(* IEC 61131-3 sources: ml2plc/benchmarks/st (part 5) *)

(* ---- GRU3.st ---- *)
FUNCTION_BLOCK GRU3_FB

    (* Model Inputs/Outputs *)
VAR_INPUT
    input_data : REAL;
END_VAR

VAR_OUTPUT
    output_data : ARRAY[0..2] OF REAL;
END_VAR

VAR CONSTANT
    weights_0_u : ARRAY[0..63] OF REAL := [-0.439286172, -0.480953246, -0.870120704, -0.69075644, -0.657077134, -0.589701712, -0.481989682, 0.11155279, -0.595970333, -0.522424638, 0.066479668, -0.477147967, -0.548775792, -0.440251201, -0.581660211, -0.851885259, -0.447049588, -0.158783153, -0.671791077, -0.790636778, -0.670549393, -0.228230864, -0.573410928, -0.463102937, 0.294410557, -0.154226393, -0.428246915, -0.419357181, -0.580893517, -0.450942427, -0.434489578, -0.354421765, -0.500179946, -0.272357315, -0.211979702, -0.347913235, -0.509638548, -0.571337163, -0.666850746, -0.102425002, -0.464207053, -0.692536592, -0.576414764, -0.25179112, -0.587422669, 0.197722241, -0.440594107, -0.0186067764, -0.233214989, -0.485925347, -0.624329388, -0.464201093, -0.771930814, -0.648595512, -0.712386131, -0.865132749, 0.0861109644, -0.699016631, -0.64285028, -0.76548481, -0.601012945, -0.522387683, -0.408631802, -0.428571761];
    recurrent_0_u : ARRAY[0..4095] OF REAL := [-0.0650523901, -0.129474998, 0.0260338224, 0.0695474148, -0.0666072816, 0.0774139315, -0.0643586814, 0.0473090038, 0.0519357473, 0.0531803295, 0.0508824363, 0.156312734, 0.0510548055, -0.0783398449, 0.0161208138, -0.0254090969, -0.0333776586, 0.0407715552, 0.0384992361, -0.00284529058, 0.0996260718, -0.0809974, -0.0287103504, 0.0288348049, 0.121645145, 0.129295856, -0.121905953, -0.0567066036, -0.0332944021, 0.10126324, -0.0619100034, -0.0120835379, -0.0321507938, 0.152141571, 0.0557904243, 0.0295200478, 0.0753500834, 0.0523380376, -0.045079913, 0.0743025169, 0.03919724, -0.0464075021, 0.0460194834, 0.0400504917, -0.0186564252, -0.0811230615, 0.0205100551, -0.0494997241, -0.0123350881, -0.0521072671, 0.0318819955, 0.0125074722, 0.086325638, -0.14838697, 0.0729614198, -0.123611242, 0.0608778223, 0.136695266, -0.0275732893, 0.103986211, 0.0964937732, 0.0746636614, 0.0518375002, 0.0131850429, 0.0481536575, 0.080832839, 0.00456657633, -0.0930995643, -0.0926894546, -0.104142435, -0.0113655347, 0.0689256042, 0.0391013213, -0.145912498, 0.0662881434, -0.125198483, -0.0359372757, 0.0683884099, 0.0814840198, -0.0467883013, -0.0385110751, 0.0412478335, -0.026082132, 0.00598589424, -0.0733542442, -0.0616489351, 0.0599563681, 0.0975151584, -0.102699503, 0.0168768093, 0.0567795113, -0.109472096, 0.0479807556, -0.0641779676, 0.0252187103, 0.0170151237, 0.052396398, -0.00687042344, -0.0297337286, 0.052699931, 0.0299865901, 0.0428941771, 0.143816575, 0.0724755228, 0.0308377538, 0.0377355814, 0.073744677, 0.100715749, 0.0200833306, 0.00330035621, 0.0808146596, 0.0683915466, 0.00292335614, -0.0387148745, -0.0278775394, 0.0165898427, -0.0266524255, -0.0119600557, 0.0607938841, -0.171499431, 0.00670967251, -0.0278419442, -0.0198536664, -0.0489947647, -0.0504177436, -0.0603820346, -0.0319245569, 0.0403733216, -0.0657449737, -0.0835127532, 0.074783206, -0.0822283328, 0.0527420714, 0.025356207, 0.00193200377, 0.0403062142, 0.011863322, 0.0911065713, -0.0981498286, 0.0448010042, 0.00674223201, 0.0832657516, 0.0133088445, -0.0096457703, -0.126930133, 0.0133038349, -0.0605163276, 0.0315002874, 0.163095102, 0.0627945811, -0.0319333449, -0.0184467398, -0.0260825343, 0.1507947, 0.0180257969, -0.113473095, -0.00113128126, 0.034390863, 0.158128366, 0.0736147836, 0.00302845053, -0.0366435051, 0.0202366989, -0.0454519801, 0.027544789, 0.00827108417, -0.116445266, 0.136078835, -0.0322153643, 0.0859275237, -0.0495595485, -0.0305913445, -0.0528560281, -0.0197725855, 0.0479791425, -0.0321966782, -0.0912050977, 0.08009094, -0.131073937, -0.073050648, 0.0158983283, -0.0129424734, 0.0236992333, -0.0654924586, 0.00780409761, 0.0303560495, 0.0224402416, 0.195856482, 0.104409501, 0.00386209786, 0.0270838067, -0.0308708213, 0.0765376315, -0.144475698, -0.00663482724, -0.0773844719, -0.0756781921, 0.0114769517, 0.07947056, 0.0525699407, -0.0490815043, -0.0797774196, -0.0738181025, 0.00899818353, 0.00655652676, -0.0247584134, -0.142790094, -0.0536906458, 0.0891067088, 0.0319167599, 0.0273121186, -0.0111009832, 0.0738681182, -0.0465159416, 0.10495235, 0.0167910457, 0.0170945786, -0.0259337351, -0.0238404684, 0.105175085, 0.0262874551, -0.0252160784, 0.0407399312, 0.0396488942, -0.000441844575, 0.0779087767, -0.101633228, 0.00611562654, -0.138864547, 0.0793924779, 0.0318161361, 0.00487799011, -0.0742631257, 0.0282261875, -0.0452414677, 0.103862561, -0.233050048, 0.0166822113, -0.0502803773, -0.105138443, 0.00815397315, 0.075144209, -0.000656956807, 0.00553116389, -0.0327767022, 0.0563323051, 0.00168130081, -0.0347454548, 0.0447669849, 0.0809304044, 0.0181033891, 0.0829547346, 0.0445744358, 0.0685421899, -0.0522269495, 0.10767854, 0.0401147828, -0.0274171568, -0.0556086302, -0.0181052946, 0.0614649057, 0.15146631, -0.107644446, -0.0519810207, -0.0192557313, -0.050705526, -0.00130558573, -0.00449152011, 0.0586461015, -0.00949175656, -0.161170155, 0.0415757112, 0.0234208908, 0.0994374529, -0.107094176, 0.0798551813, 0.00859866291, 0.00905988738, 0.17884995, -0.052185487, -0.00788529217, -0.0128635718, 0.0425841771, -0.0781655982, 0.0738354772, -0.0700388551, -0.0454497337, -0.0581207834, 0.0587512478, -0.129331231, 0.089504689, 0.0157049354, 0.0867228657, 0.0273658019, -0.0242159963, -0.0269595832, -0.0785825849, -0.0127460342, 0.0726092383, -0.0813473612, 0.0418060534, -0.098036088, -0.0871397629, 0.12796244, 0.115513436, -0.0840419456, -0.0282502882, 0.0339900963, -0.0615085512, -0.0237938426, 0.14066948, 0.0103495289, 0.0563306212, 0.0128910914, 0.0566199236, -0.0431611128, 0.0414758436, -0.0598706417, -0.00455367938, 0.010008106, 0.0502123758, -0.0128066251, 0.119871259, 0.169338882, 0.0573619083, -0.00254678726, 0.0632556081, 0.0658841059, -0.0489678681, -0.0136197284, 0.0332296528, 0.0304199178, -0.0101228859, 0.0340865031, -0.1463456, -0.0561735369, -0.078145586, -0.105770409, 0.021583017, 0.0442470424, -0.0132950321, 0.0343763754, -0.131868333, -0.0834302157, 0.0234229043, 0.0955413878, -0.00966519676, 0.133738831, 0.0799299628, -0.0209413245, -0.0201649163, -0.078094773, 0.00760632753, 0.10674265, -0.0504244342, 0.130076349, -0.0765756071, 0.0406672917, -0.0677179396, 0.0489641167, 0.0178483911, 0.0639283434, -0.0072317142, 0.0689901859, 0.0284034405, 0.0447224788, 0.080589503, -0.0753613785, -0.0883018747, -0.209824249, -0.025372155, -0.0194213465, -0.121756315, -0.0405391641, 0.0252318978, -0.113081403, 0.00984102953, -0.0379814059, -0.0696330816, -0.0607138053, 0.00136227917, -0.0684736297, 0.084016636, 0.0580409989, 0.0783514529, 0.038732525, -0.110764012, -0.184509531, -0.0218135417, 0.0410628468, 0.0143347979, 0.0210808329, 0.0938048959, 0.0952843726, 0.0369632132, -0.036689274, 0.0596370548, -0.101092562, 0.021979671, -0.00666903984, -0.0002728533, -0.102687143, 0.101846725, -0.0270557068, -0.0740891248, 0.0451480709, 0.0244468898, 0.0135530774, -0.0656716228, 0.126964301, 0.046734333, -0.0135823097, 0.104897536, 0.0116401128, -0.0351510793, -0.0270920806, -0.0317737125, -0.0427896604, 0.0606436953, -0.055717431, 0.0877809376, 0.0525183901, 0.0816646814, -0.123816505, 0.0268022101, 0.0949827731, 0.0286988262, -1.17924064e-05, -0.107156947, -0.0325826406, -0.176235095, 0.0207939055, 0.140304744, 0.0597819574, -0.0181577466, 0.117161281, 0.0191873126, 0.0420570076, 0.0174266361, 0.0642305687, -0.0820301622, 0.0203213636, -0.0772711709, 0.0149432123, 0.078445442, -0.031391941, 0.0178297423, 0.0258787423, 0.105060086, -0.185030684, -0.0465904325, 0.033022128, -0.0522077605, 0.18817015, 0.17154251, 0.0908443928, -0.114609689, -0.0463253893, 0.179783046, -0.0138813183, -0.0250236578, -0.0397495851, -0.0401404127, 0.0414455384, 0.00421553105, 0.00501056761, -0.0355476104, -0.0948569328, -0.0180768073, -0.0929266214, -6.38996717e-05, 0.0402616151, -0.04017644, 0.0292976033, 0.122893214, -0.0101269074, 0.0949848741, 0.0924490988, -0.0142561533, 0.034249723, -0.0345417485, -0.0720876306, -0.116285995, 0.0757803917, 0.0925265029, 0.0501283891, 0.0556523763, -0.0871114284, 0.063929759, 0.111392535, -0.0113485595, -0.0560661219, 0.0588565171, 0.0202990752, 0.0169391409, 0.0079346532, -0.0346361771, -0.0971538872, -0.107799433, -0.0225640163, -0.104902133, 0.0540932752, -0.0481065586, 0.0236067846, -0.135952473, 0.105642021, 0.0632608011, -0.0237644296, 0.0115678804, 0.0341430977, 0.00839798432, 0.00526432134, 0.00430205092, 0.063617371, -0.0232296586, -0.0100963581, 0.0232974347, -0.00805089623, -0.0783473253, 0.0837393031, 0.0119392872, -0.171118468, 0.0533629246, 0.0270157438, -0.0287604984, -0.024254458, -0.0379126333, 0.0377461091, -0.129247546, -0.0196368489, 0.121421359, 0.141241029, -0.0185492001, -0.0607114322, -0.118905656, 0.0243493672, 0.00225942954, -0.02267823, -0.114327833, -0.00651719887, 0.0233639106, -0.0216970742, 0.181706235, 0.0208011288, 0.019147085, -0.046965789, -0.0224242695, 0.170098603, -0.0381373689, -0.0911064297, 0.0361324437, 0.0604973882, 0.0523151048, 0.00412818976, 0.0810551196, -0.0951434225, 0.0870590508, -0.0168896336, -0.128554851, -0.0098116193, -0.0513504371, 0.0390418544, -0.0403953195, -0.101676092, 0.0051176697, -0.00728737004, 0.0545737594, 0.0803038031, -0.106364466, 0.0805499181, -0.0291947313, -0.0313916355, 0.00281906407, -0.00804035645, 0.0905895531, 0.138566479, -0.0726417452, -0.0388255194, 0.0526182652, 0.0332292169, -0.0458627641, 0.0337294526, 0.00538110361, 0.140382588, 0.0673478395, -0.0970090628, -0.0075024087, -0.0495187268, -0.0802161619, 0.123421639, -0.0669697523, 0.0695282966, 0.0278533436, 0.0633659065, 0.00612806296, -0.0442293584, -0.0825438574, 0.102498822, -0.0788070858, -0.00543309376, 0.00251733419, -0.112787522, 0.0541282296, -0.167338938, 0.0514628179, -0.0181294475, 0.00405258778, -0.144672319, 0.0080318721, -0.0168379508, 0.0630492195, -0.0291489959, 0.0451016501, -0.0668138266, 0.0430565365, 0.0430122651, -0.0329513662, 0.000115959905, -0.155294836, 0.0717644468, -0.0975336134, 0.0627146736, 0.0671754926, -0.0245223772, -0.0847209394, 0.103243671, -0.0160844456, -0.0769205019, 0.0603941306, -0.0861880928, -0.124118626, -0.0407451317, -0.0479636192, 0.0243864693, 0.0225671809, 0.0300183278, 0.0491476469, 0.0137792621, -0.101849571, 0.0899749994, -0.147746086, 0.00454038568, 0.0589881316, -0.0145919751, 0.135418221, -0.0641773641, 0.00270533562, -0.0761346892, -0.0119857313, -0.0468325913, -0.0362873077, -0.131199926, 0.0103873778, 0.119403817, 0.0133330058, 0.0119966101, 0.0999416485, -0.0672517344, -0.0058638826, -0.00583216175, 0.0140269175, -0.068311438, 0.03253185, 0.103045583, -0.0298009366, -0.0424585715, 0.049341809, 0.0334219672, 0.0674507618, -0.0598343313, -0.0709823295, -0.00613911822, -0.0969725773, -0.114717588, 0.0991245732, 0.0570561923, -0.019426886, 0.052425161, -0.0514192283, 0.0795131326, -0.0747317523, -0.0695499405, 0.0674568191, 0.0873003826, 0.183561474, 0.0483771265, 0.00801333692, -0.0329486541, 0.118730754, -0.024188403, -0.00475108158, -0.102296896, 0.0118699996, -0.0566260032, -0.00249518454, 0.0371045657, -0.0271308124, 0.0527189821, 0.0894352719, 0.186274648, 0.0990155637, -0.0390276238, -0.102149099, 0.0725147501, 0.0395716839, -0.0627084598, 0.0174233504, -0.118221872, 0.057125818, 0.00148172863, -0.0975891799, 0.0914200917, -0.0564012453, -0.00408087857, -0.115551151, 0.0542268753, 0.019407969, -0.04010031, -0.0751183033, 0.0519157983, 0.0462308973, -0.00663706008, -0.0179555975, 0.128559679, -0.0160329398, -0.0250887014, 0.0124615263, -0.0278950725, 0.0723621994, -0.0639792681, 0.0245549679, -0.0128075834, 0.0482278317, -0.00473110611, -0.0172997359, 0.0275737233, 0.0381074212, -0.0479229614, 0.15075548, 0.236614883, -0.12308903, 0.0457972996, -0.0270488337, -0.0401842594, 0.0367866941, -0.0665339977, -0.124880955, 0.0096321106, -0.0183932558, -0.0149384877, -0.0207794402, -0.0273507237, 0.0092713302, -0.137307942, 0.124376148, -0.000531716272, -0.0697186887, 0.0233710855, -0.0879249945, -0.0595673844, -0.0753096193, -0.10940744, -0.0863983482, 0.0678732842, -0.0699944496, -0.0533968322, -0.0598150305, -0.109890275, -0.0255937222, 0.0414171703, -0.028406553, 0.0625951141, 0.0562955327, -0.040136572, 0.102456421, -0.094027251, 0.0563254878, 0.0507630631, -0.100891739, 0.0114759067, -0.0276399851, -0.0600263849, -0.0218528342, 0.0106363287, 0.0762119591, 0.0472210646, 0.0182249043, 0.0761318132, -0.0902465209, -0.0155644314, 0.0497058667, 0.00891689677, -0.0575596653, -0.063269861, -0.0369747803, -0.0418471023, -0.0446194261, 0.0618177094, 0.163427904, 0.0439322591, 0.0151975229, -0.139614716, 0.0382574834, 0.0647403747, 0.0044741584, 0.0366933271, -0.0847294405, -0.098235622, -0.102225974, 0.0730303079, 0.0709254742, 0.114724368, -0.058182843, -0.0275532752, 0.0699310824, 0.073567912, -0.118505709, -0.0922444239, 0.0654501319, -0.0442147106, -0.0973261297, 0.0649150908, 0.0473677218, -0.0438311286, -0.0123466263, -0.0506518409, -0.00112013146, 0.0114555079, -0.225004256, 0.0179542284, 0.00154356682, 0.0197916869, -0.0964033976, -0.0149603887, -0.0931083262, -0.0858175233, -0.0240392219, -0.0473877937, 0.0356729813, 0.0953858122, 0.0516837016, 0.000944763422, 0.000391166657, -0.0161546711, 0.0617823638, 0.0323178768, 0.0746243447, -0.0289416965, -0.132081941, 0.0347845852, -0.00957541913, -0.146093175, 0.00121896248, -0.088182658, -0.0529079251, 0.00144353509, -0.10963767, 0.0711052567, -0.130099729, -0.127687454, -0.0238898639, 0.0237303749, -0.0463271476, -0.0377245843, 0.146435305, 0.0406003967, -0.00347847119, 0.0402232558, 0.0606766082, -0.0170659591, 0.00456166919, -0.0581656583, -0.0257244669, -0.114303187, -0.109322034, -0.000124797225, 0.0906794146, 0.0998297706, -0.0660899505, -0.0273227766, 0.00623180624, -0.0511037856, 0.0518054552, -0.130383685, -0.104795009, 0.00977518409, 0.0961738452, 0.0406313278, 0.0335147977, -0.0768964514, -0.021825349, 0.114472322, -0.0201997422, -0.0598041527, -0.0629845262, 0.105795145, -0.0276378486, -0.0260668173, -0.0237419959, -0.0401881412, 0.0480453372, 0.0071930117, 0.00337004848, 0.0128219994, 0.067926839, 0.102826566, -0.0290449653, 0.123585209, 0.0586936176, -0.129759327, -0.0223709345, -0.116297573, -0.0687413886, 0.109364361, -0.016150102, 0.0699984133, 0.0204590037, -0.0488001369, -0.0933896229, 0.11484497, 0.146208376, -0.0152992923, 0.0223931447, 0.0693335161, -0.126214027, -0.0157451089, 0.020451, -0.0159052685, 0.0770635083, -0.165799066, -0.0527213998, -0.080435276, -0.0827942193, 0.0621753186, 0.00343356607, -0.0961636975, 0.0286911149, 0.0452868044, -0.0499980301, -0.0868136883, 0.050965365, -0.0764427632, -0.0663457513, 0.0639655739, -0.121900126, -0.0106822588, 0.0629351214, -0.0268343873, -0.0563602373, 0.0208010022, -0.0950316712, 0.0376925468, 0.0941148102, 0.0284186527, 0.0386470295, -0.0649496838, 0.00324150547, -0.0536398701, 0.0218845457, 0.101267442, 0.00504809991, -0.0866092741, 0.0529379621, 0.0938520655, 0.0396423154, 0.127945945, 0.11368385, -0.0549047142, 0.114498168, -0.0241714753, 0.0520189852, -0.0362896509, 0.0509226546, -0.165635839, 0.0881007984, 0.0160411, 0.024631137, 0.0659909099, -0.0762100443, 0.0427479185, -0.00694125425, 0.143184051, -0.149732918, 0.0110863149, -0.0155461309, -0.13748844, -0.0504982434, 0.025665462, -0.0429363698, -0.0277443547, -0.0475423895, 0.0285833944, -0.0735700205, -0.144904912, -0.0755529851, -0.0403888598, -0.0527475253, -0.000688489527, 0.101409346, 0.0988431573, -0.0909979939, 0.0660976842, 0.063818492, -0.00707271695, -0.00301229395, -0.0202014614, 0.0212209262, -0.0612271912, 0.142480314, -0.102822497, 0.121017784, -0.0435582623, 0.100066409, -0.0312062576, -0.0822519436, 0.057339862, 0.0568015501, 0.0269984789, -0.0163367614, -0.0477057099, -0.101986229, -0.00421534479, -0.179487348, -0.0764475316, -0.0430073664, -0.0425812863, 0.0527436584, -0.13650541, -0.00514466688, 0.00624288665, -0.0491546728, -0.0670409873, 0.0240444243, 0.035694059, -0.0549894422, -0.0163852815, -0.0803953186, -0.0258201156, -0.0284036025, 0.0236114748, -0.0177096128, 0.0899664611, -0.136392832, -0.0611273237, 0.0208600666, 0.0675291047, -0.033409629, 0.183402792, -0.0179462973, 0.0402268246, 0.0538903326, 0.0605378859, -0.00444559008, 0.00593124051, 0.0584437177, -0.0465901792, 0.0367346182, -0.00531690102, -0.0891991258, 0.108523466, -0.000754443929, 0.0853905827, 0.0139564294, -0.0571048073, -0.0341003574, 0.0744261444, -0.0160620511, 0.0420818552, -0.072983481, 0.105422221, 0.0132888965, -0.156731457, 0.0509976372, -0.00400068983, -0.0257125702, -0.010336509, -0.0466502346, -0.0191403441, -0.0370061398, -0.0619829483, 0.0589080006, 0.085831672, -0.0815126747, -0.148456261, 0.035992898, 0.00954711344, -0.0224743038, 0.0770518929, -0.0347290412, 0.0506613515, -0.0776980445, 0.0472105034, 0.206908733, 0.0290955547, -0.113211304, 0.146189138, 0.0581367761, -0.0555344708, 0.0266725048, 0.0476324111, -0.0754805133, 0.0204973966, 0.0354307257, -0.0414481908, 0.0941888317, -0.142457843, 0.01902714, 0.00608063489, -0.142902017, -0.00904501975, -0.0471438207, 0.0187765174, 0.0261135101, -0.0300621614, 0.0145887854, -0.0236850809, 0.0117516052, -0.0394856744, 0.0042070318, -0.094953917, -0.107410148, -0.0374321714, -0.0109713413, -0.0557455085, -0.0535232276, 0.0823234618, -0.0228107423, -0.145991802, -0.142637998, -0.0141612738, 0.0681499764, -0.0601133108, -0.048684977, 0.028852893, -0.0919774398, 0.0113884229, 0.0250541884, 0.108147934, 0.125753194, 0.040229924, -0.0862782151, 0.0393346809, -0.0627611578, -0.0139939766, -0.0519772731, 0.0389488079, -0.0385627151, -0.0904045478, -0.0797261447, -0.0159214437, -0.00528162252, 0.00593003258, -0.0402139761, -0.100702733, 0.0729726627, -0.0694422498, -0.101501249, 0.026667282, -0.0488509983, -0.0981456414, 0.0895740688, -0.0577398948, -0.0186711848, -0.00111833401, 0.000157465227, 0.070121713, 0.110388353, -0.0305795819, 0.00751299458, -0.159779117, -0.0279579163, 0.0977309942, -0.00896156579, 0.0305966716, 0.0786327869, 0.0876243636, -0.0386611111, -0.0101302303, -0.160905316, 0.105016418, -0.0753878355, -0.0497038662, -0.0164555032, -0.0430143699, -0.045727957, -0.0521295182, -0.00294361566, 0.0361426473, 0.00889566541, -0.0249266233, 0.0799256191, -0.0287304316, -0.0792678446, -0.0854634121, -0.050208319, 0.0208053384, -0.0348147191, -0.114404887, 0.0125034805, -0.0298862718, -0.0686926022, 0.0476176292, -0.0698538199, -0.0111048371, 0.0644094273, 0.0129547417, -0.0727717876, -0.0681286678, 0.13020657, -0.027219126, 0.0698305443, 0.0116916075, 0.14363949, -0.113594539, -0.000844738446, 0.0082028266, 0.0454428382, -0.00381363602, 0.0126697449, -0.187009782, -0.0268669054, -0.128417894, 0.0594988614, 0.0632686764, -0.138941869, 0.107257128, 0.112114236, 0.0334792137, -0.0564817488, 0.000689910725, 0.110511348, -0.116754688, 0.00211306289, 0.0736983195, -0.00167888403, -0.0343024731, 0.0968845412, 0.0107437428, -0.0036681965, -0.0132405106, 0.0795757398, -0.0983074009, -0.17490913, -0.0407146737, 0.129254073, -0.00595551729, -0.0102427769, -0.0578140169, -0.00301308557, -0.0852808505, -0.00178171322, -0.0460724831, 0.0447371192, -0.0961295962, 0.028552942, -0.0433705673, -0.0627188534, 0.0271210223, -0.0610382147, 0.0640244409, -0.00287532061, -0.0704336017, -0.145652339, -0.163796186, -0.157491252, 0.0173620582, 0.234602943, 0.0841561556, -0.00848647393, 0.0434717573, 0.148942828, 0.0672514886, 0.0184065942, 0.0249046497, 0.0132941119, -0.065047577, 0.0867860764, -0.0353404805, -0.0038694879, -0.00896554533, -0.030097058, -0.0858454853, 0.0279321168, -0.0583353005, -0.114406154, 0.0291701369, -0.103932366, 0.10427992, -0.0508416221, 0.0617097132, 0.0285572838, 0.035257943, 0.0155800534, -0.174241856, -0.0110836942, 0.0528832301, 0.170236602, -0.0480959341, 0.0568181984, 0.0429964401, -0.0398594141, 0.142875105, 0.0198408999, -0.0234815422, 0.0413020328, 0.0316126868, -0.0242498852, -0.085475266, 0.064656049, -0.091913268, 0.00903178845, 0.0966716036, 0.0519700944, 0.050653033, -0.171772823, -0.0414884649, 0.0218126774, 0.0484813899, -0.0342098139, 0.0431513302, -0.0775837302, -0.0194175802, 0.0608915053, -0.0958085358, -0.0525278524, 0.172223568, 0.0520742238, 0.0220057666, 0.108987883, 0.130237713, -0.107932687, 0.0317093804, -0.0324443653, 0.0835223198, 0.199562863, 0.148373321, 0.112411663, -0.0236171074, -0.0052724164, -0.0620609745, 0.0111017656, -0.0111301467, 0.0467493832, -0.0206472725, 0.00297360634, -0.0119733168, -0.0970944092, -0.0316341296, -0.0132295629, -0.0338335037, 0.0520780794, 0.12766394, 0.068843931, 0.195665359, 0.0558646694, -0.0955600888, -0.077448085, -0.0211934205, -0.0296740029, 0.00166139007, 0.0591102466, 0.0120509472, 0.0354253165, 0.157639459, 0.0244942661, -0.189979553, 0.0354224183, -0.0612734891, 0.0376649685, 0.205627829, 0.00432812702, -0.02739764, -0.0818298906, -0.120526254, 0.0180814825, -0.000375784934, -0.00592299784, 0.106825203, 0.0165459365, -0.0205880832, 0.111172318, 0.0138723217, 0.0164856389, 0.0165480785, 0.062894091, -0.0380115025, 0.0288346447, 0.0361645594, 0.0495932661, -0.0227110572, 0.075070098, -0.0742200911, 0.0544882938, -0.100449175, 0.0435093604, -0.0736430958, -0.037141487, 0.0257380009, -0.0985285342, -0.0582001545, 0.0263903867, -0.133239761, 0.105293542, 0.0509466119, 0.0149480924, 0.00264212303, -0.0803615153, 0.016234152, 0.059326943, 0.0166629646, 0.129690155, 0.00954441354, -0.089779377, 0.00573088974, -0.00493869651, 0.0591944307, 0.104186028, -0.0218419582, -0.00641731732, -0.0487543717, 0.0456377119, 0.0427142642, -0.0505627245, -0.0945144147, 0.0202183761, -0.0657929033, 0.0831303746, 0.0750920549, -0.0910624713, -0.0225744545, -0.124150276, -0.152486816, -0.0330677181, 0.0442869589, -0.0471795797, -0.134105518, -0.0558637902, 0.0834738016, 0.0108987726, 0.0160592347, 0.108882993, 0.0598439351, -0.0831453726, 0.0973557979, 0.0623315871, 0.0383794159, -0.00982961245, 0.0576453581, 0.0494841523, 0.0718243048, -0.0572519116, -0.0411631241, 0.0534142479, 0.0589003153, -0.0547911972, 0.0755654052, -0.0815965533, -0.0117946044, 0.103706859, 0.0667564943, 0.0903166533, -0.038736023, 0.018129129, 0.060453929, -0.0346493199, -0.0850336775, -0.00476394966, -0.046710752, 0.0143833831, -0.015953254, 0.0134185404, -0.0532437861, 0.017363999, -3.44109721e-05, -0.149937063, -0.0611102469, -0.0427428, -0.00926883332, 0.0374133512, -0.0711838678, 0.0258399993, -0.00872873422, 0.0366705805, -0.0147527959, 0.057190951, -0.0818497464, -0.0571168959, -0.0519183539, -0.0537600778, 0.0200558268, -0.0356059968, -0.0514560342, -0.115551762, 0.0614381582, 0.0904121846, 0.0550923347, 0.09433157, -0.0337151326, 0.0622163899, 0.0612645894, 0.0891919881, -0.0207224004, -0.0534750856, -0.0296462215, -0.0158423334, 0.0887120888, -0.0703074336, 0.00989756919, 0.130590975, 0.0778346881, 0.00399551541, 0.108989477, -0.00454995502, 0.0528934747, 0.121316366, 0.0511680767, 0.0755439252, -0.0733139291, 0.0752391368, 0.0770118833, -0.000957053155, 0.0114189107, 0.0590100586, 0.00575780775, -0.0877712369, -0.0187948812, -0.0657808185, 0.0406781025, 0.0595240593, 0.00684884563, 0.0149538293, 0.00922561437, 0.114996634, -0.0660880059, 0.00837289169, 0.0117377583, 0.0296314899, 0.0261435769, 0.14703317, -0.0287333839, -0.0299690161, 0.00223761285, -0.0870166644, 0.0896945298, 0.0500493981, 0.0744577274, 0.013104694, 0.0748228654, -0.0941333324, 0.0413618535, 0.0238855034, 0.0836726874, -0.0697423667, -0.121260516, 0.0637812093, 0.0396960527, 0.0819698572, 0.0435053259, 0.0501765572, 0.00983571447, 0.0299814939, -0.0600497648, 0.04743848, 0.0918345079, -0.192011252, 0.185129195, -0.132771015, -0.0218426287, 0.0106724147, 0.0418993495, 0.07511691, -0.0415916629, 0.0514673628, 0.0512605757, -0.101605847, 0.0378510244, 0.167794362, 0.0514133871, 0.0400778428, 0.0447239429, -0.0781334937, 0.0273859277, -0.0525638573, 0.0734867603, -0.0286831781, -0.0886658579, 0.0515142232, -0.117384307, -0.161638945, 0.110049561, 0.0852481127, 0.035481941, 0.0158129036, 0.088354513, -0.00556714088, 0.0537756681, -0.0467627533, -0.00163430907, 0.0605735257, 0.109923393, 0.0235946123, -0.0543056205, -0.0435014889, -0.0780219436, 0.0887052789, 0.0288573951, 0.0956314802, -0.119991414, -0.0950825363, -0.0577025861, -0.00233832374, 0.0321475305, -0.0296782143, -0.13685973, -0.0840527713, -0.115250856, -0.086614266, -0.0719218403, 0.0350063443, 0.0287500955, -0.0230677407, 0.13799727, 0.0648974031, -0.0969269872, 0.0105827358, 0.0187805891, -0.0817399919, 0.134309664, -0.0834898725, 0.0636503398, 0.0892517194, -0.0689574108, -0.0209724437, -0.00819023326, -0.00418700883, -0.0096282959, -0.0291463416, 0.0508619435, -0.0297213681, 0.0173015445, 0.00606717542, 0.0537274331, 0.041289378, 0.00145007065, 0.0465077683, 0.130988643, -0.0168933291, -0.0218317695, 0.0134224519, 0.00168778002, -0.00168193318, -0.0929443315, 0.0933136791, 0.0271413755, 0.0012512356, -0.0429633558, 0.00577729195, 0.0381182507, 0.0506631732, 0.0104230382, -0.0946019739, -0.146492317, -0.0122778527, 0.0851407722, -0.00430129794, 0.0286120772, 0.0544554926, 0.000575783662, 0.0418614075, 0.0509960353, 0.235207349, 0.0231721811, 0.03219245, 0.0219864137, 0.0771256983, -0.0475538969, 0.0167042073, 0.043224901, 0.0525902212, 0.0109413685, 0.0310349781, 0.0262097772, -0.0763660222, 0.0886459798, 0.0879353359, 0.0266202651, -0.012050109, 0.0364502966, 0.110469103, -0.0649368986, 0.137989163, -0.00345457532, -0.00076057855, 0.0495130271, 0.0963264555, 0.0292368587, -0.0136958137, -0.0916326419, -0.09134987, -0.143160895, 0.0552338138, 0.0943126529, -0.0341492742, -0.046550639, 0.0415712446, -0.190018594, -0.0170447789, 0.0271576829, -0.0791434646, -0.0259393826, -0.0358110107, 0.114700861, -0.0451665968, 0.00859330222, -0.0176053625, -0.0665916502, -0.10659565, -0.0103667611, 0.0607822947, -0.0335317552, -0.0578957722, -0.0600993, -0.0143982824, -0.0169818364, 0.0747436732, -0.0824175626, 0.0734613463, 0.0172847919, 0.0679807961, 0.0354374871, 0.0221069511, 0.0698141977, 0.103264622, -0.0643693283, -0.0904196575, 0.0209124722, 0.0533089563, 0.138175309, -0.0808143616, 0.0518090576, -0.04021056, 0.0328150876, 0.0717661381, 0.0629613996, 0.104841411, -0.0416442491, 0.0719090104, 0.059182696, -0.15314886, 0.0215544775, -0.0130644813, 0.114227138, 0.00902843848, -0.0153322266, -0.13713704, -0.0476132631, -0.119293369, -0.0679454356, 0.122949339, 0.0693741217, -0.0994557068, 0.0399324894, -0.0314740613, -0.000461213291, 0.00562566333, 0.140679166, 0.0478050821, 0.108278081, -0.0659516081, -0.00195731036, 0.0559609048, -0.0145426169, -0.0347096696, 0.0258138534, -0.0312658995, -0.0548630729, -0.0697729737, 0.0109880194, -0.0809436738, 0.0592633858, -0.00464516133, -0.107980013, -0.0189933032, 0.0685023963, -0.0257080533, 0.074374266, 0.0587298237, -0.056436114, 0.0454883464, 0.0601172373, -0.0381640494, -0.0409820527, 0.00114455202, 0.0928920731, -0.0341993608, 0.01902242, -0.0319391079, 0.0252930373, -0.0232422352, 0.00733191008, -0.0100106141, -0.056417428, -0.0364283621, -0.0677095577, -0.0730913579, -0.0449670255, -0.112897381, -0.0383246988, 0.0491045266, -0.00531547517, -0.069094345, -0.0260258541, -0.069829613, -0.0624606349, -0.133198172, 0.0081421202, 0.0548977219, -0.0505369082, -0.021252159, -0.0689540803, 0.0545859337, -0.00222222786, 0.0334032364, 0.0678267553, 0.0439778864, -0.0222215448, 0.0925648957, -0.0336760692, 0.0680503026, 0.067150943, 0.169242263, -0.127817169, 0.0840600431, 0.0119890599, 0.0408258699, -0.0424239263, 0.0234956034, -0.0822051615, 0.127012193, -0.018799413, -0.0460282192, 0.00472665858, 0.0129743032, 0.00426072115, 0.0703843161, 0.0145993857, 0.119512692, 0.0195069741, 0.0493210033, 0.0875848681, 0.100930437, -0.0486361198, -0.0475119352, 0.0138504477, 0.208870143, 0.0598653406, -0.120691441, -0.0283632614, 0.0474334285, 0.00298458477, 0.067226842, 0.150975302, -0.0541105792, 0.0256627742, -0.0438354947, -0.0542730018, -0.00181115232, -0.105021812, -0.0556066297, 0.0338146091, -0.0549245104, 0.0143369175, -0.0539371893, 0.0432943441, -0.0535181016, 0.0258672144, -0.0821818784, -0.0270294957, 0.0225534495, -0.0127259865, 0.0120830201, 0.0125242695, -0.0619680323, -0.087769866, -0.011979159, 0.15043509, -0.10600248, 0.0364335105, -0.061168395, 0.0152373658, -0.0460021645, -0.109346926, 0.0364494249, 0.00472447462, 0.102088474, 0.0257884748, 0.0533271991, 0.0729068294, 0.00768535864, 0.112634815, -0.0691387504, -0.0601366162, 0.0453425571, -0.0314094163, 0.0349893384, 0.0256387182, -0.00378753617, 0.0768208951, -0.0505088195, 0.0269892886, -0.00966024026, 0.043255616, 0.00924504176, -0.00864656642, -0.0591106378, 0.0949935094, 0.0487293713, -0.0323852487, 0.0252678767, -0.0076211039, 0.111468486, 0.0816216171, 0.037076585, 0.00846009329, -0.0315636173, 0.0731508285, 0.10651087, -0.034380503, 0.11133229, -0.00250713434, -0.0430554636, 0.165012404, -0.0231795907, 0.0274878461, 0.0483577475, -0.0599443391, 0.0668406785, -0.0761960298, 0.0266923569, 0.00958470255, -0.0702683628, 0.0497920513, 0.0786102861, 0.0636078268, 0.021653505, -0.0515439399, 0.0863124654, 0.0131225679, 0.054686375, -0.0462396704, -0.0317671299, -0.0549215488, 0.0526956804, 0.0599532798, 0.0697892085, -0.0464518778, 0.0786490142, 0.0801427364, 0.135556832, 0.0811728388, 0.0162178427, -0.100880146, -0.0164203923, -0.09579698, 0.00686951773, 0.0556715578, 0.154748037, -0.0384738967, -0.0697567761, -0.0658533126, 0.0563082471, -0.0837014914, -0.120353431, 0.0157528166, 0.11380288, -0.0509812795, -0.184196651, 0.140463933, 0.184002206, -0.0414622352, 0.156096339, -0.0566040725, 0.127726138, -0.135966212, 0.0285594333, -0.0718551874, -0.115175165, -0.0160157103, -0.0541006215, -0.0331212506, 0.0474987626, -0.0206688922, -0.0896792114, 0.0121970847, 0.0920595378, 0.0294709988, 0.00489335647, -0.0136370827, -0.0876406729, 0.0430216789, 0.040562436, 0.0644720495, -0.0303485282, 0.122684225, -0.165262386, 0.0237433817, 0.0427406877, -0.0989692509, 0.109646007, -0.00851122849, -0.00903640781, 0.0406889617, -0.0505370982, 0.0931062922, 0.0305767655, 0.062228322, -0.0525234826, -0.102460198, 0.0645387992, 0.0533145741, -0.206492513, 0.0133064939, 0.0559483878, 0.0906168297, -0.0595491901, -0.0381035544, -0.0209744722, 0.0858725533, -0.0881853476, -0.0829888582, -0.112644993, -0.0684021264, 0.0686395615, 0.0265239459, -0.131407306, 0.0274842456, -0.166530743, -0.0467720069, 0.01258785, -0.0204203501, -0.100700855, -0.110235199, 0.0999744534, -0.067055054, 0.0858595446, 0.0564401224, -0.0734795183, 0.0984800607, 0.000628214737, -0.100944236, 0.050260745, -0.0384647399, -0.117021114, -0.00581525033, -0.118169144, -0.0531625077, -0.110389993, -0.0503460653, 0.048195146, -0.0405612253, -0.0432871655, -0.0308589637, 0.0801219493, 0.022040328, 0.0507384911, 0.0382968932, 0.0698082075, 0.0641338974, 0.00569984969, 0.0396882296, 0.019232735, -0.0757699236, 0.0707999244, 0.0159386508, 0.0308304802, 0.0468344912, 0.0355247855, 0.0718743205, -0.0121067222, -0.0105456598, 0.0769912899, 0.0374626517, 0.0373739302, -0.0699928999, 0.0847563297, -0.0230606366, -0.0388202295, 0.103667095, -0.128558323, -0.046710927, -0.0857155696, -0.0199590083, 0.151113033, 0.121398017, -0.0511609092, 0.0720787272, 0.0295494981, 0.0245097131, 0.0487351418, 0.106066108, 0.0537618995, -0.0159866326, -0.156366274, 0.0242971852, 0.159070209, 0.00524867978, -0.0994271263, 0.0449088961, -0.0211867951, -0.0390554033, 0.077684395, 0.0779460743, 0.0523676053, 0.0588788539, 0.00485968869, -0.0598566197, 0.013074277, -0.0545727536, 0.0519137047, -0.0330678336, 0.0389791094, 0.0678062215, -0.125330731, 0.0168909654, -0.0826457739, 0.0725395679, 0.123465694, -0.0158160534, 0.111778371, 0.0435737222, -0.0315076187, -0.101733088, -0.0460981056, 0.109187216, 0.0352550186, -0.0129180942, 0.171947062, 0.0519051552, 0.0502665862, -0.0938540846, -0.0937337503, 0.0209997464, 0.019742392, -0.0841773972, 0.065202415, -0.0252768025, 0.0767172575, 0.132501423, -0.041324053, 0.013803497, -0.0191468094, -0.0501539335, -0.0029412359, 0.0496336222, -0.0182176437, -0.0242415741, -0.0769018009, -0.0222259574, -0.0599570423, -0.0785850957, 0.0483198538, -0.158214718, -0.102507047, 0.0461308062, -0.0683883056, -0.0411389247, -0.0950894877, 0.100902207, -0.00471645314, 0.00992084574, 0.0858963057, 0.0614297986, 0.117100388, -0.0240918137, 0.0707100406, 0.132806167, -0.116088726, 0.00466614868, 0.0599054582, -0.0183604769, 0.0550542325, 0.0614843927, 0.00322095677, 0.0649169087, -0.0379064046, 0.0497901775, 0.0719092637, -0.154971763, 0.117400832, -0.0427108631, -0.0316413231, 0.0339113027, -0.023429919, 0.0100743826, -0.0608712286, -0.0393153466, -0.0721224099, -0.019769663, 0.0305335447, -0.00641385559, -0.0616339706, 0.0896052122, -0.0450256616, -0.0206921622, 0.0356086567, -0.0749701783, -0.0147821922, 0.0112537732, 0.097909674, 0.0569019616, 0.0509603657, -0.072360158, -0.0678833127, 0.0768040866, -0.110155649, -0.0740643889, -0.094099097, -0.0108416183, 0.060312368, -0.0583655126, -0.104549289, -0.218230203, 0.0970755219, -0.0179643556, 0.100377582, -0.0316814184, 0.0642254949, -0.0426855683, -0.0397533514, -0.0256710351, 0.0136024654, -0.0055637476, -0.200856268, 0.0169277843, 0.078002885, -0.14920415, 0.0111826845, 0.0809670985, -0.052739054, 0.0624899492, 0.0306037925, -0.0699668303, -0.0787069276, 0.0403862, 0.0614282824, -0.00977569167, -0.0857097507, 0.103655919, 0.124205105, 0.0120967291, -0.0551354587, -0.042931851, -0.0854013264, -0.0685761273, 0.0644985661, -0.0383845717, -0.0024125278, -0.063759163, 0.0521320626, 0.124909475, 0.111597076, 0.0148241296, -0.0615106374, 0.0415096581, -0.0933477953, 0.0717638135, 0.0793121159, 0.0742387325, -0.0539873391, 0.00332836807, -0.0300874971, -0.0831861719, -0.0381114557, 0.0751383677, -0.113011718, -0.0112683401, 0.0606956668, -0.172200784, 0.00429096073, 0.0602080822, -0.137329713, -0.090002872, 0.0323414132, -0.0719932467, -0.140211582, -0.0128612556, 0.0361765325, 0.0980945751, -0.010059149, -0.0461915061, -0.0139733413, -0.0086908564, 0.0273868591, 0.0861311108, 0.0443583541, 0.0680558532, -0.0228823051, 0.0917587876, -0.100482099, -0.0359601751, 0.122452661, -0.0542502478, 0.027852837, 0.0694331974, 0.00141336536, -0.109030351, -0.131108165, -0.162553549, 0.0753331035, 0.0134982076, -0.0366807505, -0.0386078581, -0.00658005895, -0.0914643705, -0.0252701417, 0.0801979229, 0.0021053683, 0.0746067539, 0.0221132264, -0.00809657201, 0.12774621, 0.0647266284, 0.0584487692, -0.064717263, -0.0277714748, 0.0883828104, -0.110183463, 0.0370126292, -0.0138474237, 0.0159780867, -0.016058648, -0.0404856317, 0.0766953677, -0.10419903, -0.141589358, 0.144594938, -0.109949932, 0.0647953376, -0.0917214304, -0.0102576986, 0.0803454667, -0.0682678446, -0.0576918498, -0.00570382923, -0.0834980905, -0.00225776061, 0.0470857583, 0.0150479516, 0.042511303, 0.0727005824, -0.128937468, -0.0655451864, -0.0340349115, -0.0954819322, -0.0620098263, -0.172165602, 0.0282320231, -0.0634708181, 0.0287884995, -0.171313956, -0.152317584, -0.0844539329, -0.0112288594, 0.120956585, -0.0573068708, -0.0637781844, -0.0221945029, 0.0527748689, -0.0105367936, 0.0755724683, -0.0467769243, 0.0614911839, -0.135969311, 0.105225481, 0.156952262, 0.0370586067, 0.15616776, -0.0840421766, -0.0951181725, -0.0149632134, 0.0322490297, 0.0670348257, 0.130084842, 0.0266189165, -0.0625972375, 0.00457772799, 0.0979716629, -0.00742265768, 0.118027046, 0.0416464359, 0.0718041658, -0.0798822492, 0.0614944771, -0.091669254, 0.00349572115, 0.0355406329, -0.0315599367, -0.0384840742, 0.0917298421, -0.0112617295, -0.0501065403, 0.0413927324, -0.0128761344, 0.0815452337, -0.0172406044, 0.130260676, -0.0188278407, -0.0011760518, -0.0579140298, 0.0338388719, 0.112019926, 0.0727667958, -0.00672438648, 0.00536828581, -0.0465201363, 0.00503383111, -0.0678088143, 0.0614547953, -0.106527671, 0.108292408, -0.0248407945, -0.0236443058, -0.0199482255, 0.0271114185, -0.0999043509, 0.0715598539, -0.0604586042, 0.0159977283, 0.101002097, 0.0251209512, -0.0435456298, 0.0404220521, 0.0287586413, -0.00336176204, 0.00109383767, 0.188423753, -0.0121071227, 0.0344866551, 0.0340253003, 0.0281979404, -0.020309411, 0.112903818, -0.0353781506, 0.0142767709, -0.0821403638, 0.0994499773, -0.0324760824, 0.108188063, -0.000992564484, 0.0135587398, -0.13331835, 0.0263649207, 0.0262281783, -0.0107785314, 0.0589572713, -0.0244767591, 0.0194578413, 0.0756996647, -0.124957405, 0.0433721058, -0.0131629705, 0.00946621597, -0.0793711543, 0.0270108059, -0.0341884941, -0.0752030089, -0.104312092, 0.0887307227, 0.0835861564, -0.0330076404, 0.162407339, 0.0132059641, 0.0758589134, -0.0445123538, 0.0380469374, -0.000802192837, -0.0470603779, 0.135118589, -0.0318722017, 0.000692218542, -0.0302473344, 0.114358984, 0.00851656124, -0.126637205, 0.0359836593, -0.00687000901, -0.0121891778, 0.0134458765, 0.0366071984, 0.0142765157, 0.0222175159, 0.000126404688, -0.0124760196, -0.0359021425, -0.0431295522, -0.0966509655, -0.0100903204, -0.0353743173, 0.0715210587, -0.081053026, 0.0999638587, -0.019016372, -0.0239935089, 0.00648718514, 0.0153071349, 0.012509536, -0.0589868091, 0.0743578523, 0.0191438161, -0.0187446624, -0.0208187737, 0.00617905706, 0.160369337, -0.025553029, -0.164978892, 0.0432493463, 0.052146554, 0.00317490846, -0.0926495492, 0.0303232074, 0.125212759, -0.0296045784, 0.024818765, -0.0604889244, 0.0330986381, -0.0673882589, 0.0580419749, -0.103213176, 0.0422696471, 0.0958758742, -0.0965849459, -0.00950852036, 0.0918902084, -0.068486914, -0.12186332, 0.0030031316, 0.131197795, 0.00548650976, -0.00403932016, 0.0173820686, -0.0290936418, -0.0979100466, 0.0117043052, -0.118052997, 0.0237339474, 0.0828405619, -0.103721827, -0.0860361904, 0.065347068, -0.0213578418, -0.00391968619, 0.0236401204, 0.0144597851, 0.054736048, 0.0231402628, -0.0840564817, 0.0548789054, 0.130872041, 0.00752765685, 0.0240224563, -0.00454153167, 0.0319019519, 0.063471444, 0.0219805893, -0.0952587053, 0.0340296663, -0.00117000053, 0.0152508952, -0.0606811643, -0.047678858, -0.0131933, 0.0261857826, 0.0161818042, -0.0327050351, -0.000714013353, 0.062065091, -0.00254658936, 0.0433586389, -0.0278949924, -0.0263456665, -0.0698257834, -0.0431765653, -0.0144449733, 0.126253545, 0.0126124537, -0.0509497039, 0.000468326733, -0.00036503002, -0.0447247848, -0.0417972095, -0.0157134756, 0.025018584, 0.0699072331, 0.0882948413, -0.0929879695, 0.00265961373, 0.00323988311, 0.00498005841, 0.00374827161, 0.0459985994, -0.0181076191, 0.0145163927, -0.0408614576, 0.0804381892, 0.0233130399, 0.00467471313, -0.0549203008, -0.0559486635, -0.0105915256, 0.0502482392, 0.0795770064, -0.162366003, 0.000561785651, 0.00131846406, -0.0867253095, -0.0644728467, -0.0526860952, -0.0904279724, 0.0680651143, 0.0549977012, -0.0198836289, 0.0226633139, 0.124892376, -0.0483702384, 0.025002405, -0.00761365099, -0.193545878, 0.116730005, 0.0593729913, -0.0828391612, 0.159838334, 0.0629694685, 0.0573315881, 0.034116488, 0.122743621, 0.00297184102, 0.0652865767, 0.0233377926, 0.0117186205, 0.00482350402, 0.00210875086, -0.133521438, -0.00392506085, 0.0866617113, 0.0794988349, 0.0499842316, 0.123910151, 0.111768797, 0.00231364276, 0.0588010177, 0.0367658734, -0.0292860344, -0.0044385083, 0.0357940495, -0.000611573458, -0.0268944241, 0.0574458987, -0.0747600868, -0.095133923, -0.0577830747, -0.0673853606, -0.0535354726, -0.000596318394, -0.035483066, 0.0208486263, 0.0316488817, -0.195054889, 0.0611732341, -0.0187134333, -0.0486381464, -0.0301590897, 0.0133740138, 0.068864353, -0.140572727, -0.0387248173, -0.0527053252, 0.108385712, -0.0978539661, -0.0396942608, 0.055108171, 0.155904785, 0.128576532, -0.0461218059, -0.00189863332, 0.0483641289, 0.0793901011, 0.0244574696, -0.0248883814, 0.108808123, -0.118639104, 0.0368720591, 0.0476099178, -0.0547937602, -0.126454487, -0.10340786, -0.131127492, -0.0437266976, 0.0529951043, 0.0883525163, 0.0980372503, -0.0825529173, 0.102423966, 0.163403392, 0.0976418331, 0.0313921869, 0.0288433321, -0.0276666954, -0.0106668435, -0.00334626157, -0.0132831838, 0.0184611958, -0.0464694872, 0.0805625767, 0.0173439197, 0.0262606516, 0.126519099, 0.138395324, -0.00254166313, 0.119938344, 0.0573389977, 0.0542154163, 0.0692043006, 0.0597935244, -0.0188125204, 0.049818065, 0.0757564455, -0.0483031236, -0.193337351, -0.00217950717, -0.0817932785, -0.106830128, -0.0650802255, -0.0446323194, 0.0341032632, 0.080365479, -0.0988180935, -0.0450610071, -0.0722491369, 0.0166641083, 0.127055496, -0.103618376, 0.0380277, -0.0759299994, -0.0933069065, 0.0111208772, 0.155003533, -0.0709212944, -0.0932924896, 0.0226059556, 0.0122168204, -0.114529938, -0.103299066, 0.0415850468, 0.00406396575, 0.0625993013, 0.00801790785, 0.0511501096, -0.0501103476, 0.1241448, -0.0662367791, -0.00844532624, 0.177476555, 0.0625147074, -0.0147227608, -0.0120679624, 0.0353377983, -0.046898514, 0.0142605919, 0.056622006, 0.172268614, -0.0329496637, -0.231005609, 0.0563728623, 0.080097951, -0.00894291885, -0.151174337, 0.0251428112, -0.0579357818, -0.0256807655, 0.0514307618, 0.0262518115, 0.0426398553, -0.001229716, -0.0286666676, -0.0170986764, -0.125903815, -0.0690000802, 0.0786091909, 0.0171093177, -0.00777454674, -0.00667924713, -0.0768917128, 0.0167301055, -0.0605392531, -0.00799709186, 0.0590173975, 0.039383892, -0.0531835444, -0.0277832299, 0.0562856458, 0.0160953552, -0.103994332, 0.0460520945, 0.190410435, 0.122205824, 0.0989888832, 0.119691916, 0.142407835, -0.022124365, -0.00849366561, 0.0506508723, 0.0850793868, 0.0271743592, -0.0376036167, 0.0482522696, 0.102856554, -0.0496400036, 0.0277350806, 0.103806086, 0.0148996105, -0.0158420596, -0.0316775106, -0.0387260206, -0.0233267397, 0.0821134523, 0.0401642285, 0.0917946175, 0.0671747178, 0.0684598088, -0.000702465884, -0.0451893173, 0.0517121479, 0.00471234322, 0.0793196112, 0.00699635781, -0.131860629, -0.0368878245, 0.104009926, -0.0268972032, -0.0428332537, 0.113431826, 0.0198208876, -0.0664840862, -0.0546237454, -0.019905258, -0.00254343264, -0.036215134, -0.0554769486, -0.0181054473, 0.140997991, 0.0111484537, 0.0367606059, -0.0674065724, 0.0212049112, -0.0561227873, 0.0290108286, -0.00833883137, 0.00222712872, -0.0847283453, 0.0431756042, -0.109141119, -0.0129319951, 0.0333293751, 0.00531570101, 0.097147122, 0.0388240851, -0.0354440808, -0.0885681733, -0.213006049, 0.0727706179, 0.036135029, 0.102887303, -0.0465593152, 0.0640048981, -0.111603916, 0.094097659, -0.0586705655, -0.075268656, 0.052961275, -0.135893717, -0.0614549555, -0.0569578558, 0.0523011349, 0.0330762491, 0.0435143337, 0.0344756283, 0.0671566129, 0.10543716, 0.0944586769, 0.0153974276, -0.050820291, -0.0458775647, -0.0345414616, 0.0962239429, -0.096707724, -0.0452955365, -0.0182661228, -0.0212264918, 0.069447279, -0.0450920016, 0.100490421, 0.0278961621, 0.0882038102, -0.0678256229, 0.0138143562, -0.0689106062, -0.00360275386, 0.0663605928, -0.0607298799, -0.0621103942, -0.0543092974, 0.0128324572, -0.0431163646, 0.0219562948, 0.00678311661, -0.0441136137, 0.0982432887, -0.0705860108, 0.182194039, -0.108619966, 0.0207179412, -0.122581631, -0.0929343551, 0.0586816929, -0.0232572667, 0.00806567539, 0.0225188695, -0.0365971811, 0.102062739, -0.055163864, 0.0595620796, 0.193907857, -0.0719701275, -0.0325663052, 0.0913035646, -0.0724671558, -0.0490570292, 0.0606238581, -0.00221333839, -0.0208245013, -0.18978031, -0.0184468329, 0.0584079362, 0.0619091392, 0.0283486024, 0.00343166548, -0.0329216793, 0.102478705, 0.0746710822, 0.042023275, -0.00857234187, 0.02867046, -0.037411008, -0.00556871109, -0.0417560525, -0.123214625, -0.00407732744, 0.0280542225, -0.115010217, 0.0420889705, -0.0983415693, 0.033393234, 0.0291160401, 0.0999559239, -0.037810795, 0.0574650541, 0.0249308553, -0.0111770369, 0.0586905405, -0.0181362778, 0.129456714, -0.028140679, -0.0116888974, 0.0460940041, -0.183939517, -0.107369378, 0.0142709417, 0.0799058527, -0.0281989574, 0.00468265638, -0.00359648839, -0.00181956217, -0.00247250684, 0.0800077394, -0.0349083468, -0.0869949088, 0.030391261, 0.0290568061, 0.0480341166, 0.0350300148, -0.218458921, -0.0633597374, -0.00389631395, 0.0858308673, -0.165539861, -0.0115812551, 0.110183015, 0.0742593631, -0.0190524422, -0.0575886704, -0.0105343126, -0.0458830781, -0.0268041249, -0.0500699021, -0.0974797457, 0.142067999, 0.00756507739, -0.0139123565, -0.219773516, -0.192728773, 0.0831120834, 0.0301636811, 0.0989038795, -0.0733708888, -0.00122421142, -0.0823754147, 0.134696111, 0.064505741, 0.099184759, 0.0629062727, 0.215615958, -0.0425261408, -0.0731833428, 0.0291134324, 0.0813642889, 0.0460265577, -0.0210361108, 0.0383235291, -0.090638876, 0.00868848525, 0.0973384976, 0.0863050148, -0.126141474, -0.0671756789, 0.0142485201, -0.00345332734, 0.085107848, -0.0468325168, -0.0311242789, 0.0531625003, 0.0203431584, 0.0540217683, 0.0213960689, -0.0126134809, 0.0620418936, 0.0049791839, 0.094513759, -0.00577996671, 0.142208964, 0.0486403853, 0.00964468438, 0.0353494138, -0.0813095719, -0.0396264419, -0.0299608354, -0.0700816289, -0.0436064377, 0.0170924012, 0.0520251021, -0.0128122233, -0.0186763313, -0.0422864184, 0.0751069486, 0.0735050514, 0.0184059013, -0.14228113, -0.0401629582, -0.0588053875, 0.110950388, 0.113210753, 0.0271767527, -0.0060010571, -0.0826001614, -0.0834111571, 0.017040506, 0.0191633068, 0.0121653015, -0.0290833972, 0.0624605678, -0.0357175432, -0.0785514563, -0.0902193189, -0.0996724367, 0.0230609588, 0.0412896797, 0.0997388065, -0.0565732531, -0.00927331299, 0.138090402, 0.0513459668, 0.142254293, 0.128031746, -0.0142473355, -0.00695161195, -0.0359653533, 0.102160811, 0.0172250327, -0.0224740561, -0.0615768358, 0.0354183391, -0.141508907, 0.00267085433, 0.0222913697, -0.133883581, 0.0196404234, -0.0762126669, -0.0453807004, -0.0193437468, 0.0606390536, 0.140449613, -0.0485979468, -0.0578757189, 0.130762786, 0.0309764072, 0.0085640084, -0.0317615718, 0.0492270291, -0.04021018, 0.0889722332, -0.0266411975, 0.0901532173, 0.132348806, 0.0413502529, 0.0548291393, 0.0590111315, -0.0898910612, 0.0582996011, 0.065266408, -0.0744625032, -0.0377952904, -0.0368359089, 0.0469830334, -0.116807431, -0.115320541, -0.0879266933, 0.00238024257, 0.0103788227, -0.069691278, 0.00391908037, 0.024099797, 0.0738078877, 0.0303493738, 0.0550419018, -0.121972822, 0.0200210288, -0.0166991334, -0.0649560243, 0.0218866523, 0.0012789527, -0.071845673, 0.120481841, -0.219442159, -0.0388041958, -0.0489232615, 0.0408151038, 0.0525902323, -0.0625492558, -0.0334295034, -0.179259941, 0.0485134721, -0.00684842002, -0.172918841, 0.0152828321, -0.00353746861, 0.0797556043, 0.171828106, -0.0856639072, 0.0483391657, 0.106606655, -0.0346524417, -0.0662102997, 0.000548389042, -0.0723318458, -0.0226519592, -0.0298163742, -0.00970225781, -0.00914438255, 0.0463590994, -0.0031957943, 0.0499412045, -0.0235150084, -0.0300997011, 0.0376598649, 0.198073745, 0.0993624479, -0.0572848916, -0.109548002, 0.0868605822, -0.0564789772, -0.113025799, 0.0835291892, -0.0292221382, 0.0901703537, 0.108187534, -0.0882775038, 0.0816135556, 0.0239357501, 0.0677815974, 0.00296494737, 0.0748788863, -0.0120913768, 0.0256078783, 0.0664716363, 0.0385060161, 0.0163188521, -0.0646069273, -0.0842390433, -0.0362252221, 0.0761245117, 0.0370759107, 0.162758842, -0.119829409, -0.015496552, -0.0286020041, 0.127342939, -0.00396361947, 0.0463322103, 0.0827808231, -0.0372733176, -0.0234975945, -0.0555949658, -0.05986543, -0.0525532961, 0.0899257213, -0.0632371083, 0.00453333929, 0.139113203, 0.0346173048, -0.00875579193, 0.0369689353, 0.116822541, 0.000411467627, -0.0311805699, -0.0324053466, 0.042315729, 0.0325569808, 0.0705077425, -0.158490002, -0.0692853034, 0.014626611, 0.127531514, 0.085432902, -0.0120464228, 0.0703074709, 0.0510105826, 0.0701586604, -0.0554094948, 0.0482138582, 0.124873832, 0.0997996107, 0.00841645058, -0.0322865173, 0.00332034309, -0.0512876958, 0.00796328858, -0.0496845655, -0.0817840248, -0.0284804404, 0.207782403, -0.00811658893, 0.0207694601, -0.0552041009, -0.00310244411, 0.0468787253, -0.133973569, -0.155573621, -0.118333511, 0.0644147024, 0.0424428135, -0.0530001745, 0.0445820577, 0.0557935536, 0.0129037797, -0.0369238518, 0.127312809, -0.0277343579, -0.0698076189, 0.15275225, 0.0398202725, -0.0484452844, -0.0406120904, -0.0565820746, 0.00224541454, 0.0964962691, 0.00645267218, -0.0306327064, -0.118842952, 0.0958830044, 0.0555735417, -0.0384260118, -0.00305845402, -0.0558330007, 0.0854666829, -0.0205603279, -0.035670273, 0.0723932087, 0.0588418469, 0.0438152626, 0.0188954454, 0.101422183, 0.0711393803, 0.111880019, -0.0488751605, 0.013999437, -0.048159752, -0.0452164672, -0.0451781154, -0.00924299285, -0.158946276, 0.0276355017, -0.019252412, 0.050336957, 0.0381732211, 0.0468685105, -0.100663327, 0.0153418193, -0.0391150564, -0.057868544, 0.107873701, -0.00606214022, 0.0402068198, 0.112427071, 0.055900462, -0.00954103004, -0.0631262213, -0.0752608627, -0.121419631, 0.0537686422, 0.0702112317, -0.0317528136, 0.0155923311, 0.0643391088, 0.0823150501, 0.011424928, 0.0866788924, -0.0557377785, 0.0242005736, 0.0581678934, 0.0170797296, 0.0112792905, -0.029697597, 0.0732057691, -0.153560072, 0.0463197939, 0.00305291638, 0.187867433, 0.0859213769, -0.0525866076, 0.0788777024, 0.0505607501, -0.0339050591, 0.00377000868, -0.0081246607, -0.0502759106, -0.0199783258, -0.0896850973, 0.0376046449, -0.159608096, -0.0208158493, -0.0547869429, 0.140949667, 0.00822881982, 0.0426262915, -0.00746865384, -0.0208673328, -0.0236783735, 0.0556462817, 0.0360817984, 0.00203144737, 0.0328801721, 0.0383945853, 0.0120557062, 0.00986700132, 0.138688341, -0.0186713263, 0.0991785973, -0.0621830449, 0.102392785, 0.196683288, -0.113352746, 0.0307539217, 0.160915852, -0.00642421097, -0.0744954497, 0.0174026955, 0.0922159851, -0.00581721589, -0.104899362, 0.0780781731, -0.0671591014, -0.00771567598, 0.0277557056, -0.0648308918, 0.128763229, 0.0467619039, 0.035747759, -0.0413503721, 0.15562813, -0.0232945103, 0.125851959, -0.230834201, 0.0893382207, -0.0495846346, -0.0385772809, -0.0353227928, 0.0507783592, -0.035266526, -0.047131449, -0.0176881682, 0.0360539183, -0.0857599825, 0.0258405209, 0.0694242418, -0.00353942811, -0.0398704633, -0.0827132091, 0.0523384586, -0.117656805, 0.0172490813, -0.0411410183, -0.0999691635, -0.0979274511, -0.114667013, 0.0348461792, -0.0144496374, 0.058701843, 0.0706167221, -0.0642464906, 0.119065277, 0.131035864, -0.0304263122, -0.0137733072, -0.0363757685, 0.0266923793, -0.0455352701, 0.0286264122, 0.00583955739, 0.00585118961, 0.175062031, 0.00927729532, -0.0204659514, -0.0332344584, -0.0079884883, -0.0494965687, 0.0365244783, 0.0589441247, -0.0634012818, 0.0168215558, 0.00974214636, 0.0313278846, -0.0947920382, -0.0776266083, 0.0622960627, 0.0688989311, -0.0952006131, -0.0346632153, -0.0338409357, 0.0726115108, 0.197687849, 0.007835133, 0.00582121126, -0.00569648948, -0.00252835872, -0.0110833589, 0.0878808126, -0.00196283776, 0.165228099, 0.0459995419, -0.00982443895, -0.0796034783, 0.00905897189, -0.153510392, 0.108211473, 0.158081084, -0.0377744958, 0.0505883135, -0.0575247556, -0.075220719, 0.0338324197, -0.130541414, -0.0906890631, 0.0591744483, 0.0738413781, -0.149436235, -0.0250280201, -0.0346436054, -0.0141798705, -0.108943425, 0.00232343376, 0.00533589954, -0.127761394, -0.032311108, -0.0971097201, 0.0150812231, -0.0370598696, -0.00486735255, -0.0548874661, -0.0815641657, -0.0441496521, -0.130818218, -0.0627015531, 0.0333955213, -0.0187171474, 0.0680370629, 0.0568083078, 0.0401994251, 0.0638009235, 0.00617516972, -0.0177865513, 0.0456849448, 0.0413590893, -0.0400048085, -0.00927871279, 0.122263268, -0.0846701115, 0.0735645965, -0.0731005818, 0.0534018949, -0.0490769558, 0.07646323, -0.0171432532, 0.111487597, -0.0126327146, -0.0667313784, 0.0441563725, 0.0396787003, -0.0108370492, 0.0236835256, -0.0392706022, -0.102848731, -0.0621793605, -0.0423569158, -0.0354129225, 0.0208173264, 0.0364403203, -0.142889783, 0.0237936713, -0.0149820875, -0.145569399, -0.0394799598, 0.0969427079, -0.054175701, -0.134356916, 0.0276410729, 0.0506090187, 0.0710193217, 0.0870926604, -0.0606542602, -0.0026505813, -0.160247087, 0.0402680226, 0.0271979403, -0.0864291713, 0.0413569026, -0.0622934103, -0.0218009725, 0.089244321, 0.0332072489, 0.0657498166, -0.00505386665, -0.0492895395, -0.0890076309, 0.0782933906, 0.0204010755, -0.0450760461, -0.0718519688, 0.0547425337, 0.0627222061, 0.0665706843, 0.0384123474, -0.00860513374, 0.012388546, -0.0839210823, -0.0487274155, -0.0539148673, 0.0449279994, 0.078998886, -0.0950290188, -0.050470002, -0.0429880768, -0.0437469818, -0.048291862, 0.10736306, -0.0979295671, -0.0811112747, -0.0530942306, -0.153853074, -0.16854775, -0.0392187871, 0.0121662412, 0.00176871335, 0.0253451467, -0.0658509582, -0.0616914257, 0.0228686966, -0.10971415, 0.135989681, -0.0335242748, -0.000956429169, 0.0553396866, 0.126581058, 0.0474915504, 0.0211014152, -0.0707104206, 0.119461305, -0.0858744234, -0.0533777773, -0.206835583, 0.0496135354, -0.0852625817, 0.0548041314, 0.108932175, -0.0661319047, 0.00594475213, -0.0798635483, -0.00666934438, -0.00316115795, -0.0238929577, 0.0638570264, -0.0389510468, 0.0643313378, -0.0307526607, 0.0883754566, -0.0476251803, 0.00247806869, 0.0990912765, 0.0571272932, -0.0656959936, -0.0876581669, 0.0539998636, 0.0428763889, -0.0565429293, 0.0822702497, -0.0976557434, 0.0224922448, -0.137141794, 0.0516681969, -0.173518211, 0.00714187324, -0.0489615425, -0.0682698637, 0.0697755441, -0.0377197936, -0.0324800834, 0.0682256967, -0.0459169932, 0.16174911, -0.00530527253, 0.0351424366, -0.0741646439, 0.0660107434, -0.0197895616, -0.141294301, -0.07206662, 0.0847613141, -0.0939313322, 0.0219362117, -0.153947011, -0.0551418439, 0.154210478, 0.04822056, 0.0734988078, -0.0403701477, -0.138773963, 0.0329378285, -0.00727817742, 0.0566106662, -0.0855385438, -0.0894598365, -0.0608090162, 0.012729533, 0.0434634276, 0.0687907189, 0.148822874, -0.0516477674, -0.0554004386, -0.0936880261, -0.0658270121, 0.0839076266, 0.0431993119, -0.00819264818, 0.0264952667, -0.016709324, -0.00969122909, 0.138044655, -0.0653872341, -0.0255857483, -0.0257683992, 0.0354169458, -0.169573903, 0.0797453597, 0.0307036862, -0.0552977026, -0.136601239, -0.0300603788, 0.050477773, 0.070897989, -0.00995214283, -0.0248042196, -0.066885978, 0.0727180913, 0.0737626031, 0.0173303485, -0.025581304, 0.0635150671, -0.0901748165, -0.0042982474, -0.0772284865, -0.0734660327, -0.0484250672, -0.0562392324, -0.0777136534, -0.142158046, 0.118982479, -0.122404516, 0.0402211547, -0.0368508734, 0.029629685, 0.0634636134, -0.0273319464, 0.0272786859, 0.0352585874, -0.0379413068, -0.0257819872, -0.0336226448, -0.0354589596, -0.0424527749, 0.102676675, -0.0579748675, -0.0432516821, -0.0110586304, 0.123912379, -0.0254480392, 0.0900846422, -0.0209755339, -0.0430043302, -0.0256560706, -0.0365977176, 0.0179417226, 0.050363481, 0.127457201, 0.0994190574, 0.0845612884, -0.0200168267, -0.104750745, 0.239868566, 0.0186115988, 0.178199813, 0.0310933404, 0.062885955, -0.0562206246, -0.0392183103, -0.0526602902, -0.0727086812, -0.0366779007, -0.122839846, -0.0177269597, -0.020671878, -0.0447096899, 0.112125948, 0.0552616157, -0.0793292597, 0.11010053, 0.0566014536, 0.0105314925, 0.0649300516, 0.0124685336, -0.065028511, -0.0814464539, -0.0535159707, 0.075172931, 0.0512848869, 0.124607354, -0.0304890964, -0.0202325247, -0.0133397505, 0.00607856037, 0.0542979315, 0.0357338227, 0.0694069266, -0.0883907303, -0.0505184866, -0.0274258684, -0.0451109298, 0.0880140737, 0.0571361668, 0.0118459854, 0.0533859767, 0.101867095, 0.00520355441, 0.12812005, 0.200060204, 0.120280221, -0.0197006054, -0.0587520935, 0.0717615932, 0.166860014, -0.0882551745, -0.0660146177, -0.0328773782, -0.137794584, -0.0938184783, -0.00144285941, -0.118490122, 0.023691915, 0.0282468814, -0.0695485622, -0.0863662213, -0.104297206, 0.0190177113, -0.00720984489, 0.0746551752, -0.054489132, 0.16164881, 0.127069384, 0.0143358847, 0.0857696831, 0.0835655481, -0.0396123752, -0.116242573, -0.0264006965, -0.0861118883, -0.0320002288, -0.0515784696, 0.0245875269, -4.10219654e-05, -0.0561805964, 0.0511259586, 0.0491109192, -0.0950999707, 0.0726895705, -0.108802855, 0.018060118, -0.133699417, -0.00267339405, 0.0589299276, 0.0167818218, 0.0702794045, 0.000833958387, 0.0499559194, 0.0545615032, 0.162329838, -0.0680439919, -0.0699060559, -0.15240258, -0.0243935026, -0.00303140096, 0.00623072311, -0.020528052, 0.00236353464, 0.0902205631, -0.0367763489, 0.0199145116, 0.0212102402, -0.0352000743, -0.00631831959, 0.0320474952, 0.0281665921, 0.0808550641, 0.0251082182, 0.0282254033, 0.0036831554, -0.0160769746, 0.0233788732, 0.0261787195, 0.0226513185, -0.0150998672, 0.0153304236, 0.0188213531, 0.0503936633, -0.045406118, 0.0820774511, 0.0189963859, -0.0735352412, 0.0783244967, 0.0159697533, 0.123810753, 0.0472124331, 0.0501417145, 0.0643201843, -0.0742305368, -0.0364033878, -0.054758314, 0.0295691304, -0.00533509441, -0.0248704236, 0.0944912434, 0.0813809186, 0.0800662935, 0.0420621634, -0.104065731, -0.00707397517, 0.0386740789, 0.168509588, -0.0944282636, 0.0742100775, 0.121663205, 0.0613658726, 0.0363074765, 0.138406873, -0.078356795, 0.0452519581, -0.0600139759, 0.150149718, 0.023582831, 0.0457559377, -0.0855897516, 0.0482263267, 0.00215817336, 0.00113095716, 0.0506576933, 0.0123284925, 0.0568627268, 0.00802153349, 0.133727148, 0.0333910063, -0.023536358, 0.141339049, 0.0279657394, -0.105808012, -0.00864004344, -0.012913486, 0.0723010227, -0.0580282882, -0.0980359167, -0.121762902, 0.0335033461, 0.0492193848, -0.00799391884, 0.0229605138, -0.0465496927, 0.0366377011, -0.0190207548, -0.0344992056, -0.0638491586, 0.19049722, -0.0673196018, 0.163322881, 0.0370728299, 0.0201039165, -0.117321387, -0.0258302167, -0.021659717, -0.0786858648, -0.042272266, 0.082426101, 0.0618773587, -0.00105269952, 0.0102046933, -0.0235174112, -0.0510242581, -0.116305858, 0.0226745121, 0.0556324944, 0.120265208, 0.0731783137, 0.0661707222, -0.0280066542, -0.0199447945, 0.0128385788, 0.0226939432, 0.0104000568, 0.00935876649, -0.213882118, 0.043200016, 0.0241836477, -0.13518852, 0.140135095, 0.0253206324, -0.089445211, 0.00240788609, -0.0890551805, -0.0191624686, 0.0517471433, -0.0367655568, 0.0598453246, 0.112564206, -0.116867706, -0.0396824777, -0.0163099933, -0.118076362, 0.11046911, 0.0247966498, 0.0313623138, -0.108059898, 0.0364985466, -0.0730506554, -0.0836252645, 0.0544317178, 0.0144574177, 0.0365974307, -0.0178850703, -0.055263631, 0.130582184, 0.0158302486, 0.0212825127, 0.0239027031, -0.0166860893, -0.0275060162, 0.0294779949, 0.0809956118, 0.0361995175, 0.0210323408, -0.0460734852, -0.0791156143, 0.0205498245, -0.0106738573, -0.00989503041, 0.0165876858, -0.0203668587, 0.0815822035, -0.0239934083, 0.0604061931, -0.00175664946, 0.0208463781, 0.0540469699, 0.174571007, -0.0146036129, 0.0423222333, 0.0977733657, -0.0425417535, -0.0710100755, 0.0760513246, 0.113821641, -0.0535171703, -0.00542533398, -0.0697968975, -0.0428297296, 0.0674038902, -0.0297512412, -0.066744484, 0.0181291327, -0.00508406153, -0.0266535934, -0.0606855378, -0.0260272212, -0.029811386, -0.107172653, -0.150785118, -0.0542859547, 0.0356353149, -0.122487269, 0.0750695467, -0.0401163846, -0.0629263371, -0.0792647377, 0.104086034, -0.0047227107, 0.103974536, 0.0502419882, 0.0476147234, 0.052882392, 0.081533879, 0.0924756974, -0.0315656103, -0.0200783983, 0.130904391, -0.0245863274, 0.0448258296, -0.0867705271, -0.0143366829, -0.0240080208, 0.0499560311, -0.00190844573, 0.0032625813, -0.000506900251, -0.0229720958, 0.0386845991, -0.0575748906, 0.00777366385, 0.0670741051, 0.065418154, 0.149928927, 0.0400025733, 0.124139905, 0.0728096142, 0.00236796588, -0.120325178, 0.16046533, -0.0657965019, -0.0568519235, -0.00610711426, 0.0497483648, -0.00804714486, 0.0444892272, 0.0504619479, -0.133039102, 0.00865272805, 0.0114317089, -0.00698417053, 0.0169084482, -0.0348446779, -0.0723827779, 0.0108677205, -0.00218051486, 0.0390979648];
    bias_0_u : ARRAY[0..63] OF REAL := [-0.931392431, -0.669652343, -1.55073643, -1.15129042, -0.928060949, -0.835326016, -1.05773425, -0.809125721, -1.0343436, -1.36020243, -0.812485695, -0.596730828, -0.800589681, -0.83492893, -1.23361444, -1.4201777, -1.06900442, -1.04275012, -1.86629462, -1.68873703, -1.34019673, -0.945544183, -0.886029959, -0.729185879, -0.675665855, -0.875132143, -0.690106928, -0.763296306, -0.747061849, -1.10096192, -0.758312643, -1.23618972, -1.4139967, -1.28251481, -0.887215853, -1.12884796, -1.17651927, -1.66531849, -1.57700455, -1.01120985, -0.878331959, -0.872978032, -0.621329427, -1.0162462, -0.99940753, -0.698668599, -1.47800922, -0.852591813, -0.93049854, -0.788715541, -0.874885857, -0.572944462, -1.31330848, -0.807830811, -0.895757496, -1.79783428, -0.845625222, -1.08024359, -1.43994868, -1.82642233, -1.50900924, -0.701206744, -1.07954109, -1.05142236];
    weights_0_r : ARRAY[0..63] OF REAL := [-0.301351488, 0.191772759, -0.403094679, -0.385009229, -0.325696975, -0.344430864, -0.430924505, -0.490683407, -0.380927861, -0.361935526, -0.291825026, 0.270645022, -0.557896674, -0.624442339, -0.570287347, -0.547084689, -0.328458816, -0.604146957, -0.345501393, -0.616985977, -0.625005603, -0.563085496, -0.468810678, -0.398420662, -0.227860957, -0.486180753, 0.0191694256, -0.046916645, 0.234420627, -0.389543176, -0.00718040438, -0.374701381, -0.612858176, -0.358533949, -0.574734867, -0.603802323, -0.283780545, -0.357478797, -0.447851956, -0.458725035, -0.410655737, -0.376305223, 0.303187847, -0.553753257, -0.386509717, -0.504178882, -0.474493176, -0.238366574, -0.448695511, -0.551571906, -0.411650151, 0.404194504, -0.465952367, -0.147349313, -0.468469918, -0.304423511, -0.4342767, -0.47622183, -0.525499105, -0.457058758, -0.439959496, 0.0408562459, -0.552530468, -0.292028844];
    recurrent_0_r : ARRAY[0..4095] OF REAL := [-0.0834894925, 0.0467989594, -0.0922519863, 0.0892271101, -0.0968513042, 0.0679784194, -0.0419990122, -0.0955153108, -0.0172851142, -0.0447769873, 0.0400388502, -0.0478489809, 0.0498131029, 0.0975087509, 0.103417948, -0.0618524924, 0.138862789, -0.0484442562, -0.106181331, -0.132875144, 0.0242299326, 0.0707813576, -0.0631774291, 0.0927816704, 0.146799028, -0.0673606545, 0.0149163306, 0.158295408, -0.0541859716, -0.0671267807, -0.00778596848, 0.000831183046, 0.0179751236, 0.0616365261, 0.0552535653, -0.11939618, 0.00227971375, 0.0860660523, 0.0384575725, 0.0739784613, 0.00518694334, -0.0637862906, -0.00229425658, -0.0886000842, 0.119190097, -0.0505612381, -0.100778803, -0.11373806, -0.046051234, 0.0172212869, 0.00996381789, 0.0867178142, 0.00406045653, 0.0659313872, 0.0901537985, 0.00407537259, -0.155829459, -0.0182549451, -0.0341455899, 0.124589838, -0.0760684684, 0.0296373926, 0.00549710728, 0.0332801342, 0.0679366067, -0.0555260926, 0.0819408521, -0.0728703663, 0.020875264, -0.0447206348, -0.024039913, 0.0543668233, 0.0924990252, -0.0224341024, 0.0680758804, -0.0131752398, 0.0171246715, -0.0379354954, -0.118314825, -0.0296662319, 0.0103624333, -0.150564685, 0.0755786151, -0.0666730851, -0.0181739815, -0.0342114717, 0.0339080915, -0.0595367178, 0.0309331622, -0.0153474286, 0.0614931062, -0.0788206384, -0.0491645597, -0.0551766492, 0.110275842, -0.0309414417, -0.087802209, -0.0610899068, -0.00560984015, 0.0977157503, 0.00970546156, -0.156553969, -0.0635337755, 0.00846432708, -0.0481569208, -0.156108454, -0.0311011374, 0.0380924568, 0.0604931377, -0.106866658, 0.0386045091, 0.0167547446, -0.0975543559, -0.0810313448, -0.00664621964, -0.0154656004, 0.0141974762, -0.0400947481, 0.0326277912, -0.0616046824, -0.0670897216, 0.163002104, 0.01041748, 0.0679064617, -0.0368735157, -0.0427763127, -0.0614703819, -0.0516258851, -0.0362892523, -0.0502930507, -0.0644264519, 0.040134564, 0.163039222, 0.0453167073, 0.0265058093, 0.0309302956, -0.0310254358, -0.0870743915, 0.0869462565, -0.0102094412, 0.02950841, -0.0191445109, 0.0157393347, 0.112097934, 0.142738387, -0.0986512154, 0.101732939, 0.0275557972, -0.0516387671, -0.024218658, -0.00215544179, 0.0165637061, 0.0156634506, 0.0115557984, -0.0915465057, -0.0172377117, 0.0396726206, -0.0412831642, 0.0991871059, -0.0850381553, 0.122572176, 0.059342213, -0.0229966789, -0.0314630009, 0.00477001816, -0.0216304138, -0.0459695496, -0.0558857583, 0.0364166088, 0.0599161908, -0.0168819502, 0.155651927, 0.141873583, 0.126577303, 0.0584061071, -0.0245434716, 0.07191585, -0.125751734, -0.096313253, 0.0990332961, 0.0953751877, 0.0237817224, 0.0773518533, -0.0857243687, 0.138499305, 0.0413452238, -0.00136547722, 0.0418496765, -0.00384547003, 0.0725840926, 0.0687962323, -0.221241683, -0.0535463355, -0.0130795371, -0.152106091, 0.00108890608, -0.0629126653, -0.109754905, 0.0672944188, 0.0458643995, -0.127328977, 0.0779956579, -0.0260329992, -0.0222704634, 0.0060250815, 0.0342492759, 0.0469465703, 0.0682547241, 0.0466573387, -0.0317380279, 0.118174516, 0.0363855176, 0.0165183749, 0.216430724, 0.0503736399, -0.0601224527, 0.047193028, 0.131177261, -0.0908262208, -0.15726164, 0.0594424009, -0.0204188749, -0.0278644171, 0.101016611, -0.0298268441, -0.080154486, -0.0577925071, -0.106108546, 0.00219925866, 0.0538200289, -0.000312333927, -0.0564782694, 0.0101036718, 0.00516057666, 0.00766485184, 0.0177538376, 0.00237444974, -0.0577772781, -0.127201959, 0.0181556642, -0.00818925537, -0.0185058136, -0.0378008261, -0.0132604018, 0.0929510295, 0.0808474272, -0.0706657469, -0.113311686, -0.0553113446, 0.0279085524, -0.105972864, -0.0372796655, -0.0130742528, 0.0488647111, 0.0226176027, 0.0247713439, 0.0545698255, -0.0249881856, -0.0808280632, 0.0343040675, 0.0220307633, 0.0778453946, 0.00909530744, 0.00474842079, 0.0245809406, 0.027137503, -0.0232185125, 0.140213117, 0.0256274082, 0.0719716772, -0.0154388361, -0.0446083136, 0.0152545236, -0.0324217938, 0.0500168242, -0.114832193, 0.0540725663, -0.201761976, 0.0459797718, 0.0488682203, -0.0374526232, -0.0756408647, 0.0282250922, 0.0548831299, -0.151702717, 0.0439265333, 0.0316746458, 0.0101707652, 0.0837145448, 0.0808735639, 0.0973392278, -0.0686043128, -0.0390135162, -0.037535198, -0.0250067096, -0.0664628521, 0.0204570256, 0.0354304649, -0.057973817, 0.0578858256, 0.0356692336, 0.0886768922, 0.0543263741, 0.0420739315, 0.084652096, 0.180876732, -0.0387669355, 0.0118383123, 0.0290507115, -0.0599402376, 0.0485393032, -0.0703626052, -0.0345942751, -0.0286344141, 0.0617277063, -0.0411391258, -0.0778558925, -0.0121396091, 0.0011215657, 0.0436940789, 0.000647306093, 0.0169583671, 0.0537803844, 0.0782520995, -0.0194653235, -0.0218962058, 0.00249565719, -0.010981407, -0.0674014688, -0.0330897793, 0.018824378, 0.157535002, 0.0308090374, -0.0746396407, -0.0875643045, -0.00356309139, 0.00969221443, 0.0921113268, -0.0434736833, 0.0130275963, -0.0466789939, -0.0251713507, 0.10718137, 0.155800402, 0.0190462153, -0.0899385735, 0.137247831, -0.0866682157, -0.0320754685, -0.0946900174, -0.0161404721, 0.0882564411, -0.112924516, -0.088722147, 0.192345887, -0.0126325535, -0.0174161885, -0.0645587966, 0.0146739678, -0.0393769257, 0.0789906681, -0.0809244365, 0.0494276024, 0.0675513595, 0.0875197873, 0.168436021, 0.0236752108, -0.0369569995, 0.0797938108, -0.119467117, -0.0492167324, 0.0533705875, -0.000214729458, 0.0990879759, 0.0621759742, 0.0427966863, 0.0239031687, 0.0799559504, -0.0621714219, 0.0745402873, 0.0781922266, 0.0327110179, 0.0261501111, 0.011958912, 0.106199577, -0.0313672908, 0.0454588458, 0.0187561624, -0.0123822438, 0.0570373051, -0.0774810463, -0.0445477366, 0.195391595, -0.0160081312, -0.0467466153, -0.15215385, 0.0304640979, 0.0530834794, 0.0519628152, -0.142502248, 0.0521924794, -0.0213847924, 0.137605369, -0.0943483561, -0.0639615729, 0.0294855349, -0.000336129218, -0.104782604, 0.0927328095, -0.028684549, 0.132814825, -0.0141541846, 0.0926760733, 0.0494773462, -0.0836238563, 0.0119094858, 0.0856154338, -0.139292598, 0.0450100079, 0.0095192045, 0.0648575351, 0.0879206955, -0.0362641513, 0.0149863679, -0.093047604, 0.0910623372, -0.0729507431, 0.099900797, 0.00975495018, 0.10402672, -0.0265085027, 0.00896766782, -0.0797617286, 0.0680103824, -0.00225491449, -0.111769781, -0.0673333183, -0.107364029, 0.0766148716, 0.0842316598, 0.0189867634, -0.139816821, -0.0133126192, -0.125086024, 0.0900506675, 0.107696734, 0.0128689855, -0.0446564034, 0.0704938099, -0.0910163745, 0.120799132, -0.0846302807, -0.0124115273, 0.010663012, 0.0126034543, -0.0300969128, 0.0170655474, 0.0514482073, 0.0689900517, -0.00158789381, 0.149908528, -0.0603792854, 0.0131468186, -0.0535668321, -0.118181631, -0.025183931, -0.109207809, 0.00673588412, -0.124501571, 0.0124984011, 0.0683000535, -0.0511983112, -0.0355482064, 0.0124112274, -0.105003238, -0.0914214924, -0.037354432, -0.0406142324, 0.0181756504, -0.0504919142, -0.0960488319, -0.0375996903, 0.0391708873, -0.0349344909, 0.0847899988, -0.0085113775, -0.0851751342, -0.0951333269, 0.0153997168, -0.0674072206, 0.0236242227, 0.0501294322, -0.0528307669, 0.131298378, 0.0220658295, -0.0347023904, 0.029442694, 0.0483123884, -0.16232118, 0.0271872394, 0.0621333644, -0.0257400814, 0.0729334578, -0.0658665001, -0.105266467, -0.171774209, -0.0453840047, -0.0155880339, 0.0938720107, 0.0879871398, 0.0643682331, 0.0427748635, -0.0361816436, -0.0438858196, 0.0104101989, -0.134780109, 0.0869414657, 0.00118048675, -0.00513844192, 0.0182014499, -0.0240692645, -0.0398045331, -0.0146628786, 0.0358414315, -0.0180199072, -0.0287214592, 0.0866206288, -0.0701739937, 0.000415597111, 0.0721387342, -0.0679822639, 0.171161994, 0.0371262208, -0.0477780961, 0.0761367232, 0.00384224392, 0.130283386, -0.0281605236, -0.0999097824, 0.00152361393, -0.0915167928, -0.0212306529, 0.0126610585, 0.0154684512, -0.0978761613, 0.0650571138, 0.107376486, 0.0881768167, 0.0337237157, 0.054977864, 0.0540641472, -0.134753376, -0.131919801, 0.0537733622, -0.0841272324, -0.0393206924, 0.0709122196, 0.102772944, 0.156615913, 0.0902129337, -0.0831259787, 0.0207677744, -0.0577425808, 0.0763535425, 0.0751461163, 0.0386200547, 0.0937433094, -0.0476259813, -0.0373367108, 0.0155079169, -0.0248294845, -0.120135389, -0.0352638401, 0.145516515, -0.100795284, -0.0410206988, -0.141030952, -0.0106899496, -0.0759382918, -0.0494840071, -0.0805307701, -0.0583564751, 0.0285217259, -0.0824788734, -0.000849559903, 0.0188932419, -0.0336842611, -0.0506386012, 0.0203082673, 0.0773929581, -0.0287808534, -0.06769678, -0.0738249421, 0.155622259, 0.0350486711, 0.0308453329, -0.0915696025, 0.0791843161, -0.0964923128, -0.00887560379, -0.0208047107, -0.133802965, 0.0323152542, -0.026939515, -0.0812889114, 0.0496312641, 0.0404926501, -0.1019504, -0.0131298713, 0.100097105, 0.115483843, -0.00638710242, 0.163589418, -0.0991462022, -0.0362230949, -0.0176009014, -0.0313397944, -0.0212460831, -0.0176329389, 0.0253308993, -0.0264203008, -0.0197697654, 0.0765542611, -0.0138612632, 0.0492661186, 0.00846538972, -0.0992811099, 0.120879501, 0.0574992225, 0.0359927192, -0.0615425259, -0.0063858442, 0.0557737239, 0.0424413607, 0.130089223, -0.0444395095, 0.107088849, -0.0397110581, -0.053124819, 0.011124542, -0.0532939099, 0.0410669371, 0.0292511564, -0.101436161, -0.0138421534, 0.261617333, 0.0745773017, -0.00261045154, -0.0530744269, 0.0931384563, -0.041711852, 0.0388382412, -0.0277338717, -0.137989819, 0.0612927973, 0.104822055, 0.0361424498, -0.081897676, 0.082424067, -0.0292748399, -0.0650308207, -0.0574782565, -0.0816696733, 0.115542442, 0.108364627, 0.150625765, 0.0555263087, 0.000987943262, 0.0676554143, -0.0174685903, -0.019615002, -0.095944263, -0.0548800603, -0.0220668316, 0.0540091395, 0.040932171, 0.0198501125, -0.0563352332, -0.0535954833, 0.0527449995, 0.157754645, 0.00486304238, -0.177564219, -0.0268895626, -0.0191486217, -0.0552683026, -0.0416013673, -0.147009224, 0.0570645519, 0.114052191, 0.0689847618, -0.00186852366, -0.0354810581, -0.0787176266, -0.0754320398, -0.0211988557, 0.00642943941, -0.0388428755, -0.0820757076, -0.0232652538, -0.0523139276, -0.192835316, -0.0925032943, 0.0320784673, 0.0165662523, -0.050621748, 0.048093807, -0.0466006622, -0.0441171862, -0.0852081925, 0.0172305536, -0.0356022976, 0.125120699, 0.00274382625, 0.0296839103, 0.0180109572, -0.00339450128, -0.200602382, -0.0330988802, 0.00348684168, -0.143698916, 0.0309801847, -0.0543181002, -0.0799558908, 0.190914512, -0.0614015609, 0.00774812885, 0.0226198081, 0.0531787537, -0.0618811138, -0.0585327186, -0.0788292214, -0.00366556738, 0.0347583294, -0.0325671248, -0.134057224, -0.0463110805, 0.0597175434, 0.0521154925, 0.00114774657, -0.0531816185, 0.019560026, 0.0392225087, -0.00842877384, -0.101296403, 0.14710924, 0.0299691372, -0.0620323084, 0.10974852, -0.0141659304, -0.0494842306, -0.0295206457, 0.0119519308, -0.0382294469, -0.139502227, -0.131658226, 0.0115597174, 0.0770779178, -0.0218290314, -0.0121306516, -0.0382104144, 0.060878098, 0.142750472, -0.0589798763, 0.0676200837, 0.0185247324, -0.0410691239, 0.0299137048, -0.127572939, -0.0378006473, -0.100536868, -0.0363167077, 0.00676896796, -0.167191088, 0.0212077759, 0.0868244767, -0.132884994, 0.0342110395, -0.0611182749, -0.0260481872, 0.102945745, 0.0365496017, 0.0234432518, -0.0248310417, 0.175976261, 0.0216019899, -0.00532627665, 0.00764858723, 0.027753979, 0.0405078456, -0.0206162166, -0.00527708791, 0.0114256972, 0.0365030132, 0.0336980522, 0.0692263246, -0.0243159756, 0.0986577272, 0.10393206, -0.0943767056, 0.00742093101, 0.0436499268, 0.0341592506, 0.0456877351, 0.0279276185, -0.039765738, 0.135489181, 0.233778447, -0.0658682585, -0.0471731834, 0.000448940322, 0.00922876596, 0.117229208, 0.011610589, 0.0243017413, 0.031091243, -0.0900265202, 0.0601132065, 0.00408360083, 0.0275879912, -0.118830316, -0.0615517758, 0.0681044236, 0.158631369, -0.0484357812, 0.124020174, -0.0326664746, 0.0409314819, -0.00422460213, -0.0324111953, 0.0290527269, -0.103400938, -0.107562162, 0.0932063311, 0.0250069126, -0.124122925, 0.03050589, 0.102034807, 0.138139054, -0.0296162739, 0.0276926365, -0.0569745451, 0.129586026, 0.0547338687, -0.116471387, -0.0195134766, 0.0506814942, 0.0076626474, -0.0558482297, -0.101829417, 0.069013834, 0.0300411563, 0.0648475587, 0.166248247, 0.101213507, 0.0444345027, 0.147666112, 0.0086207306, 0.0374275669, 0.0151421484, -0.0581510216, -0.0248833448, -0.0628596321, -0.133901253, -0.0859556645, -0.0856730938, 0.045230452, -0.0480204336, 0.033454746, 0.0220677182, 0.054104574, -0.0845751017, -0.00932334457, 0.0160639696, -0.0344653763, 0.0510070175, -0.0676326752, -0.034518566, 0.00499220565, 0.0302092172, -0.0518940836, -0.00955612399, 0.00382014737, -0.0239019413, -0.115307562, -0.0828005672, 0.0636793822, -0.0738432407, 0.0954737216, -0.109313734, -0.0578072183, -0.012398852, -0.0527146682, 0.0275513027, -0.0815594122, 0.00507738208, 0.045145262, -0.0461822748, 0.0274811871, 0.0118764099, 0.0133302175, 0.133594975, -0.0398499705, 0.065370582, 0.0196005814, -0.114700183, -0.107491247, -0.030636169, -0.0373892598, -0.00918629952, 0.129107028, 0.0423830003, 0.0965084732, -0.100005589, -0.115171194, 0.00263285707, 0.060572587, 0.0379161015, -0.0931825787, -0.116522536, 0.0266920701, -0.0241217595, 0.00282175466, 0.0295968801, 0.000478329137, -0.110135563, -0.0414175317, -0.0636743531, 0.0197038241, -0.00920526311, 0.0625352487, -0.0236603841, -0.138025969, -0.0883734673, 0.0917572156, -0.11933253, 0.0258444548, 0.0710579157, -0.0780234337, -0.0148170441, 0.0312691033, -0.00566856563, -0.0145191867, -0.0349283367, -0.00670860149, 0.105804041, -0.0641736388, -0.0366437323, 0.0522898138, 0.115683272, -0.0386916995, -0.215895638, 0.0518536642, 0.0728991702, 0.0477389321, 0.0112064974, 0.0782056302, 0.0881057382, 0.024451958, 0.120363623, -0.0709322169, 0.06867598, -0.0660766438, 0.00340095931, 0.149231806, 0.0184066538, -0.0856160894, -0.0739547834, 0.0312558375, -0.0619605556, 0.0516609736, 0.0347899199, -0.15554671, -0.0294578224, -0.0578455925, 0.0576982014, 0.036413908, 0.0532127656, -0.0513671227, -0.030536525, -0.0260005239, -0.0207533687, -0.01641028, -0.116865128, 0.124191687, 0.114527084, 0.0870671272, 0.119564414, -0.0358877964, 0.0894882455, -0.0142037831, 0.0589610264, -0.00495830178, 0.0118975155, -0.0367976651, -0.106736168, 0.0531613529, 0.00647791289, 0.0446007475, -0.0617889166, -0.0287456177, -0.124598369, 0.0289232414, 0.128152966, 0.0362791494, -0.0292951427, -0.0408745706, -0.0576321818, -0.0480503216, 0.161305472, -0.00748889893, -0.0536159575, -0.019543618, 0.0229161847, 0.038694039, -0.00959399343, -0.036313355, -0.0360907875, -0.0258969292, 0.0174424201, 0.005995363, 0.0753622204, -0.0476423204, -0.0331449658, 0.0135375774, 0.0225478727, 0.079924807, -0.0982389003, 0.100322366, 0.0484079532, 0.0593880564, -0.104930677, -0.0233237967, -0.121263564, -0.047104951, 0.0493723154, 0.0864522606, -0.00893124938, 0.0428383239, 0.0720678344, -0.0713310167, -0.00386607088, 0.093112953, 0.00370634254, -0.0390104242, 0.0295266621, 0.184043735, -0.00185719877, 0.0377220772, -0.0604721606, -0.0894271433, -0.10692969, -0.0459658429, 0.00398916379, -0.0968620628, 0.0383661166, -0.0810789838, -0.0860629678, -0.109189242, 0.169216365, 0.1289244, 0.0566616319, -0.0316038765, -0.0574379712, 0.0202376135, -0.0542436466, -0.025901895, -0.018552348, -0.00465473533, 0.0463921055, 0.00306424685, 0.0593580268, -0.0218768641, 0.0863000751, -0.00658572465, -0.0336344652, 0.0975641906, 0.0272094943, -0.167632833, 0.0712785348, 0.0234816838, 0.0755730569, 0.121718504, -0.0777702406, 0.0686770678, -0.050026767, 0.0416301936, -0.0960736573, 0.0664560124, 0.102550723, 0.0625562221, 0.110591643, -0.113259137, 0.0022691451, 0.0703474581, 0.0666949004, -0.0071596792, 0.061394833, 0.0293247029, -0.0631409734, 0.020673316, -0.0263614226, 0.0982172564, 0.00699460227, -0.0455927588, 0.0802026019, -0.10190887, 0.0846148133, -0.11210525, -0.0350118726, -0.0242762193, -0.000193818472, 0.0546705574, 0.0366264507, 0.134070396, -0.0260837413, -0.0177230798, 0.0196370408, 0.0894785747, -0.0395769067, -0.107305057, 0.0529573187, -0.081204012, -0.152088001, 0.0303028487, 0.0674561337, -0.0395990945, 0.0461127982, -0.0541351065, 0.00466474006, 0.00836414658, 0.104049645, -0.00101429038, 0.13354446, -0.0696410462, -0.0254141055, 0.00835372508, 0.000807271339, -0.0187259577, -0.0563195646, 0.105594195, 0.0708100349, -0.0317827202, 0.0994293988, -0.0434136167, 0.102707855, -0.0394269079, 0.0146331284, -0.00732005015, -0.0310396105, -0.0530030057, -0.0496953093, -0.0778527483, 0.00890290551, 0.023694545, -0.0329473205, -0.0327186771, 0.023676496, 0.0597901158, -0.0215158965, -0.0325211063, 0.0834325701, 0.0684324652, -0.0814330131, -0.0691422001, -0.0356172249, -0.0329068005, 0.0185153484, -0.0137839317, -0.0288640819, 0.136546835, -0.037425831, -0.0333168395, 0.0422376283, -0.0332692713, 0.0755482465, 0.0192054361, -0.0823622718, -0.0410633124, -0.0412313119, 0.138509929, 0.0316699706, 0.132271022, 0.0183287039, 0.0480044708, 0.147155046, -0.0573583022, -0.0365737379, 0.107809931, 0.0909634158, -0.0412379578, -0.123732083, 0.0469360687, 0.111640856, 0.0569434911, 0.0930527151, 0.140695393, -0.0894969255, 0.00256445911, 0.0125999935, -0.0562401563, -0.114302367, -0.0382896215, 0.0104759187, -0.0232379213, 0.0542952791, -0.034059599, -0.146358714, 0.066709727, -0.0732627437, -0.00571516529, -0.0198372602, 0.120803088, -0.105709523, -0.100433663, -0.0215995014, -0.0400962122, -0.0655378699, -0.0331503414, 0.0164581686, -0.0318296552, -0.100893125, -0.181700885, 0.120456025, -0.0762417614, 0.0831995532, -0.00903397053, 0.143906787, 0.0352139436, -0.0112549327, 0.0669031441, -0.0417459607, 0.00541909691, 0.0642425418, 0.116839305, -0.179413512, -0.067691505, -0.00389492046, -0.00482019968, 0.00230792724, -0.0782617629, 0.0633524507, 0.0558453351, 0.0827809349, 0.108852305, -0.0359224975, 0.0284109451, -0.0222191606, -0.101449154, -0.127913833, -0.109366447, 0.146415055, -0.0545229688, 0.157297999, -0.0392694511, -0.136351794, 0.0631641373, 0.0868870541, -0.047785867, 0.128236473, -0.0711336285, -0.0256616995, 0.125207156, 0.073627241, -0.0366111249, 0.0887460783, -0.139744967, -0.0566972345, 0.0924156308, -0.00253159087, 0.0565007627, 0.0418369919, -0.119484343, 0.0318732932, -0.0316493884, 0.00976659823, -0.0111968163, -0.123742029, 0.0509138629, 0.0725260526, -0.0395703204, -0.00607385579, -0.00724574691, -0.0408083349, 0.0192282572, -0.0687208474, 0.00142038311, -0.125461325, 0.0599353909, 0.084194988, -0.057588283, 0.00553785916, 0.0209137872, 0.00708530564, -0.064549908, 0.000950800255, 0.0361906178, 0.106690891, -0.0902081355, -0.010964714, -0.0176610649, -0.0183612779, -0.0169377495, 0.0292202812, -0.00526601076, -0.0592814647, -0.0923140794, 0.0702977553, -0.0418194905, -0.00336346775, 0.0736140683, 0.0709515214, -0.0671726838, 0.119039156, -0.044654049, -0.0310713947, -0.058872927, -0.0735617876, 0.111595832, -0.000629011542, 0.0473766737, -0.0703351051, -0.103621587, -0.062163122, 0.0484706573, 0.0491833352, -0.0284291729, 0.120324776, 0.0621699095, 0.0961769968, -0.112067148, 0.0347730964, -0.126400009, 0.0318991877, -0.0962366164, -0.0341994688, 0.0218884982, 0.0080213882, -0.0774020925, -0.0732281432, 0.00689242594, 0.0167558584, -0.0840547979, 0.0384579897, 0.0810027942, -0.145067349, -0.100323461, 0.00845299568, 0.0601886511, 0.0302432552, 0.0088377092, -0.153663918, -0.0154264988, 0.00787600968, 0.0539445095, -0.164799377, -0.0100836325, 0.00179879088, -0.0612194575, 0.0524255112, 0.0441213287, 0.042193003, -0.0278313346, 0.0382799134, -0.00075703254, -0.0351711512, -0.00383648649, 0.0892538652, -0.120289706, 0.0880583376, 0.0809447318, -0.0352157615, -0.0152201615, 0.0262710433, -0.108669877, 0.0415507369, 0.019583337, 0.161030442, 0.0468844399, 0.00803215057, 0.00341675803, -0.0586863384, -0.127230674, 0.0464866236, 0.020540949, -0.0430138856, -0.194104955, 0.00367502496, -0.0318855755, -0.134010583, 0.0450272001, 0.0145560429, -0.246621549, 0.0988970846, 0.0510415658, 0.0687515289, -0.0536560044, -0.0625091419, -0.0327615403, 0.0907914191, 0.0783033073, 0.0203253068, 0.0194462538, 0.0553661026, -0.0425359383, 0.0350326747, 0.128417015, 0.0408646986, 0.026424367, -0.105355956, -0.113743819, 0.126335546, -0.00976781547, -0.0702449083, 0.0934237987, -0.0495629832, -0.120837845, 0.140801162, -0.0129696168, -0.0515523106, 0.0654594451, 0.0878215879, 0.00559131615, -0.0391941629, -0.110382959, -0.0833658129, -0.0678980723, -0.121550776, -0.0277186874, -0.0747896284, -0.0528696813, 0.062489666, 0.0258378275, 0.14689526, 0.0139871612, -0.0774390623, -0.0257221013, -0.133306846, -0.027471479, -0.0779962316, -0.0114445668, -0.0644760877, 0.0602955893, 0.0901463851, -0.0512889475, 0.0411484092, -0.0123691522, -0.0285694972, 0.0619165599, -0.0283145756, 0.0895031691, -0.0317250974, 0.0182393733, 0.0494113527, 0.0265502576, 0.0284394547, -0.109676167, 0.106926247, -0.00997429341, 0.0960271582, -0.0780220181, 0.0630786344, 0.0139888963, -0.0320418403, 0.0691434443, 0.0730710551, 0.0373421013, 0.109231554, -0.0456483439, 0.188781306, 0.0167414919, 0.0248027481, 0.0556567833, -0.131824747, 0.0671918541, -0.0238614921, 0.0298387464, 0.0921626911, -0.043094404, 0.078622967, -0.0343140215, 0.0269713774, -0.0172435343, -0.0108120041, 0.0982474908, 0.0519196466, 0.0162194744, 0.118766591, 0.0149338562, 0.0667814463, 0.032377176, -0.115251333, 0.0373098627, -0.0259436853, -0.0307341777, -0.11223197, -0.091855742, -0.115036793, -0.0118110599, -0.0412412398, -0.104448631, 0.0298828408, 0.054202266, 0.0600945503, -0.0280554015, 0.0998843983, -0.0229049902, -0.0153931035, -0.0195422284, 0.0835999846, -0.00953147747, -0.0565470383, 0.107559517, -0.0194214284, -0.0247669406, -0.0479892194, -0.0300220288, -0.0323037095, 0.0216859505, 0.0141581837, -0.0876181722, -0.00716956332, -0.16756773, -0.0205360614, -0.046861358, 0.0352517217, -0.0290013291, 0.124769107, 0.0261376947, 0.0112239327, -0.0346608944, 0.062852174, -0.0236231424, -0.153502658, -0.19097279, -0.106461793, -0.0408299826, -0.125152305, -0.0721943304, 0.0340681151, -0.0453003272, -0.061441943, -0.102795735, -0.0569854006, 0.034737654, 0.0421225093, -0.0153091736, -0.0218936522, -0.146173477, -0.00829258747, 0.184158102, 0.122241288, -0.084177345, 0.168531835, -0.00641076453, 0.0334824249, -0.0122941528, 0.032062754, 0.059957698, 0.0355172753, 0.107312627, 0.0144212283, 0.0861650929, 0.0188808516, 0.0193134509, -0.145267516, -0.0889582932, -0.0842778534, 0.0916769803, 0.0411723703, 0.00554753607, 0.0037490651, -0.10848517, 0.051846154, 0.0776569173, 0.101116732, 0.112386301, -0.0098252669, -0.0481179878, -0.0171496551, 0.0795148313, -0.0189479142, -0.018890053, 0.178836018, 0.0138866231, -0.0821822882, 0.0711538345, 0.0129677355, 0.146517605, -0.0250943117, 0.0803776085, 0.0770965517, -0.0571847223, -0.00601102784, -0.0542757064, -0.0443117172, -0.0133484909, -0.102817506, 0.0237798542, 0.00735295052, 0.0711276382, -0.0795218721, -0.0454166718, 0.0172596034, 0.0610119589, 0.0483013652, 0.0160205476, 0.0464293063, -0.0604674481, -0.0779783204, -0.089457497, 0.0523129627, -0.0215199031, -0.0400521234, 0.125532493, 0.00734655932, -0.0142266527, 0.17185384, 0.0890401602, 0.0309686381, -0.00859410036, -0.00727661327, 0.0869946256, 0.0273250788, 0.0912422165, 0.0242036991, 0.0311453603, -0.020802971, 0.16884917, 0.023390457, -0.011494942, 0.0450326912, -0.0799407959, -0.0613714755, 0.0293006413, -0.0254077837, 0.0961817577, 0.0673164576, -0.106642745, 0.0756556317, -0.119609937, 0.00969868712, -0.0904721096, -0.0404048115, -0.0239201784, -0.0613796264, -0.0403573252, 0.00890928507, -0.0665615574, -0.026793398, 0.00395689905, 0.00609805994, -0.0335235782, 0.0222840495, 0.0283607394, -0.0275544729, 0.080691807, -0.0175271239, 0.0861111283, -0.101052701, -0.0350018553, -0.0074343998, 0.0489694923, -0.04479919, -0.0272994488, -0.000515452353, 0.11313732, 0.00529505312, 0.0637723953, -0.0843197331, -0.0343549028, 0.0817853212, 0.0610746928, -0.0720800161, -0.0684199333, 0.0722889081, 0.0581635833, 0.0892965198, 0.0583080053, -0.000900680199, 0.0381048024, -0.0110369334, 0.0662589222, 0.059857443, 0.0375354849, -0.0301726814, -0.0731346235, -0.0929167867, 0.054312624, -0.0291669834, 0.0284009241, -0.0290024541, 0.0465549082, -0.11410591, -0.139297336, 0.0127172079, -0.0130840633, -0.0452667475, 0.12527664, 0.00445348769, 0.112321369, 0.109566353, -0.0398729518, 0.0398472846, 0.151911288, 0.0120465476, 0.0567985326, -0.0720740855, -0.0592865236, -0.0561313517, -0.163934529, -0.0104121789, 0.0304081552, -0.0932850093, -0.0522189215, 0.045732826, -0.066893436, 0.0734580308, -0.0794622451, -0.00772430375, 0.0656402558, -0.00430299528, 0.0265939385, -0.0601608455, -0.0750281513, 0.00693067675, -0.00672144443, -0.0678872094, 0.0953256115, 0.121188894, -0.0479607396, -0.000628431328, 0.0833768621, -0.044921536, 0.0608398728, -0.0442973524, -0.0231449939, -0.0572286695, -0.0221622698, -0.0162954461, -0.041878514, -0.192133889, -0.0224961266, -0.0339366198, -0.0900944024, 0.0720057562, -0.0412492082, -0.0521879941, 0.00318414159, 0.028346613, -0.0885099247, -0.000461629592, 0.103174105, 0.0511165485, -0.0606587902, -0.033228077, 0.0603607632, -0.06066975, 0.00644999929, 0.0252265558, -0.0471164212, 0.0586018898, -0.0240608919, -0.0429954156, 0.166241214, 0.0847603455, -0.0853525251, 0.11635372, 0.0768302977, 0.0145210586, -0.12955749, 0.00712409057, -0.0659702271, 0.0281008687, 0.0699765086, -0.013855814, -0.0146459248, -0.0388546735, -0.00915924273, 0.0566541813, -0.0674254894, -0.0491815172, 0.0648297444, 0.0113611426, 0.00847549736, -0.00886135548, 0.0137894098, 0.0638384819, 0.00420870353, 0.090354532, -0.0619390905, 0.171965525, 0.187458158, 0.0527163669, -0.043487113, -0.147247821, 0.033757668, 0.0188759882, 0.00401037186, 0.0405628979, 0.0586508065, 0.0865700543, -0.152879521, 0.0159267597, 0.0652434751, 0.0097250808, -0.0354112461, 0.084558472, 0.0526328981, -0.0632263646, -0.00106894691, -0.00946753658, -0.100315794, 0.0185935926, -0.14264448, 0.0788547918, 0.0478432029, -0.0242307168, -0.0160921402, 0.0731759369, -0.112183109, 0.0706517175, -0.0978575125, 0.0518998057, 0.0293896683, -0.00136082526, 0.120696381, -0.0453348346, 0.091407612, -0.0290567577, 0.074232772, 0.0126435924, 0.0418775305, -0.0812566578, 0.105791613, 0.0246349741, -0.0152652264, 0.018106509, -0.0737674311, 0.150271326, -0.215129614, 0.0300735831, -0.113408081, 0.0650518909, 0.0222016051, -0.0797848776, 0.0827352777, -0.00763365626, -0.0335478373, 0.0528862737, -0.0798040032, -0.0421789326, -0.0122761875, 0.0529228002, -0.0549547821, 0.100646958, -0.00234978111, -0.00746429106, -0.0555395149, -0.173543662, 0.0105401687, 0.00531535782, -0.0594168641, -0.129437089, -0.00683795381, 0.108063489, -0.00755071267, -0.109399363, 0.114717439, 0.104691789, -0.0698268041, 0.028761737, -0.0772326216, -0.044201903, 0.0836420134, -0.0357559994, -0.0959446877, 0.016582489, 0.104911201, 0.0475973561, 0.0710235164, 0.0856918842, -0.0608736686, -0.00993047655, -0.0893506557, 0.0339855142, -0.0493616611, -0.137649253, 0.130620331, 0.0248426832, 0.034240786, -0.0214420035, -0.0842188001, -0.0435745195, 0.115031354, 0.0328332856, -0.0987135395, 0.0862497985, -0.0302738771, -0.0708632991, 0.0572016239, -0.0762674138, 0.0691025257, -0.037434496, 0.0217761323, -0.0370992795, -0.0456319712, -0.0147401839, 0.0181538314, 0.0726551414, 0.00899257138, -0.0270052366, -0.0836559385, 0.0980546325, 0.061095994, 0.000828944147, -0.057132408, -0.0950826257, -0.0256363545, -0.0929112732, 0.0425492786, -0.0024689571, -0.0306376722, -0.0523114949, 0.101528853, -0.0523844846, 0.0640822276, -0.0737137944, -0.137838081, -0.0076995492, 0.136963502, -0.0478355587, 0.0325510614, 0.111381933, 0.117927238, 0.10202948, -0.0806948617, -0.0648256764, 0.133120418, -0.00224611163, -0.0104684122, -0.000627145171, -0.0603796095, -0.0283243842, 0.0665622652, -0.142835289, -0.0274916962, 0.00142771378, 0.0558498278, -0.0643476769, -0.00676162913, -0.053988494, -0.00484051928, 0.0715775266, 0.0154943559, -0.00997336302, -0.0383435152, -0.0402208492, -0.0872833431, -0.0233834311, 0.145907968, -0.0435767137, 0.0957608968, -0.028151758, 0.0649675578, 0.190936983, 0.06481345, -0.000855347142, 0.162423104, 0.0394274928, -0.0496312082, -0.0455062985, -0.222967058, 0.0792990401, -0.137906283, 0.149159878, -0.0124643315, -0.0468844511, -0.102703512, -0.0351455733, 0.117990598, 0.106325418, 0.0819974691, 0.0866898969, -0.0903978422, -0.0957485512, 0.0534124188, -0.0865085721, -0.0171378478, -0.0201135948, 0.065308623, -0.0143852551, -0.102555662, 0.0376451202, 0.00103474874, 0.0305470023, -0.0194290355, 0.0443652645, 0.0108052883, -0.050805755, -0.0560781658, -0.0568571538, 0.0239526071, 0.0536852479, 0.0659016892, -0.00530015863, -0.113984883, 0.00188809633, -0.00598471193, -0.0527855679, -0.00734733976, 0.0682486147, 0.0730547756, 0.074361369, -0.0592212304, 0.123616904, -0.0555166192, 0.0351577625, 0.0318785086, -0.0688275099, -0.0140260011, -0.113746852, 0.0592081994, 0.0959497392, 0.0216836743, 0.0712018013, -0.0673099607, 0.103493616, -0.0469349474, -0.0424249321, 0.0547314994, 0.111671314, 0.0592016429, 0.0379485413, 0.083008185, 0.0462957546, -0.00969570689, 0.14310959, 0.0635819286, -0.120568633, -0.105409615, -0.0384053178, -0.0211726725, 0.0320640057, 0.0474545248, 0.00662817247, 0.0142514175, -0.0209808461, 0.0332401618, -0.048783768, -0.0646389797, -0.0202070791, 0.0606515482, -0.0727318227, -0.0261643417, 0.0628451109, 0.011384422, 0.0278099049, 0.0245810207, -0.0205679573, -0.080847986, 0.0436471552, -0.0715225264, -0.0238368548, 0.0790551603, -0.00950204767, -0.0530045927, 0.105068803, -0.00632932503, -0.0153049761, -0.0635962635, -0.00862434041, -0.0106838793, -0.0973426327, -0.0257954448, -0.124228589, 0.0763272569, 0.211909845, -0.0236179382, -0.0810620636, 0.0319620222, -0.002163684, -0.0705077499, -0.014357605, 0.0262934938, -0.0343292169, 0.0361409076, -0.103956789, -0.0340285748, -0.0602297559, 0.174030885, 0.0790194348, 0.0161414575, -0.0282022953, -0.0180360191, 0.0213341229, -0.00993218832, 0.0482341982, -0.0360355154, -0.0160495229, -0.0549918339, -0.0281617641, -0.215279579, -0.0329001322, -0.13107945, -0.0194422733, -0.0811705217, 0.0703393519, 0.0948659852, 0.0860955417, 0.00298020244, 0.0174867325, 0.104314342, 0.00757317059, 0.0873776898, -0.109705932, -0.00641422626, 0.0342337042, -0.0431328341, 0.140281439, -0.0141475201, -0.00715182908, -0.0821413025, -0.166424349, 0.0175308995, -0.00971734151, -0.0294843055, 0.024879612, -0.0663464367, 0.0145991985, -0.113094434, 0.0108234081, -0.0424563773, 0.0702047348, 0.146885216, 0.0739716291, 0.0807786584, -0.0294531658, 0.0644897372, 0.0465509035, -0.140208289, 0.0105558988, 0.061719127, 0.119625054, 0.122069746, -0.00659644231, -0.0888892189, 0.0391467549, 0.0318171196, 0.0392123535, -0.0693224147, 0.03465968, -0.0476835184, 0.0632190555, 0.00752518512, -0.0693088621, 0.0556228012, -0.034609288, -0.0562940314, -0.0935908407, 0.0894165337, 0.0460318811, 0.0946106911, 0.0970253497, -0.0378115699, -0.0580373146, 0.00685130805, -0.0240787845, -0.0655495301, 0.0920475721, -0.0572968684, 0.0907118097, -0.000337135047, 0.0958020017, -0.00220216811, -0.105195656, -0.00343512697, 0.135109693, -0.0170508716, -0.0159937311, 0.0629626587, 0.038738329, 0.043182198, -0.149704367, -0.0275805071, 0.0830653906, 0.135414079, -0.0911396965, 0.0255063958, 0.0678325221, 0.117846638, -0.0977108777, -0.0146968234, 0.0410707369, -0.0079479944, 0.00758772902, -0.0975005254, -0.0584881231, -0.0411358178, -0.0954357386, 0.0131467246, 0.0884373337, 0.0314341597, -0.0540474504, -0.131020159, 0.00755074248, 0.00428653974, -0.0513308756, -0.144464895, -0.0465611182, -0.0106990952, 0.166800812, 0.0565037616, 0.0638967529, 0.0368259996, -0.00591901131, 0.0741597861, -0.0822639316, -0.0216166861, -0.0142547525, -0.105811425, -0.129464537, 0.00880646706, -0.124055475, 0.0486171208, -0.0312933289, 0.0335986391, -0.0956721902, 0.0666646883, 0.00134075899, -0.0241167396, 0.0286073964, -0.0168476515, 0.0488022156, -0.204614803, 0.119252726, 0.0173368528, 0.0164972693, 0.0484212488, -0.00370501354, -0.0814251751, 0.0140291722, 0.0981728882, 0.0892434344, -0.0246675052, 0.0102536585, -0.0505557954, -0.0823860988, -0.132501259, 0.0507950634, -0.0830733478, -0.0402466208, -0.121927015, 0.0505604818, -0.0569023155, -0.217993006, 0.0493810214, -0.069898285, -0.109336302, -0.00529927202, -0.0074481531, 0.00809708796, 0.0706185475, -0.0761374906, 0.0308077484, -0.0390697792, -0.0364637785, -0.120178454, 0.0378564, -0.014556909, -0.0459425524, 0.0791534483, 0.00495853275, 0.100030519, -0.0384478159, 0.0553810075, 0.0197767988, 0.0948791057, 0.0416829251, -0.0923174024, 0.0716896504, -0.0207008142, -0.128450945, -0.00730367564, 0.0726294816, -0.0313276686, -0.143590629, 0.0255806707, 0.0434266813, -0.0224328507, -0.0891770571, -0.0527072251, 0.0488626324, -0.0659937114, 0.0346077457, 0.00469872728, 0.0800054744, 0.0616751239, 0.133224607, -0.0785946772, 0.0515422523, -0.0605530702, -0.0692069903, 0.0869517401, -0.113503605, -0.0688326433, -0.0344808921, 0.0939441845, -0.0693285838, -0.129364058, 0.0331576131, 0.00330016902, -0.060806904, -0.0473938957, -0.0382475108, 0.163586751, -0.0755013227, -0.00396516128, -0.0122583583, 0.0928661376, -0.0399830714, -0.0281913932, -0.0356783494, -0.0565432012, -0.174874783, 0.00862659141, -0.0120314248, -0.10457021, -0.0178394355, -0.0528360493, 0.0537608564, 0.00123192556, 0.00244560465, 0.12382669, -0.119202323, 0.0578210056, 0.0637606233, 0.00625109719, 0.0115161706, -0.0988153443, 0.056037128, 0.0449979082, 0.0104337549, -0.0543784313, 0.0196551364, -0.0442993864, 0.0959204882, -0.10798794, -0.116974369, 0.0091380924, -0.0100636166, -0.0393831953, -0.0654226393, -0.0669216812, 0.0244851075, 0.0065101916, 0.00610528141, -0.106983304, -0.106025919, 0.00486871041, -0.0126079768, -0.0479022302, 0.023387013, 0.0537120663, -0.0453917272, -0.0491301902, 0.0628812015, -0.00236194581, -0.00814808439, 0.0227814056, 0.0942559615, 0.020572044, -0.116628557, 0.025704002, 0.0473104045, 0.00108542852, -0.0587278195, 0.0383057073, -0.0542852655, -0.0688491538, -0.0918664262, 0.00669162348, -0.10958086, 0.122720167, 0.0522697493, 0.0986699238, 0.106197536, -0.0432841703, 0.169561595, 0.117332898, -0.101258755, 0.0558797084, -0.125172824, 0.0544885956, -0.0112890974, 0.0185600091, 0.0578551888, -0.0466390587, 0.0376987047, 0.0864820108, -0.00115627423, -0.103971407, -0.00704975054, -0.0842340961, -0.204760641, -0.0627957657, 0.0418024473, -0.0980946198, -0.0473582223, -0.165247455, 0.0316605121, -0.00382990995, -0.0291041918, 0.0644813552, 0.0037751901, -0.0172346979, -0.0422124676, -0.0885811895, 0.0166758206, -0.0435407236, -0.0773774311, -0.0941780284, -0.0396579728, 0.0649015829, 0.0159331262, -0.0516304076, 0.0835015997, 0.00978837535, 0.0443133749, 0.0297001377, 0.02662565, -0.0238366965, -0.0462984852, 0.102302514, 0.0762243196, -0.0488283187, 0.0705497861, -0.0327157043, -0.11041598, -0.131304458, -0.0191016868, 0.0133641809, 0.0544066913, -0.0260483604, -0.0965383798, 0.0911923945, -0.0630287379, 0.0826769471, 0.133001104, -0.00473366678, 0.117705062, -0.0240012761, -0.00132794864, 0.0508191586, 0.0196961872, 0.159875497, -0.130224124, 0.0234762207, -0.0394301713, 0.018752683, -0.126942426, -0.0310703404, -0.0265759863, 0.0904723406, 0.0263345651, 0.000180898234, -0.00895390101, -0.139537156, -0.00722809602, 0.00720465649, -0.0559882782, -0.0860758871, 0.127098158, -0.0140588926, -0.0518677309, -0.0136835892, -0.0306002814, -0.0346528962, -0.0281581506, 0.0666721463, -0.115534246, -0.0981145948, -0.0289623868, -0.042298682, 0.0434158035, 0.0336587578, 0.0614327639, 0.0575813316, 0.0614780337, 0.0796466991, -0.0453872308, -0.0191985294, 0.135225505, 0.123685859, -0.0242740791, 0.0496836677, -0.0200163014, -0.00225748867, -0.0373399705, 0.00826786831, -0.014817981, 0.0557427146, -0.0234015342, 0.0436130874, -0.00313477032, 0.0691500381, 0.0741273835, 0.0460153595, 0.0242686737, -0.104999177, -0.0285043865, -0.171705365, 0.145800456, 0.0221375152, -0.00735259522, 0.0132935327, 0.0232473984, -0.112734877, -0.0114636961, -0.0499154553, 0.0371822603, 0.144290581, -0.0236323997, 0.0746450275, -0.00084541738, 0.0358160064, -0.0982175469, 0.0101916995, 0.0164498053, -0.0282862056, 0.112586729, -0.0157094374, -0.0454060249, 0.0233968291, -0.048598811, -0.071312651, 0.0603617281, -0.0299381651, -0.001147056, 0.0363889188, 0.0820527822, 0.0915727168, 0.00140509382, -0.0425595418, 0.0359408632, 0.0342875011, -0.0242629163, -0.0147682372, -0.0239619911, -0.0616740361, -0.106484808, -0.00417627115, -0.0359819755, 0.178155974, 0.0617378056, 0.00666147145, 0.07771945, -0.128619179, -0.063391149, -0.0276715122, 0.02143934, 0.112703092, -0.048061125, 0.0585327521, -0.0517405607, -0.0120576713, -0.0157191195, -0.14012593, -0.0363316238, -0.0819730535, 0.027305495, 0.0567959249, -0.00592879578, 0.0371960476, 0.0609055422, 0.0134695498, -0.0132031692, -0.0557713658, 0.015527321, 0.0689506158, 0.104819506, -0.014489511, -0.0784410834, 0.0254593417, 0.0180023275, -0.0046950113, -0.147947267, -0.0200401265, 0.106144421, -0.0275860094, -0.0517215878, 0.0516379327, 0.112819403, 0.0810719505, 0.034373235, -0.0147770941, 0.0814909488, -0.119913943, -0.0797332674, 0.018588502, -0.0902142748, 0.0192847736, 0.0663855523, -0.00207715854, -0.0844640508, 0.0395605639, -0.0880021155, 0.0426400639, 0.0728933513, 0.0677083433, -0.0474901125, 0.00312681869, -0.14532721, -0.111008584, -0.0410129428, 0.0849896818, -0.0987597853, 0.0398582518, 0.0964793861, -0.0304511748, -0.153164774, 0.00261903834, -0.0031320611, -0.0169175528, 0.014321099, -0.0595640317, 0.0555091128, -0.0140340831, -0.134952247, 0.00902788155, -0.108637534, -0.0187828317, 0.115464345, -0.0165707469, 0.119169354, -0.0362934433, 0.00672626123, 0.0907325149, -0.00682189502, 0.146521851, -0.0830077678, -0.120897137, 0.127929941, -0.115087472, 0.0116726132, 0.0962724537, -0.045083411, -0.15104124, 0.0840260535, 0.0407922938, 0.0877076387, 0.0777267292, 0.0350440107, -0.0656366274, 0.0713185966, 0.0618479177, -0.10615126, 0.0526302494, -0.0329756998, 0.160746917, 0.0684841126, -0.0272260159, 0.0634056702, -0.1046855, -0.0855556726, -0.0170933641, 0.000779412687, 0.0131857395, 0.0752171651, -0.048603531, -0.0176196843, -0.021763932, -0.0501052067, 0.0336745158, -0.0360268988, -0.0449153185, 4.29404899e-05, 0.0571754873, -0.0033179298, 0.0603400432, 0.168848693, -0.0462715253, 0.0458389819, 0.029579103, -0.0101604685, 0.033889018, 0.0622398555, 0.051276058, -0.0375341959, -0.0438668318, 0.0143896788, -0.0366873965, -0.00446784124, 0.0593102835, 0.0402583517, -0.0951602682, -0.180572614, -0.0796765611, -0.190664366, -0.0470530353, -0.0576060265, -0.0824119672, 0.0122747859, -0.110321932, 0.03454623, -0.0523498654, 0.0735493973, -0.0132928854, -0.00104576163, -0.0827548802, 0.0604652017, 0.0155662512, -0.0757914558, -0.0429328866, 0.0148150176, -0.0697317421, 0.0528019294, -0.0969544649, 0.111104771, -0.196005717, -0.0987585634, 0.0712072104, 0.00649388041, -0.0332998447, -0.0260967277, -0.0369820669, 0.0213686749, 0.0171974748, 0.123341791, 0.000567279756, -0.056413956, 0.0690545887, -0.0805647224, 0.00467581116, -0.0327795148, 0.0471625067, -0.0631929487, -0.0601705611, -0.0225944482, 0.0228578821, -0.0516695455, -0.0419914871, -0.0148608834, 0.196023926, -0.0900745094, -0.0365177616, 0.0983268544, -0.0211878717, -0.00590895489, 0.0804941356, 0.0306762606, -0.0259889401, 0.0064141457, -0.0201188475, 0.045681648, 0.116616346, 0.031765677, -0.056428425, 0.0712942854, -0.0335800052, 0.124227926, 0.135445073, -0.103780881, -0.0415219292, 0.0239031091, 0.0332115144, -0.0683033392, -0.112730265, -0.013637932, -0.0741279274, 0.1100403, -0.0143038603, 0.111749701, 0.0307638887, 0.0331706181, 0.0272779148, 0.0609667897, -0.055300042, 0.0078124404, -0.0154411234, -0.0340315588, 0.0390034989, 0.107351936, 0.0303496346, 0.00232033804, 0.0530956686, 0.0861958787, -0.0758782923, -0.015927013, 0.0752552003, -0.00799689069, -0.0265250653, -0.010232335, -0.0755146593, -0.0187492482, 0.0497631207, 0.0227313042, 0.086643979, -0.0903109387, 0.0361445211, 0.0851439014, -0.0371047631, 0.0125641655, -0.0443306118, 0.0184564423, 0.0641649738, -0.00154084526, -0.0506638959, -0.0268343985, -0.0993898287, -0.132515728, -0.0298210531, 0.031581834, -0.0476533435, -0.0211789683, -0.0385781489, -0.0643052086, -0.102327302, -0.0622971244, -0.0804271996, 0.0161505565, -0.083058618, -0.0220388602, 0.0415044576, 0.00775893964, 0.100917056, 0.0302919801, 0.0594701506, -0.032192573, -0.109479927, 0.00380911306, 0.0257576611, -0.0429031029, -0.0120052826, 0.0295684189, 0.132145762, 0.0901322439, -0.0651533455, 0.0392933302, 0.0356644392, -0.0225292798, -0.1250287, 0.0637708455, -0.12362133, -0.0713968426, -0.00440163491, -0.129764214, 0.0308040008, -0.123995245, 0.0727155209, 0.0359779857, 0.0557515621, -0.00788295828, -0.0418291837, -0.0556169599, 0.0073938407, -0.0131131299, -0.09903799, 8.13147053e-05, 0.0302125141, -0.0278899334, 0.0535467304, -0.0798689798, -0.0573887378, -0.0173641667, -0.00622116029, 0.0335880443, -0.0624668077, 0.0515625998, 0.11595048, -0.0661625415, 0.10432899, -0.11084725, 0.0875949562, 0.0392709337, -0.0364517421, -0.0743830502, 0.00235208124, 4.60073352e-05, -0.0377354324, -0.0205002762, 0.139248654, -0.00987232476, 0.0279238559, -0.0376371965, -0.0748126581, -0.14912799, 0.0279988665, -0.0754584074, 0.0367791727, -0.0684543997, -0.120797753, 0.210929647, -0.0683470666, 0.0416743346, -0.00167389307, -0.03560495, -0.0740633756, 0.0182297807, 0.0579238199, -0.0464916304, 0.0312767625, 0.0230260603, 0.00420898199, -0.00905129593, -0.0361692533, 0.0551778674, 0.0748246461, 0.0900884718, 0.106486678, 0.046182286, -0.0436386056, 0.0318417326, -0.0593780093, -0.0390714593, -0.00232599862, 0.0168671533, -0.00128097087, -0.0234770365, -0.207413524, 0.091397658, 0.0404496193, -0.0955121964, -0.0953916684, 0.0376782902, 0.0643178821, 0.0802147463, -0.069396995, -0.00916909426, 0.0369172953, 0.0255105644, -0.0491899848, -0.032136552, -0.107756861, 0.0107436292, 0.019768646, 0.0980418399, 0.0568639934, 0.0204656459, 0.0187228061, -0.00544637628, 0.0828665942, -0.00240248069, -0.0522129759, 0.0143650025, 0.0482954122, 0.0405194908, 0.117483482, 0.0239349958, 0.00080441311, -0.0541618094, 0.0940204933, -0.105444238, 0.118430451, -0.0870203078, -0.123753317, 0.0329259448, 0.0420681946, 0.132282391, -0.0484123155, 0.000465761404, 0.146358669, 0.177483767, -0.0771356225, -0.0731008649, 0.0138120726, -0.0384135433, 0.0724786445, -0.0743359923, -0.034141764, -0.0258353278, 0.0891263932, -0.0614453405, 0.149894118, -0.0627272725, -0.0523161069, 0.0335989147, -0.041771844, 0.0213093907, 0.0459769294, -0.00445639715, -0.0234814584, 0.103136525, 0.0533659272, -0.022723956, -0.0382430181, 0.0330411904, -0.147755891, -0.0439336523, -0.10285791, 0.0145746469, -0.0746227801, 0.0824759454, -0.067650646, -0.11463163, -0.136612028, -0.0311640576, 0.00981829129, 0.00207894668, -0.0804388374, 0.0687851235, -0.00379346497, 0.0771161541, -0.130354851, -0.0437753089, 0.00205173716, 0.0463164002, -0.0175507255, 0.0375224687, 0.10031689, -0.0767227262, 0.0601984486, 0.0444888584, -0.0265136808, -0.084761098, -0.000143888872, 0.0326584131, -0.0210909694, -0.0118333716, 0.118986979, -0.00320465397, -0.0930535793, -0.0411692336, -0.0462614559, -0.0252511725, -0.0238584261, 0.0695445091, -0.00723118708, 0.0638550073, -0.0812215209, -0.171835899, 0.055236809, -0.0854737982, 0.00169022381, 0.108785376, 0.0245490521, -0.0220617913, -0.121044368, 0.0211217031, -0.0161820352, 0.151667625, -0.092914477, -0.110812977, -0.0416993797, 0.0688993037, 0.0716673583, 0.0323226042, 0.0435284115, 0.0607336052, -0.048121959, -0.0266444664, -0.0232259948, -0.012700025, -0.107227765, -0.0672004223, -0.207843721, 0.037615329, -0.0249993652, -0.0910415351, 0.157347187, -0.0610164329, 0.191035032, -0.0491201542, -0.0428905301, -0.0213949382, -0.0874956697, 0.10035333, 0.0531928726, 0.0230856277, -0.0840579718, -0.0603243746, 0.0622626655, -0.0587715544, 0.0670978352, 0.0656613708, 0.00271900184, -0.0609509796, -0.0492823869, -0.0401115902, -0.0509398505, -0.0496883169, 0.065441981, -0.0381773636, 0.0243011992, -0.00364368455, -0.00995516777, 0.0427191481, -0.127105564, 0.0633584261, -0.0931454301, 0.049144771, 0.0516123921, 0.0413496122, 0.00990300626, 0.048000738, -0.0535469465, -0.0971256196, -0.0142761804, 0.0540780574, 0.0527291261, -0.0447016656, 0.081862554, -0.0444602482, 0.0722750202, -0.0399135537, -0.0010391192, -0.0163113624, 0.0631549135, 0.0347271562, -0.0251329131, -0.0387175083, 0.0111792628, -0.0346063338, -0.071156919, -0.046510119, 0.107706293, 0.0824263543, 0.0127300788, 0.127644643, 0.016475996, -0.0238917824, 0.151583269, 0.114829041, 0.0530352108, -0.0179952569, 0.0800536871, -0.070317775, -0.152198091, -0.04821942, -0.0494440272, -0.024356192, -0.0940830857, 0.0912103504, -0.119127162, 0.066063486, 0.00056592375, -0.011524695, -0.00827786606, 0.0117728822, -0.0889376029, -0.00546765141, -0.0990630835, 0.145165592, -0.00199469179, 0.12126606, -0.0608006977, -0.124840729, -0.0649535656, -0.144844249, 0.0948657542, 0.0110113937, 0.0435435511, 0.0776191503, 0.0173303783, -0.0691903085, -0.0406034701, 0.0872050077, -0.0880143195, 0.021160692, 0.114508845, 0.157790467, 0.0701552182, -0.140762731, 0.0232453775, 0.0812149644, 0.0195620134, 0.0553476885, 0.00700753927, 0.0144191021, 0.0325794406, 0.00836092979, 0.00485529378, -0.150897592, 0.137030959, -0.0338992923, -0.00199312624, 0.0158948619, 0.0711862817, 0.0803703815, 0.00394163653, 0.0166742392, -0.0637132823, 0.0576172471, 0.0989794806, 0.0588038862, -0.017602291, 0.0131374076, -0.103191964, 0.149016008, 0.0303576104, -0.00741250627, 0.0757397935, -0.014678305, -0.0112621728, 0.03361753, 0.0766832829, 0.0150260366, 0.0720072687, 0.140976176, 0.0125573575, 0.0717029348, 0.00362505531, 0.0787613168, -0.084628731, 0.044434987, 0.0376896113, -0.0569761284, -0.0480788872, 0.0425903611, 0.0584106147, 0.149757862, -0.00124625303, 0.0625538826, 0.0381772146, 0.00189108262, -0.0102716405, 0.147797242, -0.0874876529, -0.0679499805, -0.00844030268, 0.0668255314, -0.0102202641, 0.0443724021, 0.00881034881, -0.0599477515, 0.0419975035, -0.109376848, 0.031993825, 0.175400287, 0.0698224381, 0.0410628542, -0.150160089, -0.0284209065, 0.022347793, 0.00905410666, -0.0653152615, -0.0166206267, 0.21127218, 0.0454411879, 0.103180595, -0.0458617359, -0.0995125696, -0.0363291949, -0.0063140206, 0.0859165043, 0.0356240943, 0.0178990569, 0.0507258661, -0.0424911156, 0.032425534, 0.0798085704, 0.013637729, -0.072872974, 0.0755365044, -0.15487203, 0.0912024528, -0.121919304, -0.0774344206, 0.0649062693, -0.047781039, -0.0749223232, 0.114782691, 0.0160173289, -0.00308426097, -0.0619944185, 0.0919422507, -0.0676485077, -0.0958780199, -0.0106051993, 0.10275393, -0.0781324804, 0.0431928039, 0.00466829911, -0.0837497413, -0.017176494, 0.0481531695, 0.138138577, 0.105663054, 0.00645310851, -0.0261352975, 0.0743861869, 0.0354747064, -0.0858714581, -0.109296694, 0.069152981, 0.029206302, -0.17600356, 0.0795082301, -0.0715349987, -0.0060289707, 0.0259194784, -0.0387955941, 0.0371407866, 0.170553535, 0.0257288963, -0.0508159474, -0.0873826891, 0.0374071039, 0.0141317174, 0.00928837713, -0.0462122709, -0.0323836878, -0.111822888, -0.0685174242, -0.11734613, -0.0474074483, -0.0817076787, 0.0350165591, -0.154563427, 0.0498186871, -0.0998867452, 0.0855002999, 0.0407505259, -0.0847005695, 0.126987442, 0.00445590727, 0.148815557, 0.0157598257, -0.0677889213, 0.0678885877, 0.103936262, -0.0291266404, 0.108563244, -0.0531429797, 0.0151067507, -0.0193862207, 0.0237437859, -0.0711940601, 0.0665370151, 0.0799864382, 0.0235979799, 0.0302098636, -0.0391180962, 0.109693781, -0.0150751481, -0.0459537059, -0.123312064, -0.0431641638, 0.101107523, 0.0692357495, -0.0784172863, 0.0979446694, -0.029822316, -0.0326684006, 0.058933042, 0.0962768197, 0.0850250125, 0.032953918, 0.0947572589, -0.0437288508, 0.0137972319, -0.016414253, -0.00187447667, -0.0200755466, 0.0115629043, -0.0379117168, -0.0243147463, -0.0448954776, 0.0678378791, 0.000306433998, 0.0608597174, -0.0208371188, -0.0125763938, 0.00191673636, -0.0388574079, 0.0198504198, -0.0477382392, 0.0470644236, -0.0107967202, 0.173992619, -0.102686241, 0.0256157219, -0.0265013464, -0.163954511, -0.155132473, 0.12658456, 0.0500281639, 0.113883637, -0.00256442651, 0.0142556829, -0.0291736908, 0.0763308406, 0.0677200407, 0.0141491592, -0.0876829028, -0.0043666102, 0.0281589571, 0.0958286226, 0.0770577639, 0.0776152313, -0.0528775752, -0.0903838351, 0.0163058825, 0.00771669205, -0.0348566175, 0.0437220633, -0.0509710833, 0.0560960732, -0.00657285191, -0.0746331811, 0.0848636627, -0.0706262589, 0.104398347, -0.00784252677, -0.0019404497, 0.0469817668, -0.0435572118, -0.00113693834, -0.0457589179, 0.010874318, -0.0671563074, 0.024623489, 0.0105352551, 0.132269993, -0.0817873329, -0.0788935944, -0.040544644, -0.0617846958, -0.045770146, -0.0200390257, -0.145366877, -0.125423431, 0.0690955371, 0.0694849268, 0.0396142192, -0.0329445079, 0.0800578892, 0.0373657644, -0.0451677516, -0.0645712614, -0.0983189866, 0.00463890284, 0.0835429803, -0.0858966112, -0.0550517738, 0.0273464136, 0.0102375317, 0.0260891337, 0.0637064651, 0.00832006708, 0.0627907887, 0.0263583213, -0.0573627055, -0.0497084148, -0.123706594, -0.0853701085, 0.00854441524, 0.0208358113, -0.00285715237, 0.00765209273, -0.0266407281, -0.011619661, 0.0538106933, -0.120938472, 0.0332855321, -0.00340719614, -0.0140140066, -0.0576705113, 0.0325996391, 0.00708473613, 0.0657776147, 0.125871018, -0.0396783389, -0.0111825448, -0.0575863793, 0.101352975, -0.00209203176, 0.0176176727, -0.0766469836, 0.0313168392, 0.117277868, -0.0965819955, -0.103153199, -0.12177901, 0.0318619497, 0.0340569839, 0.0417677611, 0.205428436, -0.0218155142, 0.0979215279, -0.0488391891, 0.0437722132, 0.0320034884, -0.176868066, 0.0120335966, 0.0552526861, 0.13601996, 0.00721526891, 0.0537095554, -0.00682887249, 0.066698432, -0.0331088603, 0.058147911, -0.00401602685, 0.122633085, -0.0158447456, 0.142422378, -0.0176462829, -0.0290186554, 0.0217498466, 0.094007045, 0.0252387803, 0.00824793242, -0.0841873437, 0.122685328, 0.0434680283, 0.0487815365, -0.00721960329, 0.0800359696, 0.104408838, -0.0127684064, 0.0803305358, 0.0346615277, -0.032716807, -0.011786636, -0.0229381695, -0.0916494429, 0.0812630504, 0.0130644422, 0.027639389, -0.0231682099, 0.0505290926, 0.0093316352, 0.11424952, 0.0581807382, -0.0550244935, 0.0636840761, -0.0720747635, 0.10009405, -0.0246030726, -0.0192512758, 0.00266349874, -0.0312189572, -0.0594217815, 0.0872601718, -0.0480652973, -0.122673392, 0.0865379944, 0.137365401, 0.037465483, 0.0619018823, -0.0269445628, -0.0328418948, 0.110974364, 0.0480593592, 0.0864270777, 0.0263310969, 0.00914893672, -0.00284557976, -0.0217671227, -0.208772793, 0.0288814195, 0.082782194, 0.0077932477, -0.079423517, 0.0557791069, -0.003898561, -0.0291814711, 0.0399448611, -0.212592274, -0.126046807, -0.0656942427, -0.00784858316, -0.0898812488, -0.038078744, 0.00671042874, 0.0882877707, -0.106805675, 0.0206672121, 0.041465424, -0.0600041747, 0.0516393073, -0.0254743993, -0.00919895619, -0.0451346785, 0.0543551184, -0.0814894438, 0.0576454438, -0.0658828095, 0.104196236, 0.104056939, 0.0577372834, 0.0187297054, -0.1470038, 0.0328220278, 0.170873776, 0.0212486815, 0.00120717101, 0.0415091738, 0.0503896177, 0.0504891835, -0.114958778, 0.0143279154, 0.0389872454, -0.13502562, 0.104704447, 0.0744781494, 0.0312258564, 0.033509139, 0.00126305455, 0.0864359662, 0.0316561647, 0.0597085692, 0.111281879, -0.106449686, 0.0440641195, -0.0202647336, -0.0856270716, 0.0558689423, -0.0269347504, 0.0359246768, -0.00160080194, 0.125313014, -0.0114528965, 0.00402942672, -0.00101586059, 0.137872115, 0.0583958626, 0.00933099166, 0.124417253, -0.139215901, -0.0709310174, -0.147631377, -0.0317863114, -0.0459677838, -0.0470133126, 0.0606892928, 0.00546924025, 0.00531811826, -0.0243411474, 0.103531994, -0.0519852005, 0.0847287029, -0.044240281, 0.0635881126, -0.0433895402, 0.0413641483, 0.0175644141, 0.00655454025, 0.0130689368, 0.0702279434, 0.0816664398, -0.048228085, 0.13485229, -0.0109039508, 0.103604622, -0.0530207232, 0.048280403, 0.0366703942, -0.139046192, 0.0208499897, 0.0570953153, 0.0474857166, -0.0780786127, 0.0406286307, -0.023971118, -0.0951811895, 0.00127734989, -0.0205095876, -0.0751637295, -0.0296861902, 0.0369220525, -0.0240838528, 0.0758907795, 0.0400747061, 0.0179445073, 0.00428873487, 0.0070068296, -0.0846178532, 0.00317023322, -0.133584976, -0.0213891938, -0.010071286, -0.0526180975, -0.0439036749, -0.0216051992, -0.121510625, 0.0654005706, -0.0649946854, 0.0866615921, -0.00906985719, -0.11152412, 0.112167574, -0.0759050325, 0.0826534778, 0.0364894494, -0.0107544642, 0.0045947358, -0.0329279341, 0.159991831, -0.0640158802, -0.0484168828, 0.00337100029, -0.0512236133, 0.0678056479, -0.0402449071, 0.0908964649, 0.0604753233, 0.0151774399, -0.0899197906, -0.0495723039, 0.213968858, -0.00480384473, 0.0268741772, -0.107549869, 0.0347231999, 0.0437693372, -0.0361597687, 0.0470806845, -0.044883579, 0.0238408744, -0.0446516797, 0.0489419661, -0.0254730321, -0.0200302601, -0.104077362, 0.062718153, -0.0531329736, 0.0116707636, -0.117419451, 0.0254259072, 0.0750542581, -0.00397553854, -0.0665199682, -0.0184707958, -0.00270925183, 0.0763828158, 0.0337355435, 0.0279260315, -0.0583564714, -0.0531061068, 0.0229404271, 0.0293381512, 0.0615486503, 0.0824794471, 0.0113682449, -0.0790008307, 0.00741539523, 0.0823355466, -0.0864413232, -0.116274506, -0.000888613984, 0.0231170058, 0.0744010955, -0.000226739794, -0.0138292881, -0.0131120011, -0.0975422934, -0.0224729143, -0.0196888447, -0.140870899, 0.0356945992, -0.0985943973, 0.123549551, -0.000760247931, -0.0291051362, 0.0804991275, -0.0239255689, -0.0181377307, -0.0692903325, -0.0611725226, -0.0522443131, -0.134671256, 0.18177627, -0.110332564, -0.144453228, -0.106152989, -0.0792289972, -0.052244164, 0.00281627057, 0.0507592373, 0.0200824514, -0.0920186713, -0.142175823, 0.0308848098, -0.0685959309, -0.0735030398, -0.0047179726, 0.0742548928, 0.0716363564, -0.051056657, -0.000936691533, -0.0247088131, 0.0673220307, -0.103734247, 0.113195941, -0.0123151951, -0.0716323107, 0.0879234299, -0.0706144571, 0.0800992474, -0.116462201, 0.0710284188, -0.0274224319, 0.0911740512, -0.0591697395, 0.128571212, 0.00942194462, 0.0112342853, 0.0594393238, 0.122481525, 0.0518759452, 0.00391112827, 0.00459925085, -0.00107023492, -0.0406995639, 0.0181504153, 0.0787359923, 0.0413333066, -0.0773825496, 0.134060547, 0.105162509, 0.100520976, -0.0857238472, -0.0685628951, 0.0463460349, -0.128627837, -0.0599386021, 0.109882325, -0.00504093058, -0.0323709436, 0.0150102321, 0.039100565, 0.00190809369, 0.033697173, 0.00305089541, 0.00202031806, -0.146391481, 0.0123923076, -0.0165218934, 0.0793899894, 0.0192385539, -0.0389196128, -0.0517317243, 0.0559310243, -0.0768021494, 0.0226306207, 0.121306881, -0.0522455648, 0.00339139812, -0.0556291714, -0.0995496213, -0.0963014066, -0.0816042349, -0.11229635, 0.0557814501, -0.0740598366, -0.0173649304, 0.139369071, -0.0306224898, -0.0580060631, -0.091436848, -0.1747071, 0.118114039, 0.02228209, -0.0473897681, 0.0664613992, 0.0720168129, 0.0845688134, 0.0528362468, 0.000815280247, -0.102460355, 0.0476971269, -0.0671160519, 0.0525707528, -0.0415160656, -0.102914102, 0.0113827325, -0.083965674, -0.0490029082, -0.0314759016, -0.0968770608, -0.0548568815, -0.104666732, -0.0537175536, -0.0062415353, 0.10947898, -0.0233759973, -0.117974564, -0.0366625525, 0.0608506501, 0.0428013578, -0.0998068377, -0.118065089, -0.0119977761, 0.124744356, 0.0283070784, -0.0802738294, 0.0655657947, -0.0954824314, 0.0362423845, 0.0332849324, -0.0834430009, 0.0715879798, 0.0472209863, -0.0373611376, -0.0470067151, -0.0612793155, 0.0413198546, 0.0846912786, -0.0206781477, 0.148907751, 0.0997918695, -0.0374904834, 0.0923477262, -0.164048508, 0.0363637581, 0.12508589, 0.0251565874, 0.0373173356, -0.0349174105, -0.0210640188, -0.0291269049, 0.0575178042, -0.0673399717, -0.111204684, 0.000690751011, -0.0608374774, 0.0883233175, 0.0703906566, 0.00799492467, -0.0885908753, 0.0663681254, 0.00513501652, -0.0683957562, -0.0635244995, 0.0509348921, -0.045457378, 0.067822583, -0.0514202528, 0.0347993821, -0.105504952, 0.0464331098, -0.0200170074, 0.124304675, 0.00249845907, -0.139286578, 0.0419195741, 0.138129503, -0.137769043, -0.0693240017, -0.144727841, -0.0269639567, -0.0316476636, -0.00926445797, 0.0155554442, 0.0988779292, 0.0360196903, -0.11852254, -0.146118566, -0.141063496, 0.0180321112, 0.044023633, 0.0607468039, 0.0902918354, -0.0553643666, -0.0225360487, -0.0291328467, 0.120564714, 0.00701142848, 0.0940650702, 0.0386316068, -0.066673629, 0.0376338474, 0.0764669105, -0.0897704884, -0.0251525287, -0.00749431085, -0.0358690172, 0.0398492031, 0.0265903752, -0.0361888818, 0.125865638, 0.054716222, 0.0339330956, -0.0974758416, -0.0556336716, 0.0554950386, 0.0709042475, -0.0551284701, -0.150779456, 0.0356293619, -0.0151905287, -0.0415148139, 0.0461233035, -0.0375088528, 0.0776319429, 0.078568168, 0.0219056439, -0.0641739443, 0.0184024908, -0.0559999272, 0.00853113644, -0.0582099259, 0.0130015435, -0.000109020621, 0.0413256809, -0.0175708272, 0.00443046819, 0.0459968075, -0.0424706116, 0.00485516898, -0.139668763, -0.107954606, -0.033286605, 0.000858554617, 0.0112799844, 0.0316995755, -0.00445954315, 0.0098643275, 0.00362277031, -0.176973119, 0.0289542675, 0.0964407027, 0.0178754423, -0.0725989938, 0.0330223516, -0.0307930931, -0.136516929, -0.0208547302, 0.0932566077, -0.0433047451, 0.127082095, 0.0337875597, -0.0496471711, 0.0266216137, -0.0302028675, -0.0671077296, -0.069399491, -0.194116816, 0.107985169, 0.119947314, 0.116231322, -0.00947291963, -0.0721068382, -0.119167857, 0.0993771553, 0.0410175882, 0.0651499629, 0.113678746, -0.0722037777, 0.0489135459, -0.0615688562, 0.00746499747, -0.0885654688, 0.00774631463, -0.00619787909, 0.0144832283, -0.00118065253, -0.0396787487, -0.000157682225, -0.138799325, -0.094255127, 0.135156259, 0.0337659083, 0.0495264307, -0.00455174129, -0.098026149, 0.13226442, -0.00644892734, -0.0126878396, -0.119426385, 0.106981225, 0.0939402208, 0.0869578496, 0.0459269434, -0.0357407071, 0.0646807551, 0.067193076, -0.0493923053, 0.0898668766, 0.0236707926, 0.00805385411, -0.079227671, -0.087250486, 0.00157636264, -0.091030851, -0.0203078557, 0.0409940705, 0.0134612247, -0.0116334986, 0.0569527075, 0.0660834983, -0.13612771, -0.0281860009, -0.0982794464, -0.0445884764, 0.0251589492, 0.0647347793, 0.0288546849, 0.0464992821, 0.0603758171, -0.0300618839, 0.0956698805, -0.129332364, 0.0559479222];
    bias_0_r : ARRAY[0..63] OF REAL := [-0.173484892, -0.0675045773, 0.0491046086, 0.0463505276, -0.0815096349, -0.110554256, -0.0473120436, 0.437425762, -0.00653401855, 0.176917329, 0.370717168, 0.0396423079, -1.08117795, -0.0953554064, 0.150914401, 0.0577960424, -0.0104229543, 0.249676898, 0.0947834998, 0.126156241, 0.072207287, 0.261239588, -0.102599576, -0.646232307, 0.596568823, 0.280415773, -0.238218173, -0.300266802, -0.174425423, 0.181508452, -0.275678068, 0.177939966, 0.170858145, 0.144983739, 0.305772722, 0.21602802, -0.058799278, 0.16263026, 0.152120188, 0.226213232, -0.139869258, -0.26692462, -8.2628685e-06, 0.244418189, -0.0422431342, 0.486167401, 0.180008084, 0.371829987, 0.247329235, -0.39782384, -0.508523405, 0.0987078175, -0.00799489487, -0.575995445, -0.137379125, 0.00688174972, 0.359871328, -0.0202121828, 0.147642806, 0.0532373562, 0.141280323, -0.153836474, 0.204907924, -0.00387164229];
    weights_0_h : ARRAY[0..63] OF REAL := [0.511881709, 0.529895723, -0.477809012, -0.506132901, 0.537910998, -0.527767479, 0.491260558, -0.324178755, -0.548811018, 0.494253427, 0.363518178, -0.522180617, 0.508872926, -0.535762608, -0.393660396, 0.486902118, -0.543106973, 0.495763212, 0.534182966, -0.454969078, 0.549818516, 0.410422921, -0.523729563, 0.518692791, -0.241631955, 0.380803972, -0.511416197, 0.452509254, 0.450534821, 0.378833294, -0.505145967, -0.454468369, -0.521197736, -0.407331824, -0.358680755, -0.488305509, 0.447431266, 0.542436302, -0.509502351, -0.401503712, -0.546306491, -0.521000624, 0.419856697, -0.42881614, -0.506078959, 0.265747756, 0.523313284, 0.384962797, -0.367372096, -0.544435382, -0.486974597, 0.513249099, 0.413192004, -0.513616383, 0.459577471, -0.420617849, -0.35950458, 0.482437223, -0.450004786, 0.459671527, 0.469759375, 0.540518165, -0.404790819, 0.54321909];
    recurrent_0_h : ARRAY[0..4095] OF REAL := [0.0151014654, 0.0315691419, -0.00384554872, -0.105252482, 0.0954181105, -0.0486003868, 0.0757943094, -0.0748094544, 0.103059046, 0.0163525231, -0.0429565907, -0.0707249939, -0.123956338, -0.0394361317, -0.146633834, -0.103257373, 0.0837373883, 0.0299536027, 0.0506832749, -0.0691065937, -0.0754909143, -0.0278890803, -0.156872854, -0.0413584113, -0.137698248, 0.0687828958, 0.0563442335, 0.018389143, 0.0312211905, -0.0644816086, -0.0680799186, 0.102891371, -0.121650897, -0.0529458225, 0.092071712, -0.00170892943, -0.0130693149, 0.12133313, -0.124405108, 0.15404433, 0.0598416552, 0.0570201501, -0.0286285356, -0.0331414379, 0.0462406948, 0.0842860341, -0.0477161668, 0.0449983403, -0.0474944636, -0.0678177997, -0.0183854587, -0.0297140516, 0.106223077, -0.00322339637, -0.0999261439, -0.0824365318, 0.0240056701, 0.0590381622, -0.0936049968, 0.0295491889, 0.107780747, 0.080072917, 0.0176341012, -0.17420283, 0.0588149242, -0.0870779753, -0.134306341, -0.0692487508, -0.157706246, -0.0270572938, 0.0707601011, 0.149820372, 0.110426478, -0.00743779354, -0.0465169512, 0.0691735372, 0.111401349, -0.0139408177, 0.0205599926, -0.0962041765, 0.0503444895, 0.0740744546, -0.0419505239, 0.0196950305, -0.0837824196, 0.0464542881, -0.0288814493, -0.0535249971, 0.0254174136, -0.0666553527, 0.0397340655, -0.0178836547, 0.0203624424, -0.0447266363, -0.0661628321, 0.0150283603, -0.122055553, 0.0711871386, 0.0188331716, -0.109750815, -0.0493549854, -0.0550094284, -0.00762387738, -0.0353097506, 0.135499761, -0.015370369, 0.0184302274, -0.0249744803, 0.2203383, -0.0442610495, 0.0065962784, 0.0633476973, 0.0377533771, -0.0880632102, -0.0339279845, -0.0212823916, -0.0435293168, 0.0181129221, -0.0127849532, 0.110028744, 0.0964113325, -0.0344761126, -0.0126675069, 0.00523473881, -0.108181819, 0.129458338, -0.154461205, -0.0144926272, -0.0874574408, -0.0518219285, 0.0588002875, 0.014298114, 0.0187594295, -0.0174597241, 0.199162781, 0.134521887, -0.0472685322, -0.0397187695, -0.0142858475, 0.0857593864, -0.0718451291, -0.0385252982, -0.0189274848, -0.0534091666, -0.00660294015, -0.0306221731, 0.0354711525, -0.0566619001, -0.0506171137, 0.0256853756, -0.0265512876, -0.0473412536, -0.0894344822, -0.116834685, -0.0509595014, 0.0759056807, 0.0700788572, 0.00462372554, 0.089258492, -0.0152192153, 0.0457421429, -0.0269401558, -0.0140602961, 0.106877066, 0.123079993, -0.0989074409, 0.0320937112, 0.0529134832, -0.00390504859, 0.0247814283, 0.0754490569, -0.121886, 0.145266309, -0.121950209, -0.0752653405, -0.0901928097, 0.00366103277, 0.0372722931, 0.0210407581, -0.0174527131, -0.0353134423, -0.00717110001, -0.0354144573, 0.0215394534, 0.0330921113, 0.0686442032, -0.0344005786, 0.0645818338, -0.0111237355, 0.0727535784, 0.0465916693, -0.0652130917, 0.106176965, 0.0119006718, -0.0605614632, 0.0079497043, 0.0370872803, 0.00775675802, 0.0357049927, -0.126892924, -0.0222051032, 0.0738216713, 0.0740928352, 0.0294515938, 0.0681039169, -0.0378874578, 0.0758690089, 0.0175420642, -0.0628558099, -0.0672130585, 0.0307014622, -0.0804512277, 0.176019937, 0.132123068, -0.0889720023, -0.0831062198, -0.135356486, -0.143481523, -0.0899433345, -0.0380111784, -0.0449125469, -0.0193431079, -0.0362437889, -0.0266001876, -0.0325177684, 0.0157292224, 0.0499577671, 0.0174572486, 0.0536411963, 0.121578008, -0.0687552541, 0.0890867636, 0.0383188464, 0.0148758721, -0.0303913709, -0.00649094395, 0.0854870602, -0.102338418, -0.0666316673, -0.0281381235, 0.0549249165, 0.0424676798, 0.0872980133, -0.0456232056, 0.022293983, -0.148441434, 0.0569621846, -0.0632671192, -0.0296576694, 0.118491352, 0.0409092493, -0.054831367, -0.105856366, 0.0819140747, -0.128674701, 0.0155766308, -0.00430044997, 0.0650782585, -0.08370094, 0.0713149831, 0.0574905761, 0.0671258867, -0.0950446203, -0.0663676858, 0.0711896271, 0.00114663318, -0.00647407491, -0.119475968, 0.160537824, 0.0439400226, -0.0349544063, -0.012381129, 0.0524228588, 0.138963565, -0.100225538, 0.00670948718, -8.71550292e-05, 0.160157681, 0.0178130865, 0.02238499, 0.0803312287, -0.00828377903, 0.00724661164, 0.0321915038, 0.0242249686, 0.0313558206, 0.00169815496, -0.042619694, -0.0616292879, -0.0522229746, -0.0935247093, 0.153820843, 0.0857300758, -0.172498316, -0.021524474, -0.0319245197, 0.0929623768, 0.0532867275, 0.0314655602, -0.0274347682, -0.0879180729, 0.0986205786, -0.0337646529, 0.0416346788, 0.0332635641, 0.0381301343, 0.079621613, 0.0737273619, -0.0366122052, 0.119512878, 0.0474161692, -0.211196274, 0.0176645368, 0.0787715167, 0.0302956551, 0.0390346721, 0.00925036147, -0.0182805713, -0.041102685, -0.0138021689, -0.0270654373, 0.0491370782, -0.0514427237, -0.0751671568, 0.0477790311, 0.0277377404, -0.0619665608, 0.0156615973, 0.00482634781, -0.00682761334, 0.00939017069, 0.067990765, 0.137770802, 0.0574506521, 0.0701330528, -0.0982482061, -0.0862303302, 0.0904136226, 0.0466973111, -0.0325784385, -0.000851515681, 0.0318356156, 0.0433966741, 0.00800497457, -0.00970953703, -0.0271797776, 0.0797721297, -0.118577689, 0.0206320807, 0.017929947, 0.0955219716, 0.17246969, -0.0278012976, 0.0755585432, 0.079024449, -0.0478332341, -0.06807217, 0.0914565176, 0.20822309, 0.0121487696, 0.0471593961, 0.0288373716, -0.00932216831, -0.149716005, -0.0538578369, 0.0268720426, -0.0361705907, 0.117366888, 0.0253876261, -0.0262836274, 0.0496964678, -0.0192397106, -0.0702153593, -0.0391614847, -0.161675587, -0.136856928, 0.0672038645, -0.0700094998, -0.00911142305, 0.038635321, 0.0767850429, -0.0122583732, 0.183748305, 0.0132101532, 0.0678323731, -0.211896747, 0.0235066377, 0.0453544036, -0.0898434073, 0.103501424, -0.0940179378, -0.016603183, -0.00502588693, 3.42298299e-05, -0.013213018, 0.0565248802, -0.0319322944, 0.0672975481, -0.0400523022, -0.134900898, -0.0601539873, 0.0332695991, -0.0905719399, 0.0467153937, -0.0810768381, 0.127729416, -0.0900901854, 0.0902750939, 0.0299907867, 0.0586670302, 0.0495708399, 0.1158012, 0.0336007997, 0.00532219745, 0.123860262, -0.0363541022, 0.0275619552, -0.00662331656, 0.109502621, 0.0298098996, -0.00811201707, 0.0412303284, -0.0805860385, -0.0472148471, 0.102457054, 0.0257757008, 0.0102556758, -0.0890942737, -0.0421103425, 0.0365854949, -0.0659021437, 0.111958601, 0.0964360982, -0.046282202, -0.0126719587, -0.0458573662, 0.116932459, -0.0212433711, -0.0881072953, -0.00770005584, -0.0857032984, 0.0025970079, 0.0132948514, 0.0339403749, -0.0626496002, -0.0146684814, 0.0161503572, 0.000780121423, -0.032719072, 0.0686777085, 0.0906086937, -0.0502825528, 0.0462821573, -0.180640206, 0.00406896137, -0.0251903422, -0.11153277, -0.0614060163, 0.0169649497, -0.00545855705, 0.0387234055, 0.061546132, -0.0173524842, -0.0139072761, 0.0299902521, 0.00907874666, -0.00572424382, -0.0507996082, -0.0923170522, 0.0297425594, 0.0514120758, -0.0830440968, 0.0198585112, 0.0656371266, -0.0585631095, 0.0178769249, -0.0531284511, -0.0271281898, -0.140999585, -0.0196059793, 0.119963646, 0.111532696, -0.103885248, -0.100702703, -0.010400556, 0.0219070762, -0.0126086501, 0.0240438357, -0.060223829, 0.0423679128, -0.00986079872, 0.0329693109, -0.0818725005, -0.0714677423, -0.0257736444, 0.0543711409, 0.0940362662, -0.119938776, -0.0633669943, -0.116895951, -0.0374297909, 0.0153847542, 0.0372343957, -0.0610368811, 0.113813013, -0.0170616098, 0.00195942726, 0.00671724509, -0.0389183983, -0.0128870467, -0.113415472, -0.0129363602, -0.0356861092, 0.0534268841, -0.0288733747, 0.0418036468, -0.153400227, 0.0296305232, 0.0245947726, 0.066393964, -0.00165655045, -0.122910373, 0.0488593057, 0.0413906798, -0.0627416894, 0.0645338818, -0.026778372, -0.0406190902, -0.0442537032, -0.00246794894, 0.0225111302, -0.00398455374, -0.0284111463, 0.124458574, 0.130251542, 0.113397017, -0.0720993355, -0.0414232314, 0.0428066999, 0.0329683721, -0.0125187151, 0.115253933, -0.0684984401, 0.0104852254, -0.136497185, 0.00998436473, 0.0500208177, -0.0262930356, 0.0352597348, 0.0552926809, -0.134685189, 0.100826129, 0.0628324151, 0.0390063636, 0.010178389, 0.0558182113, -0.00302903913, -0.0310565364, 0.0949583054, -0.153061911, 0.0321237296, -0.051590357, 0.0456893779, -0.023379581, 0.0882194489, -0.0808342993, 0.093459636, 0.00758528709, -0.106659807, 0.00587938726, -0.0590616018, -0.0399960913, 0.00719778053, 0.108343609, 0.0468838401, 0.0391731933, -0.016234532, 0.0277812388, -0.0368827656, 0.00372426142, 0.0314919986, -0.0181080867, 0.0381364822, 0.112079777, 0.157007411, -0.0116896331, -0.0103837289, -0.155438438, 0.030527778, -0.114068605, 0.108232319, -0.0308927819, 0.117109597, 0.00867082179, -0.0103414804, -0.0227078237, -0.0242070407, 0.0158710014, 0.0176119618, -0.0023907884, 0.02301763, -0.172001734, -0.0185527913, 0.066018872, -0.00374495611, 0.00550355855, 0.0396729745, 0.0719289333, 0.0583389513, 0.228415847, 0.0289598331, 0.0523797348, -0.0487385169, -0.038304951, -0.0288884249, -0.0958547294, 0.0831411406, 0.00722385664, -0.0514185987, 0.0281225797, -0.0335371867, -0.0953213423, 0.0357710347, -0.00273016654, -0.0733452439, 0.0190322548, 0.0579749383, -0.0754311532, 0.0323413908, 0.130112335, 0.0591265336, 0.0263809413, -0.0889221877, 0.0362376422, 0.00274141366, 0.0602396727, -0.00956112519, -0.0633085221, -0.0705631971, -0.00269171223, -0.0227907635, -0.0692018792, 0.0450100601, -8.21100548e-05, 0.085006319, -0.0117384307, -0.178841949, 0.00916172564, -0.0331595391, 0.0488371365, 0.0309088267, -0.0520205721, 0.0543855466, -0.0609956905, -0.0151451491, -0.119706556, 0.0521327071, -0.0239361376, 0.0619983524, -0.0344233587, 0.0928516462, 0.123764999, -0.0510081723, 0.051918298, 0.134016812, 0.00433373079, -0.0399642885, -0.0476095639, 0.058590617, 0.0102138538, 0.0473462418, 0.0685652196, -0.00715079717, 0.0423923582, -0.123237118, -0.0599423945, -0.0193803404, 0.0810124949, 0.0482463613, 0.010171093, 0.0322510414, -0.0855225101, -0.0134441592, 0.0353776589, 0.0357695967, 0.0157995224, 0.00592060806, 0.0427856967, 0.019695485, -0.120965153, 0.0518125519, -0.025982812, 0.00440140441, -0.101803318, -0.00751397945, -0.0489026457, -0.110446945, 0.0387411118, -0.0329769477, -0.026433032, -0.0734259188, -0.0359849557, 0.0301200077, 0.0163871422, 0.00114649849, -0.10535416, 0.0533666052, 0.0522046946, -0.00681710057, -0.0213999078, -0.0203455649, -0.063229993, 0.0781266317, 0.0768756866, -0.0961050317, -0.065041244, -0.133748487, 0.0100543723, -0.0106222974, -0.0259819292, -0.0329633467, 0.0461320877, -0.0447794944, 0.003435269, 0.0207778122, 0.065288499, -0.028659109, 0.0149778146, 0.0349693224, 0.0478700735, 0.014303416, -0.0856329799, 0.10475678, 0.0338214226, -0.154605776, 0.00877577253, -0.132177755, -0.0806690902, -0.00436068373, -0.0136294104, -0.0454847552, -0.108277924, -0.0509702489, -0.10566017, 0.0186794251, 0.0360619947, 0.0443202034, 0.0150199682, 0.197757751, -0.0792406127, 0.126476422, -0.0556568801, -0.0213381834, 0.140827551, 0.0756311268, 0.0323015526, -0.0986557081, -0.0878089145, 0.0130598582, 0.0204975531, 0.0466922373, -0.0937384889, 0.0174807832, 0.0393661335, -0.0838654786, 0.014209413, 0.0197430924, 0.0545310043, 0.0844336376, -0.00396912917, 0.093169868, -0.159154788, 0.0605714992, -0.00325722061, -0.0306225698, -0.0325894691, 0.0413154587, 0.0223213788, 0.0820711106, 0.0751379952, -0.087409243, 0.0902555585, -0.0316079296, 0.00693639787, -0.0477129482, 0.0698177144, 0.0563609712, 0.150307685, -0.0405079909, 0.0418194234, 0.00745331962, -0.044603765, -0.0868503079, 0.0228795428, 0.0951327384, 0.145075753, -0.00281672552, 0.0819790065, 0.100366093, 0.120265633, -0.12336693, 0.097921811, -0.0526711382, 0.0146113727, 0.0517357066, -0.00685218349, -0.0323748961, -0.0437289886, -0.00333631411, -0.0126014203, -0.0984798595, -0.114890754, 0.0288062505, -0.0771140903, 0.0382514372, -0.0117044989, 0.126339108, -0.00630878564, 0.0530857854, -0.104100645, -0.00805898756, -0.0305066146, 0.105314784, 0.048034966, -0.00172337517, 0.0301087871, 0.165835604, 0.0267596543, -0.142763242, 0.181588918, 0.0551236197, 0.0679461434, 0.101056561, 0.0339270458, -0.073371917, 0.0601740666, -0.0367997475, 0.0108242445, 0.0693133548, -0.0234897546, 0.102104969, -0.0528279245, -0.0597027726, -0.0566084348, 0.0335544311, -0.205662742, -0.0541634336, 0.00158093637, 0.0658201575, 0.0301372595, 0.0693942308, 0.107268907, 0.0292246621, 0.128294975, 0.0263936706, 0.0309509225, -0.0775180459, 0.116698608, -0.0734690353, -0.0131640136, -0.0256189536, -0.062963888, -0.126585558, 0.0140708741, -0.0230707563, 0.109207697, 0.11241141, 0.0451781824, -0.0347523019, 0.0550954714, 0.0766290501, -0.0519221164, 0.0437252149, 0.102785774, -0.105436176, 0.10736078, 0.0210221633, -0.0217525065, 0.100014761, 0.0385276638, 0.0546158366, 0.0585203208, -0.0420682579, -0.171221569, -0.142569944, 0.0215001479, -0.023452919, 0.0635518059, 0.0205523521, -0.0221534446, -0.09596131, -0.0570831373, -0.0364792533, -0.117802076, 0.0533068553, 0.0692519322, 0.0763008073, -0.0444405191, -0.141365409, -0.0190920215, -0.0462770239, -0.116279766, -0.0336749479, 0.0318626389, 0.0286726728, -0.0309933089, 0.00509904884, -0.117549956, -0.0551077612, 0.00944215711, -0.0124984551, -0.0347758941, -0.0253979862, -0.0476573743, -0.0240106434, 0.0761979371, -0.00755198859, 0.000757890753, 0.0146143194, -0.0430316068, -0.105958819, -0.0228075683, -0.0752149299, -0.0152789466, 0.0252250638, 0.00773550943, 0.147780925, -0.0151827568, 0.0613514408, -0.0986682922, -0.0442262664, -0.0455808938, 0.0428584889, -0.0703783184, 0.0335962176, 0.022636719, 0.000310000032, -0.0391520672, -0.0628906041, -0.0938398689, -0.0734697208, -0.0291133802, 0.179060459, -0.0784291476, 0.0768223926, -0.0370093696, -0.0368609205, -0.0792517066, 0.0696835145, 0.0456825048, 0.0358340479, 0.0434729829, -0.0668236166, -0.0652068704, -0.183176398, -0.0633447096, 0.0550470129, 0.0324314684, -0.131186828, 0.00050502643, 0.0845886469, 0.0555002876, -0.0492061079, -0.201960742, -0.0906325206, -0.0749930367, 0.050311245, -0.0290989503, -0.0318274796, 0.0245478377, 0.0217907615, 0.0250097271, -0.0652556121, -0.0649409145, 0.0265176073, 0.0243124366, -0.0689618066, -0.107658178, -0.0692645833, -0.054567121, -0.0179806706, 0.0172811598, -0.13332127, 0.0765545368, -0.0310513452, -0.0622933619, 0.0652891845, -0.0139535349, -0.00840768591, -0.0719554275, -0.103346743, -0.205132723, 0.047608614, -0.00250128657, -0.000518750399, 0.0459744036, -0.108746588, -0.0344416574, -0.09308438, 0.0268362872, 0.0715449229, -0.059631139, -0.0216482393, -0.0235823784, -0.0962414742, 0.0395797528, 0.0250034407, 0.0147794839, 0.016083248, 0.0418951213, -0.0584590547, 0.0527435131, 0.0311591234, 0.130391851, 0.150298372, -0.0433518961, 0.0115818251, -0.103978656, -0.00348509476, -0.0824357718, -0.071391426, 0.00255766511, 0.0320981182, -0.22617498, -0.0560468659, -0.0822790861, -0.219181985, 0.00953684561, -0.0300233066, 0.111459889, 0.0274805464, -0.140019536, 0.0153040197, 0.0539604127, -0.0157690719, 0.0947029889, -0.070151329, 0.00172157213, 0.0609328263, -0.0234152079, 0.0360128805, -0.114299558, -0.0119139217, -0.0178148597, -0.0278276093, -0.0883894339, 0.064821586, -0.15142858, 0.0802713782, 0.0321872979, -0.0716421828, -0.122801922, -0.0259564184, 0.123508014, 0.0335269272, 0.0583531, 0.043163009, -0.0497357398, -0.0202746131, 0.0915562809, -0.0884398818, 0.00746741146, 0.0121395029, 0.0458049811, 0.0897039324, -0.0835799426, 0.00104040024, 0.0218561664, -0.0829297453, 0.0716589317, 0.00597879291, 0.00369991735, 0.0972465575, 0.0318837091, 0.0861498266, -0.125971302, -0.0046215672, 0.039220728, -0.0331700929, -0.0022045821, 0.0141417515, 0.00824223831, 0.100044392, -0.0323052891, -0.00785260275, 0.0707256421, 0.0591015667, -0.00800828263, -0.0836099014, 0.0224461854, -0.00758463563, -0.0430032499, -0.0993371308, 0.0381070673, -0.0292616654, -0.0305680539, -0.0527784973, 0.0147669194, -0.0452954806, 0.00313056516, -0.0710692182, 0.0366714299, 0.154665232, -0.132521346, -0.115051359, 0.0153902564, -0.0508783571, 0.0555030368, -0.0203189589, 0.0208809953, 0.0317924544, 0.0976715684, -0.163995042, -0.0313210711, 0.0696517229, -0.0985373706, 0.0176254176, -0.0817904994, -0.111890033, 0.0534250289, 0.0213724207, 0.0842697173, -0.0279486086, -0.00327455997, -0.0896307826, -0.00842390582, -0.0768062845, -0.106076509, -0.074272871, 0.0391257666, 0.0854253918, 0.0249287318, 0.00916362368, 0.0300335549, -0.0668060482, -0.100941926, -0.075986661, -0.00613939017, 0.0470039733, -0.0999038219, -0.0575053319, 0.019524131, 0.0361823663, 0.131882608, -0.0096709393, 0.0882648826, 0.041786477, 0.034654133, 0.0255509745, -0.0886439085, 0.00837724656, -0.0773778856, 0.0229398739, 0.0581588559, -0.0465174727, 0.0858686119, -0.0553110354, -0.0148559269, -0.0410864353, -0.00901198946, -0.00128553924, -0.0114130266, 0.0124721397, 0.0549827255, -0.007832665, -0.0482536331, -0.0951088592, -0.0759178251, 0.0608368292, -0.0407103449, -0.0283425767, 0.0321998298, 0.126301706, 0.067398712, 0.139780685, 0.0905814394, 0.00255679712, -0.00767655671, -0.00840915833, 0.088301219, -0.048137214, 0.0148405693, 0.00380565645, 0.0106215859, 0.089731425, 0.034143839, -0.0650838614, -0.0764127225, 0.13296175, -0.177675739, -0.0525807329, -0.104725361, 0.064101845, 0.10076917, -0.0463725515, -0.0662362948, -0.0379772894, -0.074941963, -0.141431734, 0.000464164652, 0.0287206192, -0.0947588235, -0.0683050156, -0.0300985053, 0.0466467403, 0.104172662, -0.134927958, 0.0471047983, -0.0949884206, -0.0951971039, 0.0283831507, 0.0657143593, 0.0462317839, 0.0435468554, 0.0596275926, -0.0388186611, -0.0583273657, -0.0233254395, 0.0902210325, -0.0985154659, -0.0384789072, 0.0537803955, 0.104289338, -0.0677582994, 0.0276348703, 0.0171381459, -0.0307430662, -0.0552040786, -0.0401273668, 0.00251147803, -0.0259028301, -0.128685653, 0.0270089079, -0.0281825364, 0.0558626354, -0.0426816903, -0.0650866926, 0.0326622389, -0.0483125076, -0.055412095, -0.0244423784, 0.0109835584, 0.0196121559, 0.0430874974, 0.0266159214, 0.00617672317, -0.107649848, 0.0332261026, 0.123890027, 0.067306675, -0.0808168426, 0.101745799, -0.0675554276, -0.0669053793, 0.0962668732, -0.104982689, 0.0697224736, 0.0392863825, 0.0293577798, 0.0433183499, 0.0401539989, -0.0264592841, -0.124858037, -0.0245554093, -0.071433872, 0.0490507632, -0.0315658227, 0.0505969934, 0.040864408, -0.000168052502, -0.0109752379, 0.0373206735, -0.145048499, -0.0239026174, -0.0684744939, -0.0636875778, -0.0114831738, 0.139179409, -0.00155177619, -0.15342024, -0.033083193, 0.000420395285, -0.117142901, 0.00887246989, 0.122661121, 0.113508984, 0.0204033777, 0.00637237635, 0.0819063187, 0.00776152499, -0.106520936, 0.0975836441, 0.0585022047, 0.0782554224, 0.046391435, -0.022785807, -0.0304160044, -0.0622793511, -0.0942288488, -0.0606903024, -0.00904364698, 0.0629969984, 0.0954230279, -0.12778683, -0.0284533855, -0.0272438936, 0.0757961869, 0.028047964, 0.0972610638, 0.0580233596, -0.0828812718, 0.119468622, 0.0710946023, 0.0221559331, -0.0590557754, -0.0555966273, -0.0606284887, -0.0115851667, -0.0940932408, 0.0262915269, 0.0135664009, -0.00717134774, -0.0664277151, -0.0882107168, 0.0916490331, 0.0246482864, 0.103041373, -0.123946175, -0.0915629715, 0.00223686872, -0.073600322, -0.0802451596, 0.108621851, 0.0714537129, 0.0417542085, 0.134732231, 0.0369990319, -0.082304731, 0.052722007, -0.0231204405, -0.00113231316, -0.0775985718, -0.0870465413, -0.0127883479, 0.0597468019, 0.0681404546, -0.0372708365, -0.00268130354, 0.0848922282, -0.0623495802, -0.00645769248, -0.117754631, 0.0372559428, -0.0158301927, 0.0494583473, -0.0121700251, 0.0199690834, -0.0330053344, 0.0689561367, -0.0206274483, -0.0206134468, 0.0432984717, -0.0370494798, -0.0341483019, 0.0488845222, -0.0686890259, 0.179095566, 0.0062625967, -0.0568772294, -0.091103442, 0.0186275057, 0.0290343128, 0.115588844, -0.0852092206, 0.0256224014, 0.0983831733, -0.00113785639, 1.40275806e-05, 0.0457989648, 0.0426610336, 0.152750835, -0.0321622267, 0.138436332, 0.0073488988, 0.0764992163, -0.0264629424, -0.0250669904, -0.00355184451, -0.0162453055, 0.0607386976, -0.125566661, -0.0264021866, -0.0892097577, 0.0325158015, -0.0342464149, -0.108295441, 0.0783299357, -0.0384992883, -0.045980528, -0.0264427215, -0.0641009584, 0.0916307718, -0.160485119, 0.101107836, -0.124456659, -0.0714205652, -0.0165864844, -0.0105503872, -0.0963487178, -0.00333322771, 0.0448205657, -0.0510514453, -0.0136782899, -0.096345827, 0.0154198436, 0.0299618877, -0.0672173873, -0.102037974, 0.0483165756, -0.0276720915, 0.130227983, 0.0581221469, -0.072762236, 0.047728993, -0.0352324732, -0.0594642349, -0.002675422, 0.139455602, 0.00566758122, -0.0134287253, -0.0688176528, 0.0625232831, 0.140319631, 0.0563304573, 0.0567270331, 0.0983596072, 0.150661379, -0.0800207555, -0.0853598565, 0.0336976275, 0.0131315533, -0.0819277465, 0.057536494, 0.00667545758, -0.0457928032, -0.038779866, -0.00723124668, 0.00690400228, 0.0680176616, -0.0253968798, -0.172183186, -0.0330998711, 0.0270697325, 0.0356532708, -0.0886402205, 0.0234502219, -0.0174542684, 0.0187187009, 0.00804674998, -0.0369820781, 0.00467156246, -0.0236953069, 0.104239531, -0.0260523707, -0.0250848345, 0.0440467596, -0.0172335394, 0.0141086634, 0.114409156, -0.0390056148, -0.143985286, -0.0538066439, 0.066485323, 0.0168812945, -0.0859410539, -0.00942959171, -0.0697698146, 0.15309763, -0.143645525, -0.191575617, -0.0842180029, 0.0131736286, -0.0419890843, -0.0355420783, 0.0517604202, 0.0332058445, -0.0892739147, 0.107086726, -0.047652822, 0.0188595317, 0.131176427, 0.0565858409, -0.021854572, -0.110475987, 0.0490295179, 0.118606359, 0.0701356754, -0.0754051432, 0.014309682, -0.00493702851, 0.00770587474, -0.00327124819, -0.00881879777, -0.0423447676, 0.010203043, 0.0713135451, -0.148224965, 0.00333502889, -0.0559453182, 0.0410412326, 0.0759655833, 0.0172477216, 0.0831833854, -0.0297368802, 0.111099362, 0.0883169025, -0.0722597763, 0.0131261591, 0.0140464399, 0.0175292101, -0.0339123756, -0.0285929143, 0.108016133, -0.0652214736, 0.0378189981, -0.05128555, 0.124187529, -0.0402831659, 0.0293531604, 0.00742054172, 0.00414653495, 0.0328657441, 0.00383558497, 0.0537207313, -0.0284183696, -0.0582612269, 0.0320823602, -0.0386008807, 0.0356729515, -0.0504770167, 0.0652536973, -0.098795183, 0.120945551, -0.0412323773, -0.113359623, -0.168529689, -0.044518292, 0.0557504669, 0.0932161137, 0.0808147937, 0.0658239126, 0.061269097, -0.0194292106, -0.0816457719, -0.122028135, 0.161170825, -0.0266123172, 0.000504847616, -0.10841462, 0.0521031097, -0.0749769509, 0.146326363, 0.085672766, 0.0806948692, -0.0364968404, 0.051602222, 0.00282965973, 0.015352767, -0.0605669692, -0.0158483312, 0.0319661647, 0.0238912627, 0.0661585629, 0.0638670698, 0.115828492, -0.15485394, -0.0117736533, 0.108005427, -0.0221562441, -0.0248847492, -0.00074852258, 0.0295029134, 0.0192475319, 0.0617187917, -0.0633570254, -0.0326333679, 0.109099194, -0.0391615331, 0.0408077464, 0.104218476, 0.0296367407, 0.141252548, -0.0425838605, 0.0149380863, -0.0466234013, 0.00988053158, 0.0613031909, -0.0232185572, -0.0452623069, 0.0944167376, -0.0354872383, -0.0408066846, -0.0227842871, 0.0703361928, 0.139385894, -0.095162794, -0.0230612122, -0.00723451842, 0.0986850411, -0.119977117, -0.00739560928, 0.112956479, 0.15224497, 0.0479522869, -0.0886996239, 0.105766222, -0.141112834, 0.028072454, 0.0646339506, -0.0836297721, 0.00408888934, 0.0167465769, -0.046307411, 0.0784704909, 0.103682615, -0.058488939, -0.0245305765, -0.180317387, 0.0136912018, -0.0455013961, 0.0150855631, 0.0137447789, -0.0616712347, -0.0202290341, -0.0954892188, -0.080296129, 0.0467284843, -0.0212473609, -0.0775994211, -0.00118725002, -0.0782555565, 0.0178641155, -0.0689989477, -0.0248651691, 0.0331919342, -0.0804729313, 0.147161454, -0.0213274248, 0.0495033935, 0.0764237717, 0.0679708943, 0.0652758181, -0.00163454004, 0.0484560132, -0.0121581219, -0.0294768251, -0.0991435349, 0.0434749015, 0.041380845, -0.0336263925, -0.00684622675, 0.00642223284, 0.113141291, 0.00063541159, 0.0797164962, 0.00572476164, 0.00803749915, 0.00497916713, 0.0753425732, 0.0550090857, 0.0912253633, 0.0515357107, -0.0963370577, 0.0212445389, 0.110619225, 0.0104701724, 0.038355682, 0.0566010661, -0.0528693311, -0.0188960116, -0.00828725286, 0.00950297341, 0.013510732, -0.00288709812, 0.036969047, 0.0287468154, -0.0306389034, -0.0461689308, 0.0143044386, 0.10684415, 0.0850169808, 0.0378084108, -0.0764039159, -0.11663378, 0.0441069901, 0.0465431176, -0.111619808, 0.161576584, 0.0282414705, 0.0527949333, -0.084071584, -0.0209491625, 0.0541457981, 0.0392391868, -0.0112208202, 0.131430283, 0.0981135964, -0.0509605333, 0.0122558931, 0.000687881373, 0.0265618041, -0.0195218176, 0.0836447179, 0.0750810206, 0.0458138585, 0.146810755, 0.112280034, -0.0652331486, -0.0341970846, 0.0334284902, 0.0540269427, 0.041710116, 0.00432903506, 0.00225922838, 0.0864569694, -0.0504702739, 0.0638329089, -0.103701279, -0.0741944537, 0.0245679785, -0.00566792488, -0.0840940848, -0.109055251, -0.092332907, 0.0407088175, 0.0101407645, 0.00827308837, 0.0545968898, 0.0400347561, -0.0566380098, 0.056541197, 0.17530027, -0.0367391258, -0.0958183855, -0.00934026763, -0.158351377, -0.155936778, 0.118473843, 0.0447239876, 0.0262825079, 0.0385334156, -0.109556459, -0.0255446192, -0.110488355, 0.00124787726, -0.0593225025, -0.00273051858, -0.119895019, 0.0221740324, 0.0167334601, -0.00351163605, -0.113927417, -0.0656535029, -0.0626883954, -0.104976065, 0.0191272385, -0.0353834517, -0.00768600404, 0.070701763, 0.0799218565, 0.0391910449, 0.00603917427, -0.059693262, -0.0492252111, 0.00577678531, 0.0442071334, -0.030128587, 0.066669561, 0.0311337113, -0.0896128789, -0.0929164663, -0.0267600212, -0.0353194922, -0.0334425792, 0.0913329497, 0.150555521, -0.028989261, 0.0309862904, -0.0615032986, -0.0679526925, 0.127847388, -0.050558269, 0.0688756928, -0.0219995752, -0.0388680398, -0.0246833228, 0.0794024989, 0.0578956082, -0.122922733, -0.00071552489, -0.0139164357, -0.030640576, 0.04551965, 0.0506845452, 0.0188603736, 0.0150425369, -0.0802400485, -0.154520959, 0.08918643, -0.0576012246, -0.0230565853, -0.0639366955, 0.0376155786, -0.00303743314, 0.0425109267, 0.0585362539, -0.0916770697, 0.0326580703, -0.0483011715, -0.0244255308, 0.00619422412, 0.0650111437, -0.0211275108, -0.0167442448, -0.0301489234, -0.0189132728, 0.0992666334, 0.099879846, -0.0303247832, -0.00238152314, 0.0860659778, 0.041869022, -0.0518088713, -0.116496213, 0.0370620675, -0.0484162308, 0.104685262, -0.10294643, -0.0191542041, 0.0183966011, 0.067674771, -0.0119359214, -0.0921194628, -0.0441772528, -0.0722718909, 0.0796230286, 0.0795891881, 0.061415635, 0.0472054407, 0.00711930217, -0.0801173747, 0.0219572019, 0.117652074, 0.0209528711, 0.0392731838, -0.0209772401, -0.14853999, 0.129064411, -0.0459602326, -0.0507139154, -0.0590851903, 0.0681848675, -0.0333252326, 0.0525169, 0.0554127023, 0.00368930586, 0.085702166, -0.0775162429, 0.00429337425, -0.0587444566, -0.113069221, 0.000643355772, 0.00562279858, 0.03658548, 0.052098155, 0.107099369, 0.0667936131, -0.0185411349, 0.054342512, -0.0529061705, 0.0734526962, -0.0151351551, -0.0273972377, -0.00876887143, 0.0737391412, -0.0285417158, -0.0303514209, 0.165578246, 0.0638718382, -0.117830209, 0.0496585406, 0.041049473, -0.041145876, 0.00240243599, -0.134060368, -0.0371007062, 0.156852558, -0.038457267, 0.117742702, -0.109646179, -0.0261033438, -0.0273322314, 0.0502961725, -0.00987560581, -0.176500574, 0.10560666, -0.0534770451, 0.0755180418, 0.073453106, -0.00855196454, 0.0408811681, 0.0972820148, 0.00222174916, -0.0196923241, 0.0295872837, 0.045618359, -0.0173810925, -0.0635485649, -0.05865952, 0.0125012361, -0.117654167, 0.0167404786, 0.00176727842, 0.0445348695, -0.110756509, -0.0411797725, 0.060854964, -0.0363162272, 0.0225862637, 0.148795485, -0.0943279639, -0.00545653328, 0.0138726663, -0.0828919411, -0.035351567, -0.0137856416, -0.0302281063, 0.00956151262, -0.000997079536, 0.0637324005, -0.124670953, -0.135817915, -0.0111148534, 0.0395183228, 0.0349599272, -0.0692137033, 0.0396531895, 0.0560348853, 0.0915048048, -0.0951796025, 0.104822598, 0.0226972662, -0.0891933069, 0.0428549908, 0.0416089669, -0.0720485374, 0.0193011872, -0.0514923371, 0.0840799958, -0.0275733396, -0.143871188, 0.0486096255, -0.120800242, -0.014725361, 0.0171756092, 0.0356361233, -0.0434459001, -0.0433174782, 0.0299344528, -0.0154602686, -0.0220428221, -0.0309799686, -0.0465802662, -0.00123932632, 0.01409504, 0.0529759042, 0.0602477156, -0.086191386, 0.0324929543, 0.128435671, -0.10888043, 0.000272087753, 0.0894615874, -0.0358649753, 0.166124359, -0.0133904777, 0.109172203, -0.0641209632, -0.107063599, -0.0110514136, 0.041730687, -0.0877945274, -0.142711118, -0.0765860453, -0.0497560874, 0.0428826585, 0.0574328303, -0.0130979903, 0.125451609, -0.0108842459, -0.0494310446, 0.109787889, 0.0778675824, 0.0823265761, -0.0133256987, -0.103071883, 0.0263200104, -0.0636986345, -0.0152745089, -0.0770010874, 0.0953732282, -0.0105203716, 0.0261606909, 0.027641397, 0.00574612617, 0.0131082274, 0.0553812869, -0.0236430056, 0.0110867014, -0.062127091, -0.0989792496, -0.0495412424, -0.0565992408, 0.0525233187, 0.0198662262, -0.179235637, 0.0898453221, 0.0248485431, 0.0347248986, -0.127199203, 0.0660550743, -0.0934803188, 0.00469446182, 0.00628458615, -0.015294848, 0.0112601621, 0.0915097445, 0.0121056205, -0.00299266726, -0.0751530081, -0.0402411073, -0.0411809869, -0.117185861, -0.0398585685, 0.083669208, -0.040651612, -0.0212481618, 0.0913396031, 0.0123984385, 0.0395914689, -0.0734995976, 0.0387141407, -0.0307631381, 0.0512015224, -0.0166006796, 0.0476839878, -0.00363002811, -0.044824414, -0.0565983057, 0.0472218171, -0.103720374, -0.0252437219, -0.0110661779, -0.0145094479, 0.0776091963, 0.132596031, 0.165300861, 0.105620116, -0.00800295733, 0.134556919, -0.0709809735, 0.0141896494, -0.0762698054, -0.0081240423, -0.0925129652, -0.0793496817, -0.0711927637, -0.0323574767, 0.0483066738, 0.0424038321, -0.0841650516, -0.0245392136, 0.0438334122, 0.0510460362, -0.0362881906, 0.0453605168, 0.0559055582, -0.0746992081, -0.0399772748, 0.0465168618, -0.141152978, 0.00446203956, 0.108306855, -0.0510297939, -0.0421319678, -0.0211320929, 0.0714860559, 0.104075775, -0.0466121845, 0.0498371385, -0.0711495504, -0.0451222062, 0.0821564347, 0.0265221037, -0.0201894213, -0.0309638102, -0.0375229344, 0.108002588, 0.1360026, -0.041354008, 0.0148476101, -0.136250153, -0.111906879, -0.114485517, -0.0318824686, -0.0298597962, 0.083672829, 0.0479454696, 0.0930844545, -0.060877461, 0.0467161275, 0.0868022069, -0.134293407, 0.00406222977, -0.0133788846, 0.00992775895, 0.0371012837, 0.000178516842, 0.0635174811, 0.0686589777, -0.0874956846, 0.0660264939, 0.0604191311, 0.0928163305, 0.00827313028, -0.0172130056, -0.0890372694, 0.0775875002, 0.0471425802, 0.0283339173, 0.0665764511, 0.121209987, 0.00305609987, -0.0121471994, 0.0831000879, 0.0268709604, -0.0201124046, 0.138248697, 0.100675456, 0.0173395015, -0.0172923226, 0.123695709, 0.0999183804, -0.0625192374, 0.193295047, 0.0205619447, -0.0610130019, -0.0741292834, 0.00925136171, -0.0755780712, 0.0248802584, 0.0684561953, -0.0357257873, 0.0628755689, -0.0676857382, 0.149378628, 0.078054443, -0.017178461, 0.0729198828, 0.0285188742, -0.0298199169, -0.107661113, -0.000575106591, -0.0742195025, 0.0206028353, -0.015194552, 0.0513066649, 0.0439567007, 0.11916057, 0.0410906821, -0.101361863, 0.00873067416, 0.0579848811, -0.00293635204, 0.0556497499, -0.0703574941, -0.0211555995, -0.0211676806, 0.0805090666, 0.0674633011, -0.0395794064, 0.0116857458, 0.0380934738, 0.0536395274, -0.0107757486, 0.0702201724, -0.0111099351, -0.0208020341, 0.0421061739, 0.015531511, 0.0450606272, 0.139781103, -0.0504179224, -0.151396498, 0.104282871, 0.168288693, 0.0592916235, -0.104686722, 0.077467382, 0.0554249324, 0.168543816, -0.0889628679, 0.0860685781, -0.075816907, -0.00723795965, -0.0432170518, 0.0212600082, 0.049996458, -0.0394047275, -0.0971770585, 0.0513941944, 0.0137694366, -0.0819444507, -0.0508803576, -0.09034881, 0.0181277636, -0.0112295821, -0.0214229617, -0.0297272354, -0.0584390461, 0.0124653149, 0.0346170813, -0.0422079898, 0.124681838, -0.126552731, -0.0979950204, -0.0617791265, -0.0607632399, 0.0271472353, 0.0653879493, 0.0878731906, 0.0700205639, -0.0435249135, -0.056338612, 0.0412846953, 0.0253047347, 0.027021125, 0.105870433, -0.0201928541, 0.0810924619, 0.0396603718, 0.0434814692, -0.0732205659, 0.152788639, -0.0767242163, -0.057194937, 0.0340616703, 0.0693667531, -0.0196612254, -0.0826099664, 0.0341789797, -0.0540570468, 0.0862257481, 0.155302301, 0.0740946457, -0.0832137838, -0.0889928043, -0.0929092243, 0.105825774, 0.110529013, -0.0169815123, 0.0412914976, -0.120870762, 0.0653953329, 0.0719392151, 0.0856548399, -0.0752637684, -0.0918144956, -0.0356733054, 0.0593351759, 0.0192785952, 0.134731516, 0.0298854578, -0.22963056, -0.089094311, 0.0390513539, 0.0759049505, -0.0633867681, -0.0268667713, -0.00343836844, -0.0256426632, 0.0398066193, 0.022945866, 0.0420098975, -0.00350727141, -0.014944654, 0.101577669, -0.108422257, -0.200207785, -0.00578112528, -0.139163405, -0.08182697, 0.0119988667, -0.0297275037, 0.0233182143, -0.103024743, -0.00383697683, -0.0522182137, -0.0818012059, 0.181222022, 0.0674812645, -0.0762788802, 0.0478710756, 0.0257269125, 0.0580434762, 0.00955753028, 0.0505937375, 0.0182330348, 0.0231178608, 0.0381997339, 0.0372849107, 0.0418353304, 0.0989421234, 0.0434807688, 0.0115981149, 0.0344024263, -0.0854934603, -0.00655464642, -0.0535590649, 0.11046946, -0.0398580283, 0.0241416339, 0.0115565509, -0.0263186991, 0.021106042, -0.00454965793, 0.00473457016, -0.0293057654, 0.00974595081, -0.153997883, 0.0386386216, -0.0189007111, -0.0384422429, -0.0820041448, -0.000343965366, -0.101367287, 0.158929065, -0.167421445, 0.0100682098, -0.0276947729, 0.127314717, 0.109571099, -0.0979896188, -0.00764027238, 0.0627418682, -0.062974833, 0.0021440573, 0.0187398717, -0.116322875, -0.0296423174, -0.0309300087, 0.0427315794, 0.0603606105, 0.0492910594, -0.0101312613, 0.0403695591, -0.122192383, -0.0596618354, -0.006468195, -0.00582188414, 0.0456683524, 0.08462248, -0.0642502531, 0.0695199221, 0.104578532, -0.0763068423, -0.0383230411, -0.115195557, 0.0805008113, 0.0371084101, 0.0499783009, -0.0620879009, 0.110976398, -0.0233650394, 0.178990453, 0.00924512744, -0.0522588454, -0.0252414644, -0.0995525867, 0.0605548769, 0.041917529, -0.0127279628, -0.0714572221, 0.0253617242, -0.113619633, 0.0571864396, 0.0421477221, -0.0455778614, -0.0354776122, 0.0346949771, -0.0156272464, 0.0213422589, 0.00892110169, -0.0124027561, -0.0183743574, -0.0407236591, -0.0177347586, 0.0878833383, -0.0695776194, 0.052132871, -0.0773894116, -0.144517958, 0.00482582301, -0.0226116925, 0.0160243455, -0.0286830291, -0.11305742, 0.101025783, -0.0856631398, -0.0672385097, -0.063888438, 0.134303913, 0.0549882837, -0.10768798, 0.0699498281, -0.00243488327, -0.0660401583, 0.0233532116, -0.0300203152, 0.0456442125, 0.101627544, 0.0769642889, 0.126996264, 0.000388812274, 0.0238995105, 0.0611703172, 0.161981046, 0.0104111126, -0.0210280977, 0.054599572, -0.163943604, -0.0888782218, 0.0246563032, -0.0952074975, 0.0669457465, -0.028490793, 0.124237835, -0.0327320583, 0.0467088819, 0.00436432566, 0.0165604576, 0.0425928347, 0.0523858219, 0.0352160819, -0.0192053169, -0.0619856268, 0.00652379543, 0.0649601892, -0.0250049718, -0.0268743802, -0.1220228, -0.04697432, -0.107010745, 0.0142582282, -0.1341566, 0.112670496, 0.0275352411, 0.0738019124, 0.0107060857, -0.132511884, -0.0193026438, -0.110272646, 0.0176010579, 0.0456731617, 0.0540217906, 0.101229809, -0.0176883563, -0.0548925437, 0.0111844558, 0.0977346152, -0.0939161479, -0.120759696, 0.00728588551, 0.0550565235, -0.029833205, 0.0463131741, 0.0199479777, 0.0799656361, 0.024923414, -0.0735116154, 0.133153856, 0.00860225316, -0.0625157654, -0.0283735283, 0.0827504992, 0.0140353963, 0.0028263703, 0.0391749628, -0.0747612491, 0.0264509879, 0.0634570345, -0.0968047306, 0.0735668764, -0.01932019, 0.0665857419, -0.0885678008, 0.0111907255, -0.0831329077, -0.0440419391, -0.0322117545, 0.0892609581, -0.0616574325, -0.0200462975, 0.0808087736, 0.0819935501, -0.0530164167, -0.0429007262, -0.00939739309, -0.0263765268, -0.137593597, -0.00815229025, 0.0761511475, -0.0534029752, 0.0863740742, 0.0341856666, 0.0761782378, 0.0798772946, -0.0981286988, -0.0827985257, 0.0168975629, 0.093077831, -0.168395638, -0.0431145653, 0.016699478, -0.00326111913, 0.015668232, 0.0981467217, -0.000121034682, -0.00150727481, 0.00911068171, -0.194074079, 0.14716652, -0.0177265238, -0.0327950604, -0.0578373149, 0.0473306887, -0.0268291067, 0.00913901348, 0.0758189857, 0.00338140503, 0.0992139801, 0.0170033798, 0.0540252551, 0.00315051153, 0.160677493, 0.0503151082, -0.0142692998, -0.0541427769, -0.0480790213, -0.141287893, -0.0236011781, 0.0220742133, 0.00780775771, 0.0283384491, 0.0634254366, 0.0844219178, 0.117850721, 0.0364065841, -0.00560771488, -0.0684203058, 0.0683472604, -0.0800958723, -0.024984628, 0.0593558885, 0.0699148774, 0.0657431185, -0.0415165834, 0.111496188, 0.0136796553, -0.00992874987, 0.0449885093, -0.0500408486, 0.00715490058, 0.0617081225, -0.0271681473, 0.0663627312, 0.0376835912, 0.00175093859, 0.0915442854, 0.105019227, 0.0400546379, -0.00614744518, 0.0322519839, -0.0272529051, 0.0788775086, 0.0287162662, -0.0435082987, 0.0217745118, 0.0680316836, -0.0822205916, -0.00315487385, -0.176027328, -0.121989861, 0.0802285671, 0.068146795, -0.168543041, -0.00805228017, 0.0575836152, 0.0659630448, 0.00027151301, -0.184287474, -0.077234745, 0.0259619169, -0.0104427869, 8.8326633e-06, -0.0462127365, -0.0143509647, 0.0386136211, -0.0137817906, -0.094456248, -0.159782857, 0.0176643096, 0.0408019051, -0.205906004, 0.0498316512, -0.0390802771, -0.00614602491, 0.0377606116, -0.0166628994, -0.0740462244, 0.0353523642, 0.180034012, -0.00229755789, -0.0284066554, 0.028490454, 0.0382132977, -0.0177712403, 0.00686036982, -0.030679781, -0.125406608, 0.0881356671, 0.0438567437, 0.117961451, -0.00673158048, -0.0559261478, 0.130192861, 0.189995065, 0.000300833955, -0.0918848291, -0.0665715709, -0.0063006077, 0.0395032689, 0.0745402798, -0.0587377436, -0.13368988, -0.180422559, 0.00515289791, 0.0346100554, -0.0216367804, -0.0543315858, -0.0574583523, 0.00970618054, -0.0398748443, 0.0254109539, 0.114461258, -0.121243052, -0.0534580722, 0.017572619, -0.0689000115, -0.0722096637, 0.0707206577, 0.0562217236, 0.0416003615, 0.110389158, -0.00586797949, 0.109078795, 0.0627859309, -0.0746139437, -0.178598255, -0.0356704518, -0.00472285412, 0.107308924, 0.0908543617, 0.0450132415, -0.0254008416, -0.00743856747, 0.0904664099, 0.0640947297, 0.0863719136, -0.0958629251, -0.0241381582, 0.0598428063, -0.0499173477, -0.0409107246, -0.0345571712, -0.0390259549, 0.0102475435, -0.0146067096, 0.0161825232, -0.150251925, -0.0792580172, -0.0553167947, -0.0292260703, -0.0188379996, 0.000643459149, 0.0435580686, -0.084482573, -0.0985249802, -0.0343088098, -0.0382055268, -0.0432224087, 0.0883175135, 0.0756114796, -0.107673466, -0.134927794, 0.156511784, -0.0245051514, -0.0353129432, 0.00829586387, -0.00211312249, -0.108969897, -0.00366004184, 0.0100791585, 0.0278191306, 0.0497515127, 0.0214323848, -0.178656191, -0.0619581416, -0.0192200616, -0.0922988132, -0.0254442655, -0.0353798307, -0.00773616694, -0.0958243981, -0.0667599365, -0.0184887256, 0.00128525868, -0.00953026954, -0.0225979239, -0.108141951, 0.0378866009, -0.00547851995, -0.0586479455, 0.0130515173, 0.0227658413, 0.0219786353, -0.202414721, -0.0952945799, 0.0276389942, -0.0366673917, 0.200630739, -0.0574049354, 0.219369635, -0.00560873933, -0.0660076439, -0.0390148684, -0.031058291, -0.0553637519, -0.0270704888, 0.0335120894, 0.0195704568, 0.150406182, 0.0333154984, 0.0506328456, -0.0182577893, 0.0639431775, -0.0194490161, -0.00723955827, 0.0276241396, 0.0438724533, 0.00639448036, 0.122798778, 0.143087864, -0.0388212763, -0.0141448826, 0.0388008952, -0.144713074, -0.0721375495, 0.0446854755, 0.109467804, 0.120496161, 0.00206460478, -0.0913183168, -0.0142692104, -0.0134913214, -0.0455319732, 0.0245725252, 0.0421691984, 0.0899413675, 0.102732658, -0.0451376662, 0.00271292776, -0.0701145157, -0.000515389256, -0.00187888183, 0.123769432, -0.0278835259, 0.000219712034, 0.0368434861, -0.0115500763, 0.0699552074, 0.0782960579, -0.00789592229, -0.0588972867, 0.015475966, -0.0345260911, 0.0453729257, -0.0503094792, 0.0914688855, -0.0559914261, 0.0229284205, -0.0123081263, -0.032612633, 0.0111059695, 0.0172873586, -0.0874353051, 0.0297923144, 0.0108721172, 0.0613508858, -0.00696083298, 0.0901359767, -0.0355426744, 0.0571047217, -0.0433449, -0.0547627285, 0.0374375358, -0.241334602, 0.00544045493, 0.0808352008, 0.0276897345, -0.0174633767, 0.071427986, 0.0266567338, 0.0054734163, 0.0435120538, -0.015824059, 0.123210691, -0.0259859301, 0.079398334, -0.0699486658, -0.0321526751, 0.0427672118, 0.107578516, 0.0229987837, 0.112871855, -0.0395532139, 0.00172494003, -0.129916966, -0.117473572, 0.118357927, -0.061017476, -0.0727849305, 0.0315671861, -0.0112778656, 0.00469734892, -0.106646806, -0.0425762646, -0.0328396969, 0.0200689025, -0.126754105, 0.0516137779, -0.00969748292, 0.0385525115, 0.0171331055, 0.0715736002, 0.0561930761, -0.0456623957, -0.0544602834, 0.0509038232, -0.0235189423, 0.0454678312, -0.0445984229, -0.0730791166, -0.0636863112, -0.0429399535, 0.0852165446, -0.00184737332, -0.0186565965, -0.0110966153, 0.162937522, -0.0437614545, 0.0861722082, -0.072525084, 0.0506918468, 0.0179148056, -0.0612825491, -0.0275459439, 0.0272253174, -0.0334783643, -0.0732806772, -0.0769508258, -0.0695436373, 0.0133161955, 0.0472069159, -0.0879593343, -0.0580082238, -0.0633575395, 0.0257822312, 0.030667264, -0.0600329526, 0.10595277, -0.0886051506, 0.092257075, 0.00813044235, 0.013223296, -0.0289506428, -0.00761445984, 0.107809797, 0.0216514673, 0.0489909947, 0.0685153082, -0.104536615, -0.154011056, -0.0122282058, -0.100846365, 0.00166160613, -0.00527038006, 0.0229451079, -0.169116393, 0.00357444584, 0.130249828, 0.0318445526, 0.0451219939, -0.0985371321, 0.077016972, -0.0675574839, -0.0485341214, 0.0892937258, -0.0119261499, 0.11686936, -0.0256366096, -0.064719893, -0.138646811, -0.0230368841, -0.0518703535, 0.0107466932, 0.0913660228, -0.0292170253, -0.00676173903, -0.161402151, 0.0616877712, -0.00999165885, -0.138042018, -0.0479046628, 0.109722525, -0.020709455, 0.00616726419, 0.0622854307, 0.0453955196, 0.0129737593, -0.0028758687, -0.0481419265, -0.0273242481, -0.0312653147, 0.0190724395, -0.102354854, 0.133722231, 0.0744988471, -0.0438664332, -0.118296951, -0.060179811, 0.0385666713, -0.0278032012, 0.0657609701, 0.0827093944, 0.0629360303, -0.0218015127, 0.0498604961, 0.0824899077, 0.00780756585, -0.121808678, -0.023255948, 0.018228665, 0.0122035956, -0.0136935897, 0.0258074179, 0.0411146283, 0.021556396, -0.0242421646, 0.0856881812, -0.0653296635, 0.0157615319, 0.0421842411, 0.0580450147, -0.00777962804, -0.0839014277, -0.151935533, 0.0329401083, -0.0699129552, 0.0765977055, 0.0439387038, -0.0685167909, -0.0831892118, -0.0514106527, -0.028607633, 0.061502032, 0.086351648, -0.00262156688, -0.0871760249, 0.12683478, -0.159808025, -0.163172737, 0.033106152, 0.00390011352, -0.0290324241, -0.0548253208, -0.0273482688, 0.11500749, 0.202738315, -0.00152360462, 0.0413755588, -0.00100732222, -8.979626e-05, -0.170355201, 0.06213855, 0.062782988, -0.062111754, -0.0467889421, -0.123734884, -0.0822224766, 0.0064563714, -0.0526950732, 0.0135611612, 0.00378175639, -0.0321302637, -0.00103278458, -0.0106755365, -0.0156611875, -0.0274015479, 0.066288501, -0.00762125198, 0.0554921851, -0.0248665251, 0.0889319927, -0.193257019, 0.00683034211, -0.00892718881, 0.0225240719, -0.0810979083, 0.0546551943, 0.0133333094, -0.00835020654, -0.0154363895, -0.0218534134, 0.0765927285, 0.0662077218, -0.0222853124, -0.0838636458, 0.0949314907, -0.0462717786, 0.0445657931, -0.0973079279, 0.00222689845, 0.052203007, -0.0551824458, -0.016072819, 0.157039225, 0.146399975, 0.214229614, -0.00472382829, -0.0298488569, -0.0895316973, 0.0459648371, -0.0893030912, 0.0142214783, 0.00727055222, 0.0673766881, 0.153079078, 0.0623493977, -0.0353417471, -0.0408567637, -0.0287689026, -0.164291218, -0.072588101, 0.122869678, -0.0809252784, -0.0744258314, -0.0263943821, 0.022311585, -0.0519490838, 0.0310675688, -0.0436468273, 0.023407463, -0.0411918163, 0.0230428837, 0.0311317667, -0.066521503, 0.0143625438, 0.0257104225, 0.055129271, 0.0788489655, 0.0219211429, 0.0075901784, 0.0655827448, -0.00681952946, 0.0695478916, -0.0999718606, 0.0466005281, 0.0790512338, 0.0724594891, -0.0388102382, -0.0497607887, 0.0118607767, -0.120786272, -0.0297009759, 0.0503409319, 0.0806155726, 0.0945888907, 0.0203324463, 0.1338211, 0.00627672672, -0.0638806894, -0.096447587, 0.0469171293, 0.134490743, 0.0629716888, -0.0161998235, 0.0417893231, -0.127393022, -0.0704433918, -0.00859997049, 0.0384261608, -0.00676104892, -0.0117424373, 0.00263016298, 0.0532458425, -0.0523997359, 0.0430650339, 0.0897080898, 0.0859533995, -0.037975464, 0.00416474417, -0.207259476, 0.0323172584, -0.0114803053, 0.0962532684, -0.0106872888, 0.0364580899, -0.16184397, 0.0418573469, -0.122858383, 0.0221215859, -0.121820882, -0.102466725, -0.089056842, 0.0367734917, -0.110163748, 0.0508830175, 0.0022703018, -0.0185247958, -0.0431330279, -0.0516164042, -0.0410573855, 0.0802833885, -0.0442520902, 0.00709324144, 0.0835353509, 0.0636074319, -0.01820039, -0.116703451, -0.0991834998, 0.0787881315, -0.00421014987, -0.0709599182, 0.0636661947, -0.0746797398, 0.0826184154, -0.0111790467, 0.0135124158, 0.0346965566, 0.0317447968, -0.0182662159, 0.0654354095, -0.0183947254, -0.0237028897, -0.112371206, -0.00207559043, 0.0984482542, 0.057263054, 0.145837754, -0.0390798263, 0.0178938676, 0.0160873868, 0.0243467428, -0.0410782658, -0.0260812677, -0.0531546474, -0.011475645, -0.0513886809, -0.0241638664, 0.00806893036, -0.0697995052, -0.16929169, 0.144684523, -0.0839521885, -0.0113528688, -0.133523107, 0.0680152699, -0.00267725252, -0.0366772451, -0.0540373474, 0.0585089996, 0.00522282999, -0.0195852555, -0.00349725457, -0.0399441458, -0.0847067609, -0.0519267805, 0.0270239264, 0.0249403715, -0.0854221731, -0.0345031247, -0.0426385999, -0.114951417, -0.11833813, 0.0797540545, -0.138187185, -0.200031623, 0.0208405778, -0.114357784, -0.0794100016, -0.0402523465, -0.0483966842, -0.055653058, 0.0419644527, -0.0422492661, -0.0022473936, -0.016253138, 0.103890084, 0.0317640528, -0.0461630151, 0.0666900128, -0.0453241915, -0.0304095335, 0.120142452, -0.0867946148, -0.0395014733, 0.0954977423, -0.0116896294, 0.0413545854, -0.0663651079, -0.0479582623, -0.0986374393, 0.01779503, -0.0141012948, -0.147269323, 0.043544963, 0.0628029183, 0.0814529136, 0.103698663, -0.0168878809, 0.0208992399, 0.127812594, 0.133393362, -0.0354451574, 0.0245596617, -0.0433239639, 0.116616994, -0.029590657, 0.0375297517, -0.0554959513, -0.00119716767, 0.044206921, 0.0155456532, 0.0627288669, -0.0212567691, 0.0345831551, -0.0273814127, 0.070053488, -0.0332821012, -0.0976672098, -0.0103713432, 0.112356469, -0.110892266, -0.115188025, 0.0184156187, 0.15654473, 0.105028741, 0.0263991877, -0.119852051, -0.124294557, 0.0738592073, 0.0314462334, 0.0596648566, 0.0754985213, -0.0108051253, 0.00271856412, -0.0948751941, 0.0416161828, 0.094782874, 0.0168600567, 0.100057401, 0.0786821395, 0.0506573021, 0.0367843024, 0.122363187, -0.0764172822, -0.0260445774, -0.0560432374, -0.137111887, -0.0604897812, 0.000700753182, 0.0843180567, 0.0795811936, 0.106576502, 0.0707424656, -0.00559558813, 0.186479449, 0.00338681787, -0.0375811607, -0.0175246857, -0.206482515, 0.0203088261, -0.00335052237, 0.00765392184, -0.0219054036, -0.092422016, 0.130213648, -0.00963715278, 0.0746578574, 0.0298792869, 0.0852276832, 0.0452477895, 0.00293635018, -0.0406028107, 0.0471775532, 0.00875167921, -0.103349723, -0.0448772684, -0.0290297251, -0.0449584275, 0.0139079317, 0.042584952, 0.0688365772, -0.0339850076, -0.0264592171, -0.029722875, -0.0137560796, 0.0814295486, 0.139631897, 0.0442709774, 0.0383184664, 0.00529657491, -0.0937576964, 0.0498953275, -0.0153518096, 0.109351449, -0.102684058, 0.0631108433, -0.0590194762, 0.00657091849, 0.0752271339, 0.0661112741, -0.0187464096, 0.075098075, -0.00506668538, -0.0846352205, 0.102858834, 0.0224678852, -0.12960352, 0.0128765544, -0.047212813, -0.0523117818, -0.0533741787, 0.0276528094, -0.0502135083, 0.0194695443, -0.0143132471, -0.108509399, 0.148433045, 0.0380441174, -0.00505725481, -0.00490636192, 0.00429776311, 0.0980975479, 0.0316283181, -0.0629595444, 0.0340179801, 0.0504700691, -0.0740982369, -0.0247772243, -0.00488639064, -0.0241223183, 0.0343791023, 0.0140596097, -0.11004588, -0.162041143, 0.160919592, 0.0192217976, 0.0153533816, -0.116443589, 0.0119418502, 0.0596936829, 0.0197722968, -0.0355095007, 0.0546094067, 0.0722641721, -0.14327307, -0.0360650346, -0.0379500166, 0.0014279075, -0.147924304, -0.020114379, 0.0699339956, -0.170718387, -0.0270746127, 0.00512433425, 0.092315577, 0.131550461, -0.00501552038, -0.0553552136, -0.082342945, 0.0269107912, -0.0393439606, 0.0932399482, -0.0991183147, -0.0281126946, 0.0545121729, 0.158625185, -0.151274264, -0.0417198464, 0.106845811, 0.0443828851, -0.0319172107, 0.106447905, 0.0355612896, 0.0712697878, 0.0547756553, 0.0446596593, -0.00519914692, -0.0135855507, -0.0165826976, -0.0246209577, 0.0719221979, -0.0314692408, 0.0288045667, 0.0762285292, -0.0109113827, -0.022664547, -0.0388147011, 0.0331881642, 0.0150379529, 0.0966883153, -0.0536429547, -0.00123625062, 0.0361921415, 0.0258746333, 0.00602638721, 0.0252074562, -0.0116876867, -0.0563903525, -0.0773122236, 0.0541616417, -0.0449338108, -0.0872624815, 0.0239573307, 0.044475887, 0.109698713, 0.00538090896, -0.110722005, -0.0317043215, -0.0926145539, 0.134996489, 0.0132420855, 0.0307217035, 0.129866838, 0.0446491763, 0.142542303, 0.0755499601, 0.0766458809, -0.0939057022, 0.0864705145, 0.0947403759, 0.0673735887, 0.0167821161, 0.081167236, 0.0321459137, 0.0442270897, -0.12323533, -0.00251188874, 0.128289878, 0.0102645457, 0.0948777199, -0.0265928544, -0.0382959172, 0.0444154963, 0.00423470698, 0.0442593768, 0.0491274074, 0.0461569838, -0.00353324227, -0.00449061394, -0.00850099511, -0.0989271998, -0.020404553, -0.0843655318, -0.0262944549, 0.0354807973, 0.0195747688, 0.111938857, 0.0576216951, -0.0198118836, 0.0159228332, -0.0617595017, 0.0832970738, 0.125676692, -0.0676809177, -0.044418402, 0.112666965, -0.139435753, 0.0150006581, 0.0409631506, 0.00353996176, -0.0138108842, 0.0315121263, -0.138240442, -0.0448639207, -0.0652330965, 0.168961555, -0.00368394144, 0.0176044479, -0.0080471728, 0.0863961801, -0.0953193232, -0.1276021, 0.00624971464, 0.0463307425, -0.104270786, -0.012664225, -0.143328652, -0.0620809272, -0.0988290012, -0.0149173979, -0.133307338, -0.0877726898, 0.0622825958, 0.0848572403, -0.0544980206, 0.0604782254, -0.0921068341, 0.136214122, -0.136167347, -0.0482977405, 0.0570528917, 0.00825358182, -0.0369862393, 0.000268530101, -0.128857091, 0.0113458, 0.201225728, -0.0113300551, 0.117818505, -0.0952969566, 0.0119970953, -0.096570082, 0.0346703082, -0.000416658819, -0.0108677037, 0.0852801204, -0.00154381618, 0.0486050583, -0.0845545381, -0.0183461979, -0.00870124996, -0.0703145713, 0.127825424, 0.0226284154, -0.108716726, 0.07842464, -0.0543230176, -0.000194082037, 0.119213894, -0.0854408368, -0.016298499, -0.0377904773, 0.0239778813, 0.0804838911, 0.159557447, 0.0241290852, -0.0569810495, -0.0283770934, 0.00125440955, -0.0842455029, -0.00941268913, 0.00669839699, -0.140971035, -0.121554032, 0.0335644558, -0.0518988892, 0.0265859105, 0.071242772, -0.0262365974, -0.0189802349, -0.0420945585, -0.0380737334, -0.0346987396, 0.104707107, -0.0260187313, -0.00708856294, 0.0157035533, 0.00604697037, 0.00217210129, -0.00494368188, 0.0197832491, 0.0417141728, -0.129215866, -0.0305279493, -0.0844836831, -0.0354751274, -0.0694699809, 0.0929484665, -0.0291762762, -0.188328281, -0.0487990417, 0.0315973833, 0.0206779912, 0.128925368, 0.030309651, -0.118210331, 0.057885319, 0.0857507288, 0.213871256, -0.0757404938, -0.0637934059, -0.0889232978, -0.070100069, -0.125684023, 0.0101588191, 0.0788855776, -0.0299824625, -0.096968323, -0.00361710414, 0.0302541051, 0.060895294, 0.117318891, 0.00945788436, 0.00684899278, -0.0141613223, 0.0400242209, 0.0520439968, 0.0600204505, -0.0246140398, -0.0945139974, -0.0242358223, 0.0106533356, 0.00207729638, 0.138632506, 0.0240307096, -0.205044702, 0.099337101, -0.105229884, -0.0547111779, 0.0454545133, 0.0346658826, 0.0309550203, 0.105702542, -0.0286708586, -0.0798922405, -0.0711463839, 0.0419986509, 0.0664751306, -0.0887834206, 0.115568608, 0.106128082, -0.0161237307, 0.0741705745, -0.0297651812, -0.10414964, 0.0249607414, 0.0709991083, 0.0542765446, 0.0252491813, -0.153204277, 0.114114977, -0.103163362, 0.0376967713, -0.0982381552, 0.0341025777, 0.0852912813, 0.0688287467, -0.00458452106, -0.0439122654, 0.0618342012, -0.0331042111, -0.0731438547, -0.00486975163, -0.134314567, 0.043294467, 0.0666260123, -0.135846078, -0.0551270843, 0.087324217, 0.0839074999, 0.0684562847, -0.0524627268, -0.0236464273, -0.0132759549, -0.0257256441, 0.0554094352, 0.0464685708, -0.0353934243, 0.0220088363, 0.0119866524, -0.0649880096, 0.0026059635, 0.0198674537, -0.0815643817, -0.154027954, 0.0209241249, 0.102914758, 0.104896873, 0.0796399266, -0.00783735327, 0.0127343731, 0.00208612438, -0.0909104943, 0.00549368933, 0.165070027, 0.0412174463, 0.0781062245, 0.0734480992, 0.12345285, -0.123697817, -0.0625981539, 0.092018649, 0.161089271, 0.0978915393, 0.0666619316, 0.0156493112, 0.0594945885, 0.112634279, 0.0463874377, -0.123239174, -0.188735694, -0.0156784058, 0.012096677, -0.0238690488, 0.0179750621, -0.078954801, -0.00978407636, 0.0626665205, -0.0990869999, -0.0145246116, 0.00753659382, -0.00861090422, -0.0665304884, -0.151779816, -0.029356245, 0.0170859136, -0.0718050748, -0.0878710374, 0.0907980502, 0.0137243588, 0.0385664813, -0.0811820328, 0.110349387, 0.0768834054, 0.00795546919, -0.0456569828, 0.0282176752, 0.0154700279, -0.0885322466, 0.0165600739, 0.0242743976, -0.0512486175, 0.134710655, -0.0499701425, -0.0583954751, -0.00552345859, 0.154104307, -0.0116950572, -0.0820651501, -0.0163469426, -0.0135069452, 0.0772170275, 0.164869577, -0.038731534, 0.0343382843, 0.038465336, -0.136547878, 0.165900111, 0.0708707944, -0.0871039405, 0.0610905364, -0.0182755925, 0.0436922237, 0.050334923, 0.10117881, -0.120075844, -0.0543433391, 0.0410908833, 0.00921290368, -0.185134232, 0.188845456, -0.0383938029, 0.0805517957, -0.0509419739, -0.0603957325, -0.0172433928, -0.130541846, -0.0454375632, -0.0793359652, -0.211888015, 0.124995843, 0.0437471159, -0.0308959447, 0.0279041976, -0.118342206, 0.105505772, 0.0511259995, 0.0539516434, -0.0503093079, 0.0535409003, 0.0130187161, 0.0835435614, -0.0394603834, 0.00284699211, -0.0404362157, 0.0310821142, 0.100886263, 0.0214795284, -0.0352247208, -0.0306135565, -0.00715743657, -0.0303195789, 0.0534922257, -0.0375283137, -0.0457643941, -0.000629881397, -0.131434873, -0.0565093048, 0.0461451709, 0.0843777359, 0.00991098676, -0.024788959, 0.0906525478, 0.0581897125, 0.0328901224, 0.0550921038, -0.0313090384, 0.100491121, 0.0201333854, 0.062505886, 0.00610055029, 0.0380043164, 0.123201445, 0.000253286678, 0.0919304714, 0.0447422415, -0.026506843, 0.0406525247, -0.031096993, 0.0363907889, 0.00152044883, 0.080487363, 0.0627110079, 0.0874619409, -0.0519537963, -0.127790511, 0.00459417142, 0.00682846317, -0.0457928702, 0.0522196144, 0.0924303308, -0.038464509, -0.086849615, -0.160356224, 0.0408706851, 0.095490247, 0.0122903381, 0.0136974026, 0.0707636774, 0.12187013, 0.0146573596, 0.082080096, -0.0131755602, 0.0621735193, 0.0556824245, -0.108569272, -0.076609239, -0.0237353258, -0.00559871644, 0.115258977, 0.191743419, -0.0252263285, 0.0221248195, 0.0200040527, -0.0291588716, 0.0777552426, 0.0164593514, -0.0550806075, 0.0520639569, 0.0552635677, 0.0685346872, -0.0388821326, 0.0650468916, 0.0153346471, -0.0405179337, 0.0162673183, 0.173001856, -0.0572070144, -0.158739433, 0.0474437848, 0.0186247621, -0.0384489819, -0.025185056, 0.0661928505, -0.0579020381, -0.00272467011, -0.0764068663, 0.0295968316, 0.0987232104, -0.0359727219, -0.0147707537, 0.066143699, -0.0598340631, -0.0150769847, -0.119023167, 0.149456948, -0.00938773807, -0.00291891396, 0.0483479574, -0.00588743994, -0.0343669839, -0.00993183814, 0.0173940733, 0.0307970271, 0.0672329217, 0.101019584, 0.0220003892, 0.0636140481, -0.0627934486, -0.0827511996, 0.154713675, -0.0319037884, 0.0897481441, 0.00334194303, 0.0564720593, -0.141668037, 0.0508314818, -0.124435812, 0.0426802114, -0.0346642956, -0.038462922, 0.0804857686, -0.0440798588, 0.025364805, -0.0434191748, 0.11817079, 0.0416435152, -0.0273104757, 0.157931626, -0.0276355185, 0.123778537, -0.0851543918, -0.0501176491, -0.0156346746, 0.0620692186, 0.0481165498, -0.160365403, -0.0612192973, -0.0219055358, 0.0891804919, 0.102926239, -0.0611294955, 0.0267112441, -0.00692081638, -0.0512603037, 0.0842123702, 0.0915205926, -0.080886066, 0.0240275264, -0.138876632, 0.0464169867, -0.0722726956, -0.00494793104, 0.0103371255, 0.053213045, -0.0334090777, 0.128605515, -0.012526406, 0.106924511, -0.0166248754, 0.0593191124, 0.036283195, -0.0135625023, -0.146235406, 0.0251276847, -0.126170442, 0.044441469, -0.0732398182, 0.0177746881, -0.00336868223, 0.0126545895, -0.125758231, -0.0463296212, 0.000760551542, 0.0746849254, -0.0746463388, -0.103783503, -0.21176663, -0.00526075624, -0.196705297, -0.0411077552, 0.0015835464, -0.0345042162, 0.0313511938, -0.0428696312, -0.00496423617, -0.0575777479, -0.040053606, 0.100102738, 0.189796567, -0.0651216954, -0.00988450833, 0.00966881588, 0.00536490232, -0.0826966986, 0.0192021336, -0.0573377647, -0.057390485, -0.00228849798, 0.102888875, 0.0277957432, -0.0254602786, 0.0783777982, 0.0107650012, -0.016606804, 0.0569796078, -0.0925672203, -0.0503984913, -0.0248753857, 0.0985915661, -0.0352421179, -0.119261652, -0.0386371911, 0.0383000784, 0.00993614178, -0.0306219943, 0.0372465104, -0.0314411968, -0.0700695142, 0.0865592733, -0.110574499, 0.0532203689, 0.040152695, -0.11676003, -0.0943935215, -0.0335536599, 0.0619540289, 0.0414873697, 0.0805522352, -0.0169619527, 0.0864372402, -0.0705546364, 0.0452733934, -0.00907016173, -0.064847514, 0.0581720583, -0.114057466, -0.0363059863, 0.0896648243, 0.0615061969, -0.111177891, -0.00641831011, 0.0757474527, 0.0730857551, -0.0960297883, -0.121426262, 0.179821208, -0.0260676071, -0.112282872, -0.0372998379, -0.161543563, 0.0876609832, -0.0419862084, 0.0595651567, 0.047704272, -0.0540253408, -0.246272579, -0.114966534, 0.0210301299, 0.0170566794, -0.058123529, -0.00903307181, 0.108617522, 0.123143926, -0.106013909, 0.140455604, -0.00474341772, 0.0790526718, 0.0832593143, 0.0311025977, -0.0661242753, 0.0702918619, 0.033441782];
    bias_w_0_h : ARRAY[0..63] OF REAL := [-0.0328608565, 0.0353249349, 0.0676618442, 0.0616552494, -0.0419506915, 0.0316758305, -0.0423809998, 0.206494898, 0.050283879, -0.110759951, -0.186538026, -0.0580092184, -0.00209416403, 0.00920274295, 0.0975962356, -0.0612216219, 0.0531282201, -0.1364595, -0.0861791223, 0.0857749358, -0.0629618913, -0.140043736, 0.0230254605, 0.0186893195, 0.274617553, -0.143400162, -0.0180932954, 0.0126953581, 0.00789607875, -0.102969147, -0.00854359195, 0.110707261, 0.101612948, 0.104877286, 0.155045539, 0.120350428, -0.0493059158, -0.109052174, 0.0994426012, 0.120997518, 0.0253830422, 0.0221965443, 0.0652017593, 0.127511516, 0.0405574776, -0.223452628, -0.106970645, -0.184132561, 0.130376682, -0.000101010766, 0.0180109702, 0.0785107389, -0.0454430841, 0.00758665288, -0.0226881728, 0.0657565445, 0.175357804, -0.0399201475, 0.0946480408, -0.0675376579, -0.0944304764, 0.0255580787, 0.114538141, -0.0542288534];
    bias_r_0_h : ARRAY[0..63] OF REAL := [-0.02572597, 0.0358566716, 0.0725965649, 0.0658897385, -0.0349466167, 0.0312440004, -0.0520541295, 0.229264349, 0.053602159, -0.114199713, -0.188671976, -0.0562148206, -0.00815096032, 0.042876251, 0.128237545, -0.0830967203, 0.0521300212, -0.172336012, -0.0845128968, 0.120621495, -0.0981689841, -0.171339214, 0.0380116738, -0.00155168783, 0.27826634, -0.166642264, -0.0124149593, 0.00777016627, 0.0202645063, -0.110686347, -0.00758656999, 0.116100229, 0.137906507, 0.108378269, 0.189799592, 0.156204492, -0.0414909273, -0.111529253, 0.11403127, 0.138321266, 0.0324263275, 0.0199548732, 0.0663017482, 0.155816868, 0.0454924814, -0.249957547, -0.124289908, -0.17978096, 0.148145601, 0.0183632877, 0.0141077479, 0.0873264968, -0.0591249838, 0.00012417727, -0.0334720835, 0.0621513799, 0.192247525, -0.0562552325, 0.11991331, -0.0805595443, -0.108275652, 0.0187377501, 0.144540057, -0.0489126071];
